REGION Network 22: Salidas Mesas
   RUNG wire#powerrail
      Contact( TRUE )
      wire#w1
      Contact( #Avance_E1 )
      Coil( "DB900_Estado_Mesas".EstadoVI[#Mesa].Sa_Rod_Avance )
   END_RUNG
   RUNG wire#w1
      Contact( #Avance_S2 )
      Coil( "DB900_Estado_Mesas".EstadoVI[#Mesa].Sa_Cad_Avance )
   END_RUNG
   RUNG wire#w1
      Contact( #TEMP_MA_TR_Pos_E1 )
      Coil( "DB900_Estado_Mesas".EstadoVI[#Mesa].Sa_Trans_Sub )
   END_RUNG
   RUNG wire#w1
      Contact( #TEMP_MA_TR_Pos_S2 )
      Coil( "DB900_Estado_Mesas".EstadoVI[#Mesa].Sa_Trans_Baj )
   END_RUNG
   // the same network as SCL:
   "DB900_Estado_Mesas".EstadoVI[#Mesa].Sa_Rod_Avance := TRUE AND #Avance_E1;
   "DB900_Estado_Mesas".EstadoVI[#Mesa].Sa_Cad_Avance := TRUE AND #Avance_S2;
   "DB900_Estado_Mesas".EstadoVI[#Mesa].Sa_Trans_Sub := TRUE AND #TEMP_MA_TR_Pos_E1;
   "DB900_Estado_Mesas".EstadoVI[#Mesa].Sa_Trans_Baj := TRUE AND #TEMP_MA_TR_Pos_S2;
END_REGION

REGION Network 23: Etapa MESA en RESET
   RUNG wire#powerrail
      Contact( TRUE )
      wire#w1
      Contact( "DB902_Estado_ZonaMesa".EstadoMesas[#Mesa].PerReset_CBx )
      Coil( "DB900_Estado_Mesas".EstadoVI[#Mesa].Etapas_Reset )
   END_RUNG
   RUNG wire#w1
      Contact( #Avance_E1 )
      Coil( "DB900_Estado_Mesas".EstadoVI[#Mesa].Etapas_Carga_E1 )
   END_RUNG
   RUNG wire#w1
      Contact( #Avance_S2 )
      Coil( "DB900_Estado_Mesas".EstadoVI[#Mesa].Etapas_Descarga_S2 )
   END_RUNG
   RUNG wire#w1
      I_Contact( #Avance_E1 )
      I_Contact( #Avance_S2 )
      Contact( #PhsMx )
      Coil( "DB900_Estado_Mesas".EstadoVI[#Mesa].Etapa_Cargada )
   END_RUNG
   RUNG wire#w1
      I_Contact( #Avance_E1 )
      I_Contact( #Avance_S2 )
      I_Contact( #PhsMx )
      Coil( "DB900_Estado_Mesas".EstadoVI[#Mesa].Etapa_Vacia )
   END_RUNG
   // the same network as SCL:
   "DB900_Estado_Mesas".EstadoVI[#Mesa].Etapas_Reset := TRUE AND "DB902_Estado_ZonaMesa".EstadoMesas[#Mesa].PerReset_CBx;
   "DB900_Estado_Mesas".EstadoVI[#Mesa].Etapas_Carga_E1 := TRUE AND #Avance_E1;
   "DB900_Estado_Mesas".EstadoVI[#Mesa].Etapas_Descarga_S2 := TRUE AND #Avance_S2;
   "DB900_Estado_Mesas".EstadoVI[#Mesa].Etapa_Cargada := TRUE AND NOT #Avance_E1 AND NOT #Avance_S2 AND #PhsMx;
   "DB900_Estado_Mesas".EstadoVI[#Mesa].Etapa_Vacia := TRUE AND NOT #Avance_E1 AND NOT #Avance_S2 AND NOT #PhsMx;
END_REGION

REGION Network 24
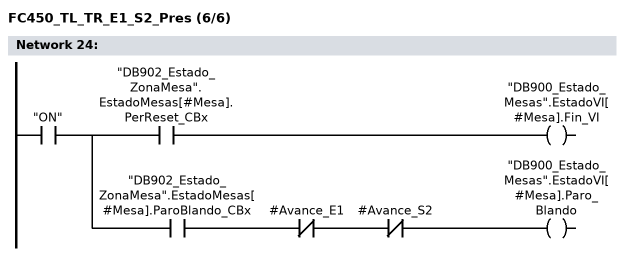
   RUNG wire#powerrail
      Contact( "ON" )
      wire#w1
      Contact( "DB902_Estado_ZonaMesa".EstadoMesas[#Mesa].PerReset_CBx )
      Coil( "DB900_Estado_Mesas".EstadoVI[#Mesa].Fin_VI )
   END_RUNG
   RUNG wire#w1
      Contact( "DB902_Estado_ZonaMesa".EstadoMesas[#Mesa].ParoBlando_CBx )
      I_Contact( #Avance_E1 )
      I_Contact( #Avance_S2 )
      Coil( "DB900_Estado_Mesas".EstadoVI[#Mesa].Paro_Blando )
   END_RUNG
   // the same network as SCL:
   "DB900_Estado_Mesas".EstadoVI[#Mesa].Fin_VI := "ON" AND "DB902_Estado_ZonaMesa".EstadoMesas[#Mesa].PerReset_CBx;
   "DB900_Estado_Mesas".EstadoVI[#Mesa].Paro_Blando := "ON" AND "DB902_Estado_ZonaMesa".EstadoMesas[#Mesa].ParoBlando_CBx AND NOT #Avance_E1 AND NOT #Avance_S2;
END_REGION
END_FUNCTION

FUNCTION "FC451_TL_TR_E1E2_S3_Simul_Pres" : Void   // FC451, LAD
{ S7_Optimized_Access := 'FALSE' }
AUTHOR : TLigero
NAME : 20160208
VERSION : 3.2
// stored: AutoNumber false, SetENOAutomatically false
   VAR_INPUT
      Mesa : UInt;
      En_Tension : Bool;
      PhsMx : Bool;
      Termico_E1 : Bool;
      Termico_E2 : Bool;
      PosTR_E1 : Bool;
      PosTR_E2 : Bool;
      PosTR_EnReposo_E2 : Bool;   // Si está a false la posición de reposo será E1
      Avance_E1_Tx_Ok : Bool;
      Avance_E2_Tx_Ok : Bool;
      AVTF_Ent_M1 : Bool;
      AVTF_Ent_M2 : Bool;
      NXT_Avance : Bool;
      PTF_Mx_MSig : Bool;
      V_CNT_ApHsMx : UDInt;
      V_Paro : UDInt;
      V_Separacion : UDInt;
      V_Caja_Max : UDInt;
      V_CNT_pHsMx_E1 : UDInt;
      V_CNT_pHsMx_E2 : UDInt;
      V_TOut_Tx_Mx : UDInt;
      V_TOut_TR : UDInt;
      V_Reparto_E1_E2 : UDInt;   // cuantas cajas de E1 dejamos pasar antes de forzar una entrada por E2 (en caso de que siempre haya cajas esperando en ambas entradas)
   END_VAR
   VAR_OUTPUT
      PTF_Ent_M1 : Bool;
      PTF_Ent_M2 : Bool;
      AVTF_Mx_MSig : Bool;
   END_VAR
   VAR_IN_OUT
      NXT_Descarga_Act : Bool;
      Mem_FP_pHs : Bool;
      Mem_FN_pHs : Bool;
   END_VAR
   VAR_TEMP
      Aux_Parar : Bool;
      Mem_CNT_Separacion : Bool;
      Mem_CNT_Pres : Bool;
      atasco : Bool;
      tout_tr : Bool;
      Mem_CNT_Tmp_AUS : Bool;
      Mem_CNT_Tmp_Paro : Bool;
      TEMP_MA_Ir_Pos_E2 : Bool;
      TEMP_MA_Ir_Pos_E1 : Bool;
      ok_tension : Bool;
      Valor_presencia : UDInt;
   END_VAR
   VAR_TEMP   // added for the SCL form of the ladder/FBD networks
      _w1 : Bool;
   END_VAR
BEGIN

REGION Network 1: Marca General Error
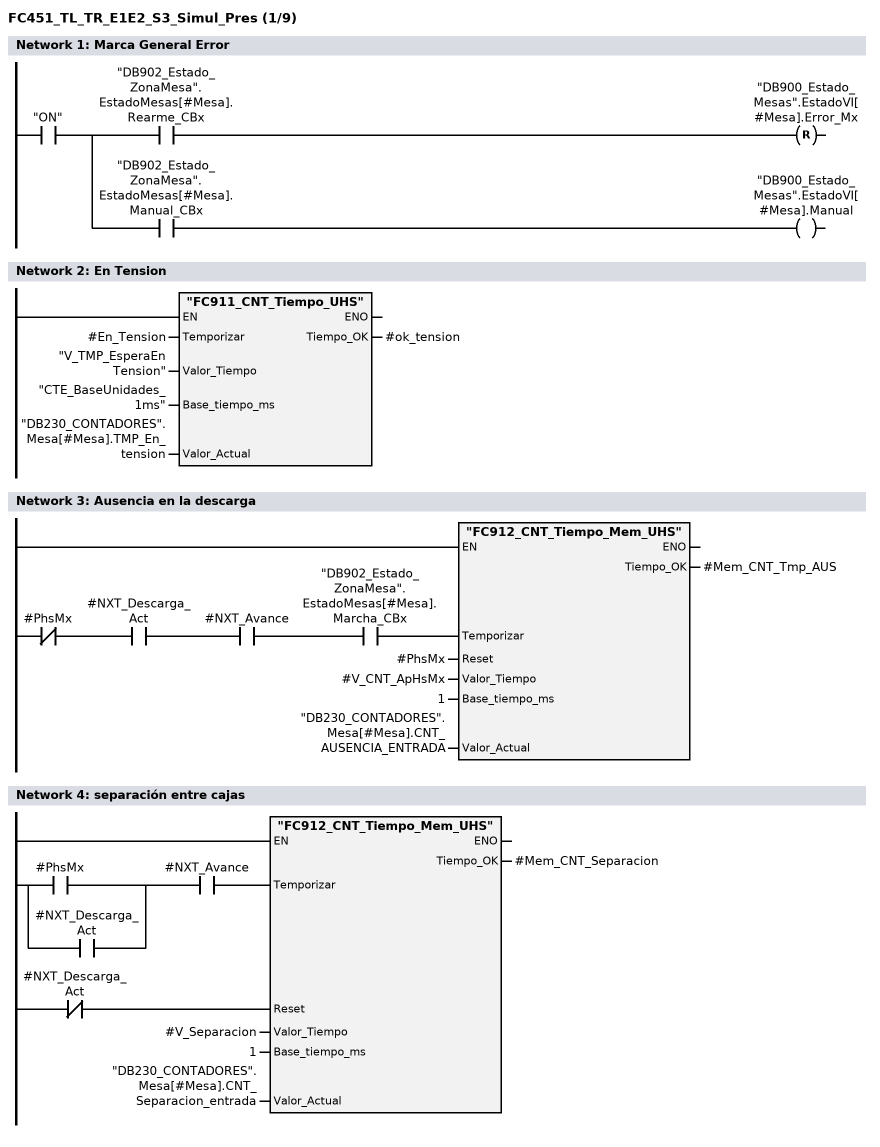
   RUNG wire#powerrail
      Contact( "ON" )
      wire#w1
      Contact( "DB902_Estado_ZonaMesa".EstadoMesas[#Mesa].Rearme_CBx )
      R_Coil( "DB900_Estado_Mesas".EstadoVI[#Mesa].Error_Mx )
   END_RUNG
   RUNG wire#w1
      Contact( "DB902_Estado_ZonaMesa".EstadoMesas[#Mesa].Manual_CBx )
      Coil( "DB900_Estado_Mesas".EstadoVI[#Mesa].Manual )
   END_RUNG
   // the same network as SCL:
   IF "ON" AND "DB902_Estado_ZonaMesa".EstadoMesas[#Mesa].Rearme_CBx THEN
       "DB900_Estado_Mesas".EstadoVI[#Mesa].Error_Mx := FALSE;
   END_IF;
   "DB900_Estado_Mesas".EstadoVI[#Mesa].Manual := "ON" AND "DB902_Estado_ZonaMesa".EstadoMesas[#Mesa].Manual_CBx;
END_REGION

REGION Network 2: En Tension
   RUNG wire#powerrail
      "FC911_CNT_Tiempo_UHS"(Temporizar := #En_Tension, Valor_Tiempo := "V_TMP_EsperaEnTension", Base_tiempo_ms := "CTE_BaseUnidades_1ms", Valor_Actual := "DB230_CONTADORES".Mesa[#Mesa].TMP_En_tension, Tiempo_OK => #ok_tension)
   END_RUNG
   // the same network as SCL:
   "FC911_CNT_Tiempo_UHS"(Temporizar := #En_Tension,
                          Valor_Tiempo := "V_TMP_EsperaEnTension",
                          Base_tiempo_ms := "CTE_BaseUnidades_1ms",
                          Valor_Actual := "DB230_CONTADORES".Mesa[#Mesa].TMP_En_tension,
                          Tiempo_OK => #ok_tension);
END_REGION

REGION Network 3: Ausencia en la descarga
   RUNG wire#powerrail
      "FC912_CNT_Tiempo_Mem_UHS"(Temporizar := wire#w1, Reset := #PhsMx, Valor_Tiempo := #V_CNT_ApHsMx, Base_tiempo_ms := 1, Valor_Actual := "DB230_CONTADORES".Mesa[#Mesa].CNT_AUSENCIA_ENTRADA, Tiempo_OK => #Mem_CNT_Tmp_AUS)
   END_RUNG
   RUNG wire#powerrail
      I_Contact( #PhsMx )
      Contact( #NXT_Descarga_Act )
      Contact( #NXT_Avance )
      Contact( "DB902_Estado_ZonaMesa".EstadoMesas[#Mesa].Marcha_CBx )
   END_RUNG wire#w1
   // the same network as SCL:
   "FC912_CNT_Tiempo_Mem_UHS"(Temporizar := NOT #PhsMx AND #NXT_Descarga_Act AND #NXT_Avance AND "DB902_Estado_ZonaMesa".EstadoMesas[#Mesa].Marcha_CBx,
                           Reset := #PhsMx,
                           Valor_Tiempo := #V_CNT_ApHsMx,
                           Base_tiempo_ms := 1,
                           Valor_Actual := "DB230_CONTADORES".Mesa[#Mesa].CNT_AUSENCIA_ENTRADA,
                           Tiempo_OK => #Mem_CNT_Tmp_AUS);
END_REGION

REGION Network 4: separación entre cajas
   RUNG wire#powerrail
      "FC912_CNT_Tiempo_Mem_UHS"(Temporizar := wire#w2, Reset := wire#w3, Valor_Tiempo := #V_Separacion, Base_tiempo_ms := 1, Valor_Actual := "DB230_CONTADORES".Mesa[#Mesa].CNT_Separacion_entrada, Tiempo_OK => #Mem_CNT_Separacion)
   END_RUNG
   RUNG wire#powerrail
      Contact( #PhsMx )
      wire#w1
      Contact( #NXT_Avance )
   END_RUNG wire#w2
   RUNG wire#powerrail
      Contact( #NXT_Descarga_Act )
   END_RUNG wire#w1
   RUNG wire#powerrail
      I_Contact( #NXT_Descarga_Act )
   END_RUNG wire#w3
   // the same network as SCL:
   "FC912_CNT_Tiempo_Mem_UHS"(Temporizar := (#PhsMx OR #NXT_Descarga_Act) AND #NXT_Avance,
                           Reset := NOT #NXT_Descarga_Act,
                           Valor_Tiempo := #V_Separacion,
                           Base_tiempo_ms := 1,
                           Valor_Actual := "DB230_CONTADORES".Mesa[#Mesa].CNT_Separacion_entrada,
                           Tiempo_OK => #Mem_CNT_Separacion);
END_REGION

REGION Network 5: Valor de presencia
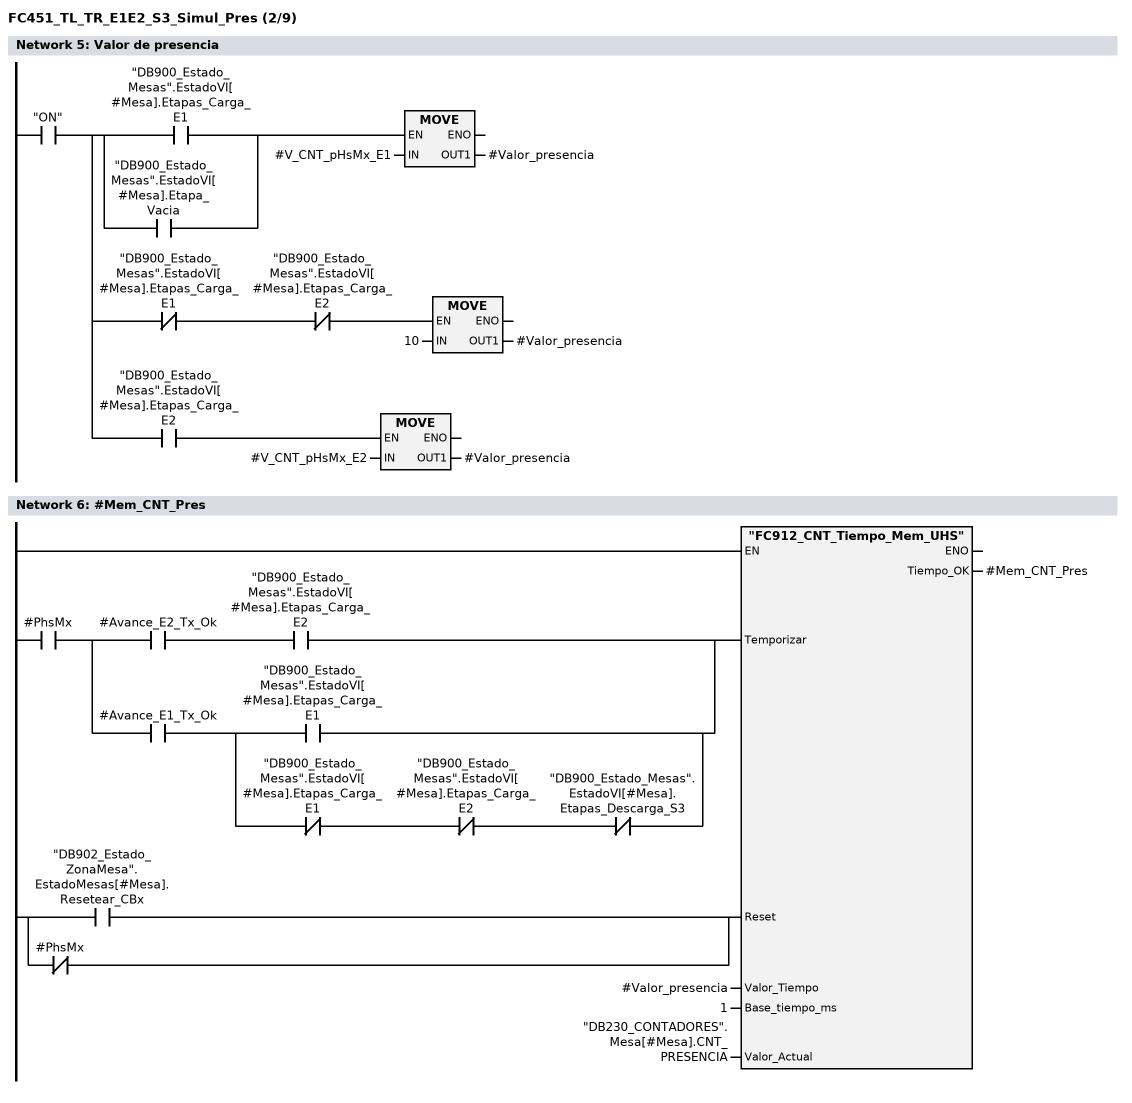
   RUNG wire#powerrail
      Contact( "ON" )
      wire#w1
      Contact( "DB900_Estado_Mesas".EstadoVI[#Mesa].Etapas_Carga_E1 )
      wire#w2
      Move(in := #V_CNT_pHsMx_E1, out1 => #Valor_presencia)
   END_RUNG
   RUNG wire#w1
      Contact( "DB900_Estado_Mesas".EstadoVI[#Mesa].Etapa_Vacia )
   END_RUNG wire#w2
   RUNG wire#w1
      I_Contact( "DB900_Estado_Mesas".EstadoVI[#Mesa].Etapas_Carga_E1 )
      I_Contact( "DB900_Estado_Mesas".EstadoVI[#Mesa].Etapas_Carga_E2 )
      Move(in := 10, out1 => #Valor_presencia)
   END_RUNG
   RUNG wire#w1
      Contact( "DB900_Estado_Mesas".EstadoVI[#Mesa].Etapas_Carga_E2 )
      Move(in := #V_CNT_pHsMx_E2, out1 => #Valor_presencia)
   END_RUNG
   // the same network as SCL:
   IF "ON" AND ("DB900_Estado_Mesas".EstadoVI[#Mesa].Etapas_Carga_E1 OR "DB900_Estado_Mesas".EstadoVI[#Mesa].Etapa_Vacia) THEN
       #Valor_presencia := #V_CNT_pHsMx_E1;
   END_IF;
   IF "ON" AND NOT "DB900_Estado_Mesas".EstadoVI[#Mesa].Etapas_Carga_E1 AND NOT "DB900_Estado_Mesas".EstadoVI[#Mesa].Etapas_Carga_E2 THEN
       #Valor_presencia := 10;
   END_IF;
   IF "ON" AND "DB900_Estado_Mesas".EstadoVI[#Mesa].Etapas_Carga_E2 THEN
       #Valor_presencia := #V_CNT_pHsMx_E2;
   END_IF;
END_REGION

REGION Network 6: #Mem_CNT_Pres
   RUNG wire#powerrail
      "FC912_CNT_Tiempo_Mem_UHS"(Temporizar := wire#w3, Reset := wire#w4, Valor_Tiempo := #Valor_presencia, Base_tiempo_ms := 1, Valor_Actual := "DB230_CONTADORES".Mesa[#Mesa].CNT_PRESENCIA, Tiempo_OK => #Mem_CNT_Pres)
   END_RUNG
   RUNG wire#powerrail
      Contact( #PhsMx )
      wire#w1
      Contact( #Avance_E2_Tx_Ok )
      Contact( "DB900_Estado_Mesas".EstadoVI[#Mesa].Etapas_Carga_E2 )
   END_RUNG wire#w3
   RUNG wire#w1
      Contact( #Avance_E1_Tx_Ok )
      wire#w2
      Contact( "DB900_Estado_Mesas".EstadoVI[#Mesa].Etapas_Carga_E1 )
   END_RUNG wire#w3
   RUNG wire#w2
      I_Contact( "DB900_Estado_Mesas".EstadoVI[#Mesa].Etapas_Carga_E1 )
      I_Contact( "DB900_Estado_Mesas".EstadoVI[#Mesa].Etapas_Carga_E2 )
      I_Contact( "DB900_Estado_Mesas".EstadoVI[#Mesa].Etapas_Descarga_S3 )
   END_RUNG wire#w3
   RUNG wire#powerrail
      Contact( "DB902_Estado_ZonaMesa".EstadoMesas[#Mesa].Resetear_CBx )
   END_RUNG wire#w4
   RUNG wire#powerrail
      I_Contact( #PhsMx )
   END_RUNG wire#w4
   // the same network as SCL:
   "FC912_CNT_Tiempo_Mem_UHS"(Temporizar := #PhsMx AND ((#Avance_E2_Tx_Ok AND "DB900_Estado_Mesas".EstadoVI[#Mesa].Etapas_Carga_E2) OR (#Avance_E1_Tx_Ok AND ("DB900_Estado_Mesas".EstadoVI[#Mesa].Etapas_Carga_E1 OR (NOT "DB900_Estado_Mesas".EstadoVI[#Mesa].Etapas_Carga_E1 AND NOT "DB900_Estado_Mesas".EstadoVI[#Mesa].Etapas_Carga_E2 AND NOT "DB900_Estado_Mesas".EstadoVI[#Mesa].Etapas_Descarga_S3)))),
                           Reset := "DB902_Estado_ZonaMesa".EstadoMesas[#Mesa].Resetear_CBx OR NOT #PhsMx,
                           Valor_Tiempo := #Valor_presencia,
                           Base_tiempo_ms := 1,
                           Valor_Actual := "DB230_CONTADORES".Mesa[#Mesa].CNT_PRESENCIA,
                           Tiempo_OK => #Mem_CNT_Pres);
END_REGION

REGION Network 7: Temporizador PARO
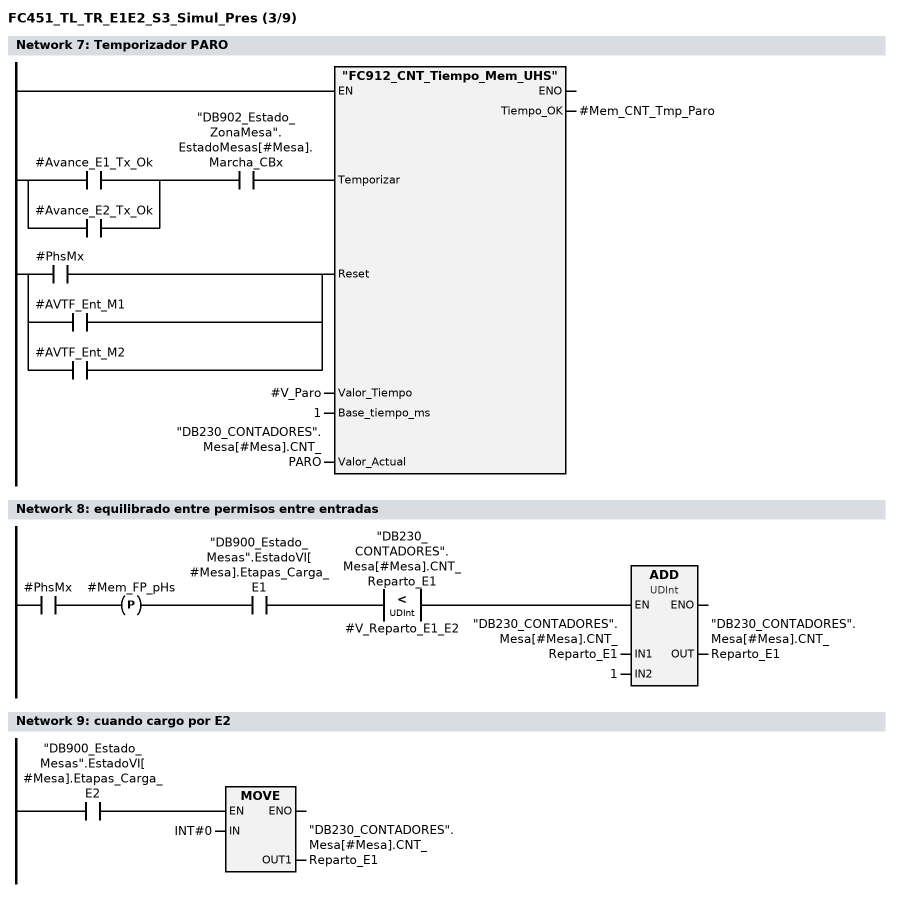
   RUNG wire#powerrail
      "FC912_CNT_Tiempo_Mem_UHS"(Temporizar := wire#w2, Reset := wire#w3, Valor_Tiempo := #V_Paro, Base_tiempo_ms := 1, Valor_Actual := "DB230_CONTADORES".Mesa[#Mesa].CNT_PARO, Tiempo_OK => #Mem_CNT_Tmp_Paro)
   END_RUNG
   RUNG wire#powerrail
      Contact( #Avance_E1_Tx_Ok )
      wire#w1
      Contact( "DB902_Estado_ZonaMesa".EstadoMesas[#Mesa].Marcha_CBx )
   END_RUNG wire#w2
   RUNG wire#powerrail
      Contact( #Avance_E2_Tx_Ok )
   END_RUNG wire#w1
   RUNG wire#powerrail
      Contact( #PhsMx )
   END_RUNG wire#w3
   RUNG wire#powerrail
      Contact( #AVTF_Ent_M1 )
   END_RUNG wire#w3
   RUNG wire#powerrail
      Contact( #AVTF_Ent_M2 )
   END_RUNG wire#w3
   // the same network as SCL:
   "FC912_CNT_Tiempo_Mem_UHS"(Temporizar := (#Avance_E1_Tx_Ok OR #Avance_E2_Tx_Ok) AND "DB902_Estado_ZonaMesa".EstadoMesas[#Mesa].Marcha_CBx,
                           Reset := #PhsMx OR #AVTF_Ent_M1 OR #AVTF_Ent_M2,
                           Valor_Tiempo := #V_Paro,
                           Base_tiempo_ms := 1,
                           Valor_Actual := "DB230_CONTADORES".Mesa[#Mesa].CNT_PARO,
                           Tiempo_OK => #Mem_CNT_Tmp_Paro);
END_REGION

REGION Network 8: equilibrado entre permisos entre entradas
   RUNG wire#powerrail
      Contact( #PhsMx )
      P_Trig( #Mem_FP_pHs )
      Contact( "DB900_Estado_Mesas".EstadoVI[#Mesa].Etapas_Carga_E1 )
      { S7_Templates := "SrcType := UDInt" } LT_Contact(in1 := "DB230_CONTADORES".Mesa[#Mesa].CNT_Reparto_E1, in2 := #V_Reparto_E1_E2)
      { S7_Templates := "SrcType := UDInt"; S7_GenerateENO := "TRUE" } Add(in1 := "DB230_CONTADORES".Mesa[#Mesa].CNT_Reparto_E1, in2 := 1, out => "DB230_CONTADORES".Mesa[#Mesa].CNT_Reparto_E1)
   END_RUNG
   // the same network as SCL:
   #_w1 := #PhsMx AND NOT #Mem_FP_pHs;   // rising edge
   #Mem_FP_pHs := #PhsMx;
   IF #_w1 AND "DB900_Estado_Mesas".EstadoVI[#Mesa].Etapas_Carga_E1 AND ("DB230_CONTADORES".Mesa[#Mesa].CNT_Reparto_E1 < #V_Reparto_E1_E2) THEN
       "DB230_CONTADORES".Mesa[#Mesa].CNT_Reparto_E1 := "DB230_CONTADORES".Mesa[#Mesa].CNT_Reparto_E1 + 1;
   END_IF;
END_REGION

REGION Network 9: cuando cargo por E2
   RUNG wire#powerrail
      Contact( "DB900_Estado_Mesas".EstadoVI[#Mesa].Etapas_Carga_E2 )
      { S7_GenerateENO := "TRUE" } Move(in := INT#0, out1 => "DB230_CONTADORES".Mesa[#Mesa].CNT_Reparto_E1)
   END_RUNG
   // the same network as SCL:
   IF "DB900_Estado_Mesas".EstadoVI[#Mesa].Etapas_Carga_E2 THEN
       "DB230_CONTADORES".Mesa[#Mesa].CNT_Reparto_E1 := INT#0;
   END_IF;
END_REGION

REGION Network 10: Etapas carga E1
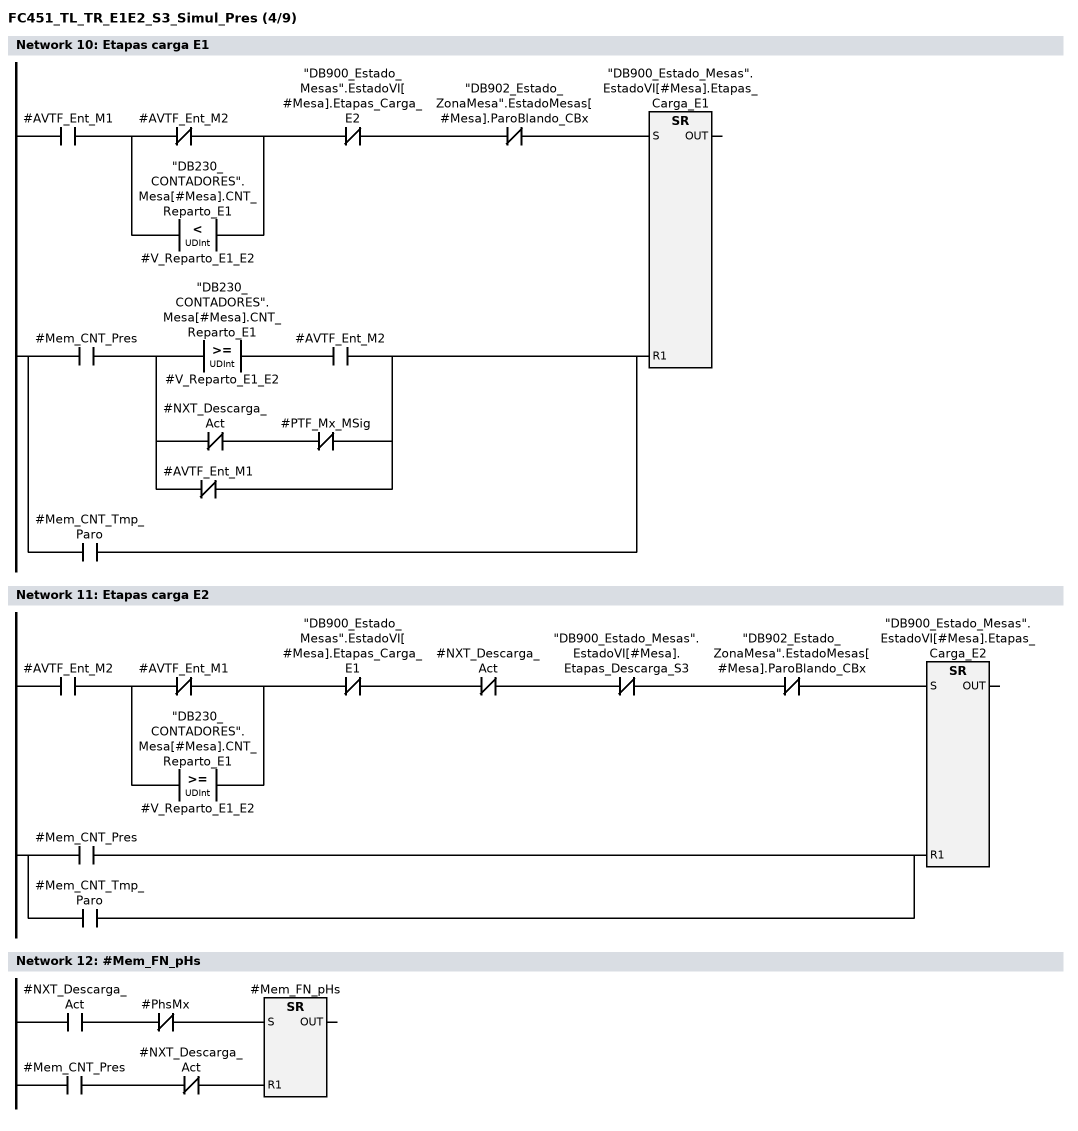
   RUNG wire#powerrail
      Contact( #AVTF_Ent_M1 )
      wire#w1
      I_Contact( #AVTF_Ent_M2 )
      wire#w2
      I_Contact( "DB900_Estado_Mesas".EstadoVI[#Mesa].Etapas_Carga_E2 )
      I_Contact( "DB902_Estado_ZonaMesa".EstadoMesas[#Mesa].ParoBlando_CBx )
      S_SR(operand := "DB900_Estado_Mesas".EstadoVI[#Mesa].Etapas_Carga_E1, r1 := wire#w4)
   END_RUNG
   RUNG wire#w1
      { S7_Templates := "SrcType := UDInt" } LT_Contact(in1 := "DB230_CONTADORES".Mesa[#Mesa].CNT_Reparto_E1, in2 := #V_Reparto_E1_E2)
   END_RUNG wire#w2
   RUNG wire#powerrail
      Contact( #Mem_CNT_Pres )
      wire#w3
      { S7_Templates := "SrcType := UDInt" } GE_Contact(in1 := "DB230_CONTADORES".Mesa[#Mesa].CNT_Reparto_E1, in2 := #V_Reparto_E1_E2)
      Contact( #AVTF_Ent_M2 )
   END_RUNG wire#w4
   RUNG wire#w3
      I_Contact( #NXT_Descarga_Act )
      I_Contact( #PTF_Mx_MSig )
   END_RUNG wire#w4
   RUNG wire#w3
      I_Contact( #AVTF_Ent_M1 )
   END_RUNG wire#w4
   RUNG wire#powerrail
      Contact( #Mem_CNT_Tmp_Paro )
   END_RUNG wire#w4
   // the same network as SCL:
   #_w1 := (#Mem_CNT_Pres AND ((("DB230_CONTADORES".Mesa[#Mesa].CNT_Reparto_E1 >= #V_Reparto_E1_E2) AND #AVTF_Ent_M2) OR (NOT #NXT_Descarga_Act AND NOT #PTF_Mx_MSig) OR NOT #AVTF_Ent_M1)) OR #Mem_CNT_Tmp_Paro;
   IF #AVTF_Ent_M1 AND (NOT #AVTF_Ent_M2 OR ("DB230_CONTADORES".Mesa[#Mesa].CNT_Reparto_E1 < #V_Reparto_E1_E2)) AND NOT "DB900_Estado_Mesas".EstadoVI[#Mesa].Etapas_Carga_E2 AND NOT "DB902_Estado_ZonaMesa".EstadoMesas[#Mesa].ParoBlando_CBx THEN
       "DB900_Estado_Mesas".EstadoVI[#Mesa].Etapas_Carga_E1 := TRUE;   // SR flip-flop
   END_IF;
   IF #_w1 THEN "DB900_Estado_Mesas".EstadoVI[#Mesa].Etapas_Carga_E1 := FALSE; END_IF;
END_REGION

REGION Network 11: Etapas carga E2
   RUNG wire#powerrail
      Contact( #AVTF_Ent_M2 )
      wire#w1
      I_Contact( #AVTF_Ent_M1 )
      wire#w2
      I_Contact( "DB900_Estado_Mesas".EstadoVI[#Mesa].Etapas_Carga_E1 )
      I_Contact( #NXT_Descarga_Act )
      I_Contact( "DB900_Estado_Mesas".EstadoVI[#Mesa].Etapas_Descarga_S3 )
      I_Contact( "DB902_Estado_ZonaMesa".EstadoMesas[#Mesa].ParoBlando_CBx )
      S_SR(operand := "DB900_Estado_Mesas".EstadoVI[#Mesa].Etapas_Carga_E2, r1 := wire#w3)
   END_RUNG
   RUNG wire#w1
      { S7_Templates := "SrcType := UDInt" } GE_Contact(in1 := "DB230_CONTADORES".Mesa[#Mesa].CNT_Reparto_E1, in2 := #V_Reparto_E1_E2)
   END_RUNG wire#w2
   RUNG wire#powerrail
      Contact( #Mem_CNT_Pres )
   END_RUNG wire#w3
   RUNG wire#powerrail
      Contact( #Mem_CNT_Tmp_Paro )
   END_RUNG wire#w3
   // the same network as SCL:
   IF #AVTF_Ent_M2 AND (NOT #AVTF_Ent_M1 OR ("DB230_CONTADORES".Mesa[#Mesa].CNT_Reparto_E1 >= #V_Reparto_E1_E2)) AND NOT "DB900_Estado_Mesas".EstadoVI[#Mesa].Etapas_Carga_E1 AND NOT #NXT_Descarga_Act AND NOT "DB900_Estado_Mesas".EstadoVI[#Mesa].Etapas_Descarga_S3 AND NOT "DB902_Estado_ZonaMesa".EstadoMesas[#Mesa].ParoBlando_CBx THEN
       "DB900_Estado_Mesas".EstadoVI[#Mesa].Etapas_Carga_E2 := TRUE;   // SR flip-flop
   END_IF;
   IF #Mem_CNT_Pres OR #Mem_CNT_Tmp_Paro THEN
       "DB900_Estado_Mesas".EstadoVI[#Mesa].Etapas_Carga_E2 := FALSE;
   END_IF;
END_REGION

REGION Network 12: #Mem_FN_pHs
   RUNG wire#powerrail
      Contact( #NXT_Descarga_Act )
      I_Contact( #PhsMx )
      S_SR(operand := #Mem_FN_pHs, r1 := wire#w1)
   END_RUNG
   RUNG wire#powerrail
      Contact( #Mem_CNT_Pres )
      I_Contact( #NXT_Descarga_Act )
   END_RUNG wire#w1
   // the same network as SCL:
   IF #NXT_Descarga_Act AND NOT #PhsMx THEN
       #Mem_FN_pHs := TRUE;   // SR flip-flop
   END_IF;
   IF #Mem_CNT_Pres AND NOT #NXT_Descarga_Act THEN #Mem_FN_pHs := FALSE; END_IF;
END_REGION

REGION Network 13: #Aux_Parar
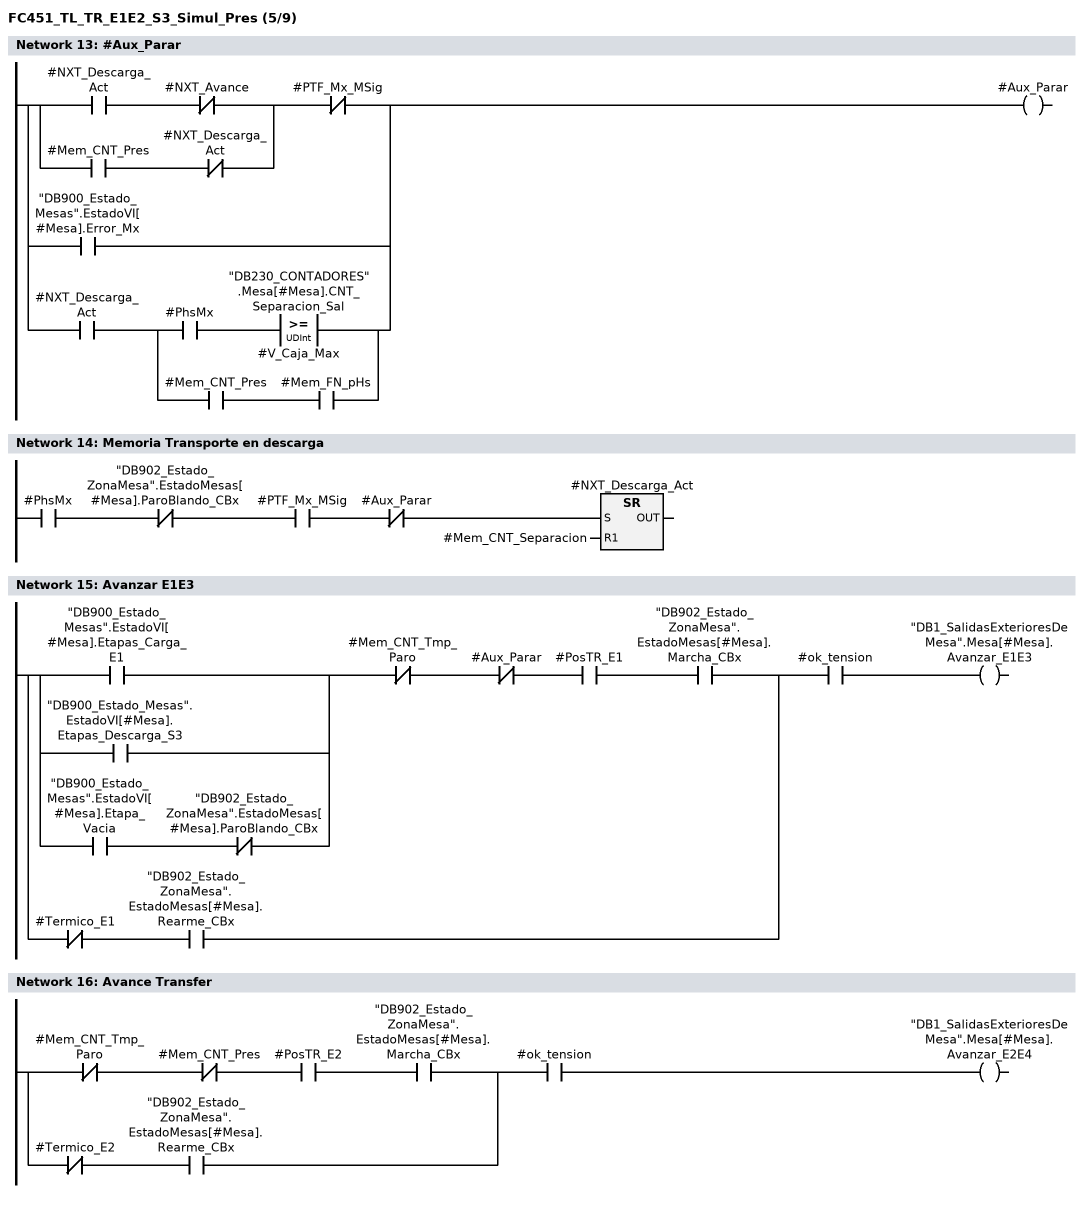
   RUNG wire#powerrail
      Contact( #NXT_Descarga_Act )
      I_Contact( #NXT_Avance )
      wire#w1
      I_Contact( #PTF_Mx_MSig )
      wire#w2
      Coil( #Aux_Parar )
   END_RUNG
   RUNG wire#powerrail
      Contact( #Mem_CNT_Pres )
      I_Contact( #NXT_Descarga_Act )
   END_RUNG wire#w1
   RUNG wire#powerrail
      Contact( "DB900_Estado_Mesas".EstadoVI[#Mesa].Error_Mx )
   END_RUNG wire#w2
   RUNG wire#powerrail
      Contact( #NXT_Descarga_Act )
      wire#w3
      Contact( #PhsMx )
      { S7_Templates := "SrcType := UDInt" } GE_Contact(in1 := "DB230_CONTADORES".Mesa[#Mesa].CNT_Separacion_Sal, in2 := #V_Caja_Max)
   END_RUNG wire#w2
   RUNG wire#w3
      Contact( #Mem_CNT_Pres )
      Contact( #Mem_FN_pHs )
   END_RUNG wire#w2
   // the same network as SCL:
   #Aux_Parar := (((#NXT_Descarga_Act AND NOT #NXT_Avance) OR (#Mem_CNT_Pres AND NOT #NXT_Descarga_Act)) AND NOT #PTF_Mx_MSig) OR "DB900_Estado_Mesas".EstadoVI[#Mesa].Error_Mx OR (#NXT_Descarga_Act AND ((#PhsMx AND ("DB230_CONTADORES".Mesa[#Mesa].CNT_Separacion_Sal >= #V_Caja_Max)) OR (#Mem_CNT_Pres AND #Mem_FN_pHs)));
END_REGION

REGION Network 14: Memoria Transporte en descarga
   RUNG wire#powerrail
      Contact( #PhsMx )
      I_Contact( "DB902_Estado_ZonaMesa".EstadoMesas[#Mesa].ParoBlando_CBx )
      Contact( #PTF_Mx_MSig )
      I_Contact( #Aux_Parar )
      S_SR(operand := #NXT_Descarga_Act, r1 := #Mem_CNT_Separacion)
   END_RUNG
   // the same network as SCL:
   IF #PhsMx AND NOT "DB902_Estado_ZonaMesa".EstadoMesas[#Mesa].ParoBlando_CBx AND #PTF_Mx_MSig AND NOT #Aux_Parar THEN
       #NXT_Descarga_Act := TRUE;   // SR flip-flop
   END_IF;
   IF #Mem_CNT_Separacion THEN #NXT_Descarga_Act := FALSE; END_IF;
END_REGION

REGION Network 15: Avanzar E1E3
   RUNG wire#powerrail
      Contact( "DB900_Estado_Mesas".EstadoVI[#Mesa].Etapas_Carga_E1 )
      wire#w1
      I_Contact( #Mem_CNT_Tmp_Paro )
      I_Contact( #Aux_Parar )
      Contact( #PosTR_E1 )
      Contact( "DB902_Estado_ZonaMesa".EstadoMesas[#Mesa].Marcha_CBx )
      wire#w2
      Contact( #ok_tension )
      Coil( "DB1_SalidasExterioresDeMesa".Mesa[#Mesa].Avanzar_E1E3 )
   END_RUNG
   RUNG wire#powerrail
      Contact( "DB900_Estado_Mesas".EstadoVI[#Mesa].Etapas_Descarga_S3 )
   END_RUNG wire#w1
   RUNG wire#powerrail
      Contact( "DB900_Estado_Mesas".EstadoVI[#Mesa].Etapa_Vacia )
      I_Contact( "DB902_Estado_ZonaMesa".EstadoMesas[#Mesa].ParoBlando_CBx )
   END_RUNG wire#w1
   RUNG wire#powerrail
      I_Contact( #Termico_E1 )
      Contact( "DB902_Estado_ZonaMesa".EstadoMesas[#Mesa].Rearme_CBx )
   END_RUNG wire#w2
   // the same network as SCL:
   "DB1_SalidasExterioresDeMesa".Mesa[#Mesa].Avanzar_E1E3 := ((("DB900_Estado_Mesas".EstadoVI[#Mesa].Etapas_Carga_E1 OR "DB900_Estado_Mesas".EstadoVI[#Mesa].Etapas_Descarga_S3 OR ("DB900_Estado_Mesas".EstadoVI[#Mesa].Etapa_Vacia AND NOT "DB902_Estado_ZonaMesa".EstadoMesas[#Mesa].ParoBlando_CBx)) AND NOT #Mem_CNT_Tmp_Paro AND NOT #Aux_Parar AND #PosTR_E1 AND "DB902_Estado_ZonaMesa".EstadoMesas[#Mesa].Marcha_CBx) OR (NOT #Termico_E1 AND "DB902_Estado_ZonaMesa".EstadoMesas[#Mesa].Rearme_CBx)) AND #ok_tension;
END_REGION

REGION Network 16: Avance Transfer
   RUNG wire#powerrail
      I_Contact( #Mem_CNT_Tmp_Paro )
      I_Contact( #Mem_CNT_Pres )
      Contact( #PosTR_E2 )
      Contact( "DB902_Estado_ZonaMesa".EstadoMesas[#Mesa].Marcha_CBx )
      wire#w1
      Contact( #ok_tension )
      Coil( "DB1_SalidasExterioresDeMesa".Mesa[#Mesa].Avanzar_E2E4 )
   END_RUNG
   RUNG wire#powerrail
      I_Contact( #Termico_E2 )
      Contact( "DB902_Estado_ZonaMesa".EstadoMesas[#Mesa].Rearme_CBx )
   END_RUNG wire#w1
   // the same network as SCL:
   "DB1_SalidasExterioresDeMesa".Mesa[#Mesa].Avanzar_E2E4 := ((NOT #Mem_CNT_Tmp_Paro AND NOT #Mem_CNT_Pres AND #PosTR_E2 AND "DB902_Estado_ZonaMesa".EstadoMesas[#Mesa].Marcha_CBx) OR (NOT #Termico_E2 AND "DB902_Estado_ZonaMesa".EstadoMesas[#Mesa].Rearme_CBx)) AND #ok_tension;
END_REGION

REGION Network 17: Ir_Pos_E2E4
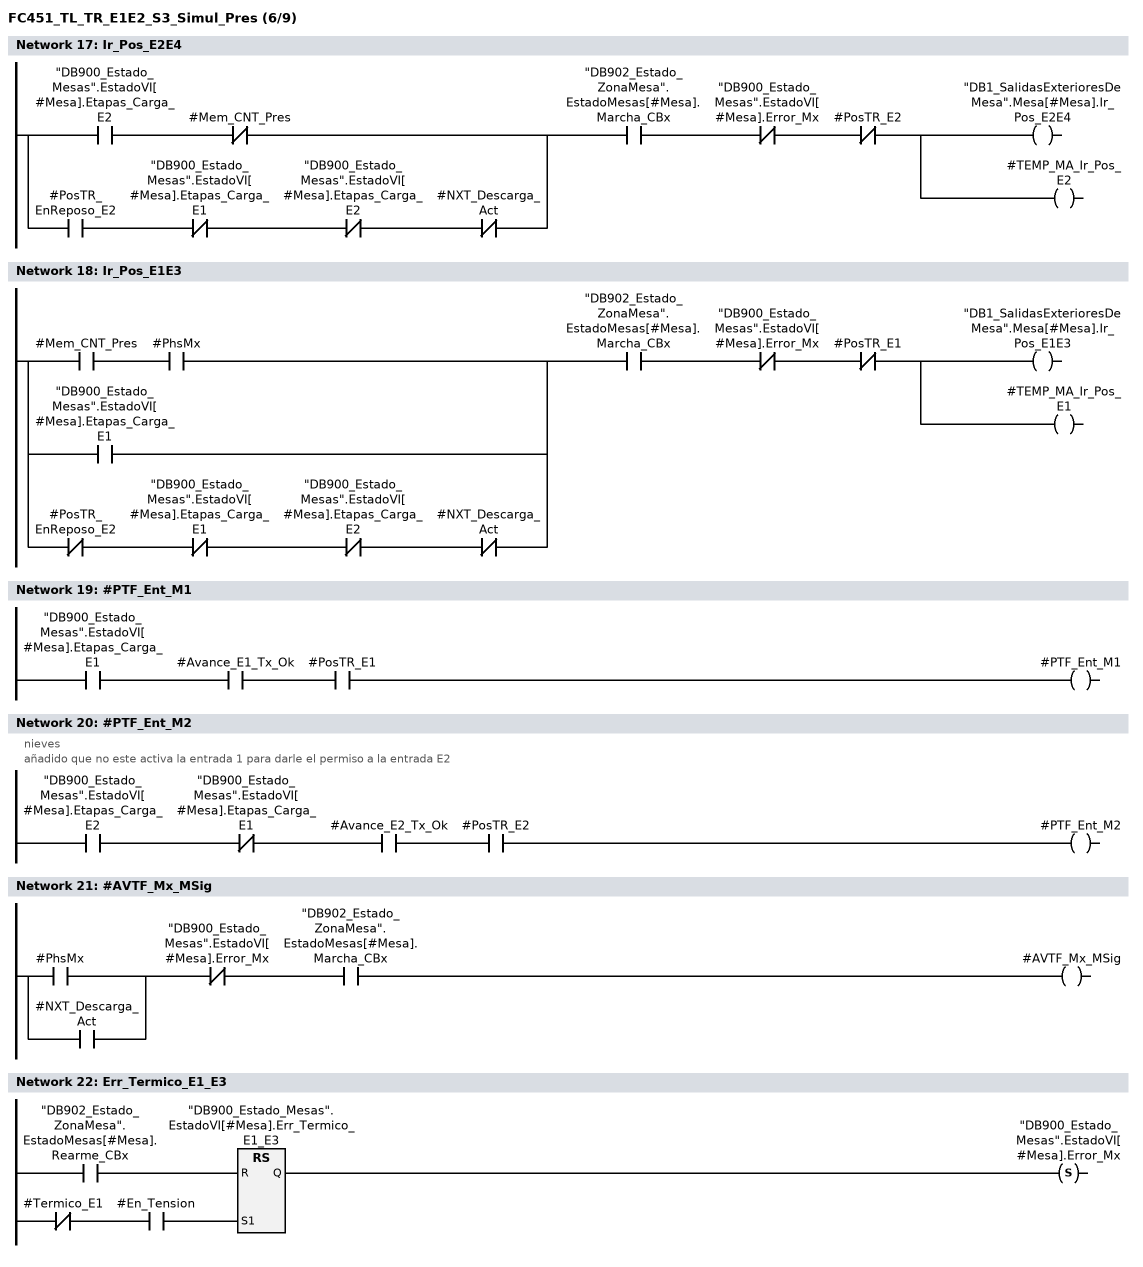
   RUNG wire#powerrail
      Contact( "DB900_Estado_Mesas".EstadoVI[#Mesa].Etapas_Carga_E2 )
      I_Contact( #Mem_CNT_Pres )
      wire#w1
      Contact( "DB902_Estado_ZonaMesa".EstadoMesas[#Mesa].Marcha_CBx )
      I_Contact( "DB900_Estado_Mesas".EstadoVI[#Mesa].Error_Mx )
      I_Contact( #PosTR_E2 )
      wire#w2
      Coil( "DB1_SalidasExterioresDeMesa".Mesa[#Mesa].Ir_Pos_E2E4 )
   END_RUNG
   RUNG wire#powerrail
      Contact( #PosTR_EnReposo_E2 )
      I_Contact( "DB900_Estado_Mesas".EstadoVI[#Mesa].Etapas_Carga_E1 )
      I_Contact( "DB900_Estado_Mesas".EstadoVI[#Mesa].Etapas_Carga_E2 )
      I_Contact( #NXT_Descarga_Act )
   END_RUNG wire#w1
   RUNG wire#w2
      Coil( #TEMP_MA_Ir_Pos_E2 )
   END_RUNG
   // the same network as SCL:
   #_w1 := (("DB900_Estado_Mesas".EstadoVI[#Mesa].Etapas_Carga_E2 AND NOT #Mem_CNT_Pres) OR (#PosTR_EnReposo_E2 AND NOT "DB900_Estado_Mesas".EstadoVI[#Mesa].Etapas_Carga_E1 AND NOT "DB900_Estado_Mesas".EstadoVI[#Mesa].Etapas_Carga_E2 AND NOT #NXT_Descarga_Act)) AND "DB902_Estado_ZonaMesa".EstadoMesas[#Mesa].Marcha_CBx AND NOT "DB900_Estado_Mesas".EstadoVI[#Mesa].Error_Mx AND NOT #PosTR_E2;
   "DB1_SalidasExterioresDeMesa".Mesa[#Mesa].Ir_Pos_E2E4 := (("DB900_Estado_Mesas".EstadoVI[#Mesa].Etapas_Carga_E2 AND NOT #Mem_CNT_Pres) OR (#PosTR_EnReposo_E2 AND NOT "DB900_Estado_Mesas".EstadoVI[#Mesa].Etapas_Carga_E1 AND NOT "DB900_Estado_Mesas".EstadoVI[#Mesa].Etapas_Carga_E2 AND NOT #NXT_Descarga_Act)) AND "DB902_Estado_ZonaMesa".EstadoMesas[#Mesa].Marcha_CBx AND NOT "DB900_Estado_Mesas".EstadoVI[#Mesa].Error_Mx AND NOT #PosTR_E2;
   #TEMP_MA_Ir_Pos_E2 := #_w1;
END_REGION

REGION Network 18: Ir_Pos_E1E3
   RUNG wire#powerrail
      Contact( #Mem_CNT_Pres )
      Contact( #PhsMx )
      wire#w1
      Contact( "DB902_Estado_ZonaMesa".EstadoMesas[#Mesa].Marcha_CBx )
      I_Contact( "DB900_Estado_Mesas".EstadoVI[#Mesa].Error_Mx )
      I_Contact( #PosTR_E1 )
      wire#w2
      Coil( "DB1_SalidasExterioresDeMesa".Mesa[#Mesa].Ir_Pos_E1E3 )
   END_RUNG
   RUNG wire#powerrail
      Contact( "DB900_Estado_Mesas".EstadoVI[#Mesa].Etapas_Carga_E1 )
   END_RUNG wire#w1
   RUNG wire#powerrail
      I_Contact( #PosTR_EnReposo_E2 )
      I_Contact( "DB900_Estado_Mesas".EstadoVI[#Mesa].Etapas_Carga_E1 )
      I_Contact( "DB900_Estado_Mesas".EstadoVI[#Mesa].Etapas_Carga_E2 )
      I_Contact( #NXT_Descarga_Act )
   END_RUNG wire#w1
   RUNG wire#w2
      Coil( #TEMP_MA_Ir_Pos_E1 )
   END_RUNG
   // the same network as SCL:
   #_w1 := ((#Mem_CNT_Pres AND #PhsMx) OR "DB900_Estado_Mesas".EstadoVI[#Mesa].Etapas_Carga_E1 OR (NOT #PosTR_EnReposo_E2 AND NOT "DB900_Estado_Mesas".EstadoVI[#Mesa].Etapas_Carga_E1 AND NOT "DB900_Estado_Mesas".EstadoVI[#Mesa].Etapas_Carga_E2 AND NOT #NXT_Descarga_Act)) AND "DB902_Estado_ZonaMesa".EstadoMesas[#Mesa].Marcha_CBx AND NOT "DB900_Estado_Mesas".EstadoVI[#Mesa].Error_Mx AND NOT #PosTR_E1;
   "DB1_SalidasExterioresDeMesa".Mesa[#Mesa].Ir_Pos_E1E3 := ((#Mem_CNT_Pres AND #PhsMx) OR "DB900_Estado_Mesas".EstadoVI[#Mesa].Etapas_Carga_E1 OR (NOT #PosTR_EnReposo_E2 AND NOT "DB900_Estado_Mesas".EstadoVI[#Mesa].Etapas_Carga_E1 AND NOT "DB900_Estado_Mesas".EstadoVI[#Mesa].Etapas_Carga_E2 AND NOT #NXT_Descarga_Act)) AND "DB902_Estado_ZonaMesa".EstadoMesas[#Mesa].Marcha_CBx AND NOT "DB900_Estado_Mesas".EstadoVI[#Mesa].Error_Mx AND NOT #PosTR_E1;
   #TEMP_MA_Ir_Pos_E1 := #_w1;
END_REGION

REGION Network 19: #PTF_Ent_M1
   RUNG wire#powerrail
      Contact( "DB900_Estado_Mesas".EstadoVI[#Mesa].Etapas_Carga_E1 )
      Contact( #Avance_E1_Tx_Ok )
      Contact( #PosTR_E1 )
      Coil( #PTF_Ent_M1 )
   END_RUNG
   // the same network as SCL:
   #PTF_Ent_M1 := "DB900_Estado_Mesas".EstadoVI[#Mesa].Etapas_Carga_E1 AND #Avance_E1_Tx_Ok AND #PosTR_E1;
END_REGION

REGION Network 20: #PTF_Ent_M2
   // nieves
   // añadido que no este activa la entrada 1 para darle el permiso a la entrada E2
   RUNG wire#powerrail
      Contact( "DB900_Estado_Mesas".EstadoVI[#Mesa].Etapas_Carga_E2 )
      I_Contact( "DB900_Estado_Mesas".EstadoVI[#Mesa].Etapas_Carga_E1 )
      Contact( #Avance_E2_Tx_Ok )
      Contact( #PosTR_E2 )
      Coil( #PTF_Ent_M2 )
   END_RUNG
   // the same network as SCL:
   #PTF_Ent_M2 := "DB900_Estado_Mesas".EstadoVI[#Mesa].Etapas_Carga_E2 AND NOT "DB900_Estado_Mesas".EstadoVI[#Mesa].Etapas_Carga_E1 AND #Avance_E2_Tx_Ok AND #PosTR_E2;
END_REGION

REGION Network 21: #AVTF_Mx_MSig
   RUNG wire#powerrail
      Contact( #PhsMx )
      wire#w1
      I_Contact( "DB900_Estado_Mesas".EstadoVI[#Mesa].Error_Mx )
      Contact( "DB902_Estado_ZonaMesa".EstadoMesas[#Mesa].Marcha_CBx )
      Coil( #AVTF_Mx_MSig )
   END_RUNG
   RUNG wire#powerrail
      Contact( #NXT_Descarga_Act )
   END_RUNG wire#w1
   // the same network as SCL:
   #AVTF_Mx_MSig := (#PhsMx OR #NXT_Descarga_Act) AND NOT "DB900_Estado_Mesas".EstadoVI[#Mesa].Error_Mx AND "DB902_Estado_ZonaMesa".EstadoMesas[#Mesa].Marcha_CBx;
END_REGION

REGION Network 22: Err_Termico_E1_E3
   RUNG wire#powerrail
      Contact( "DB902_Estado_ZonaMesa".EstadoMesas[#Mesa].Rearme_CBx )
      S_RS(operand := "DB900_Estado_Mesas".EstadoVI[#Mesa].Err_Termico_E1_E3, s1 := wire#w1)
      S_Coil( "DB900_Estado_Mesas".EstadoVI[#Mesa].Error_Mx )
   END_RUNG
   RUNG wire#powerrail
      I_Contact( #Termico_E1 )
      Contact( #En_Tension )
   END_RUNG wire#w1
   // the same network as SCL:
   IF "DB902_Estado_ZonaMesa".EstadoMesas[#Mesa].Rearme_CBx THEN
       "DB900_Estado_Mesas".EstadoVI[#Mesa].Err_Termico_E1_E3 := FALSE;   // RS flip-flop
   END_IF;
   IF NOT #Termico_E1 AND #En_Tension THEN
       "DB900_Estado_Mesas".EstadoVI[#Mesa].Err_Termico_E1_E3 := TRUE;
   END_IF;
   IF "DB900_Estado_Mesas".EstadoVI[#Mesa].Err_Termico_E1_E3 THEN
       "DB900_Estado_Mesas".EstadoVI[#Mesa].Error_Mx := TRUE;
   END_IF;
END_REGION

REGION Network 23: Err_Termico_E2_E4
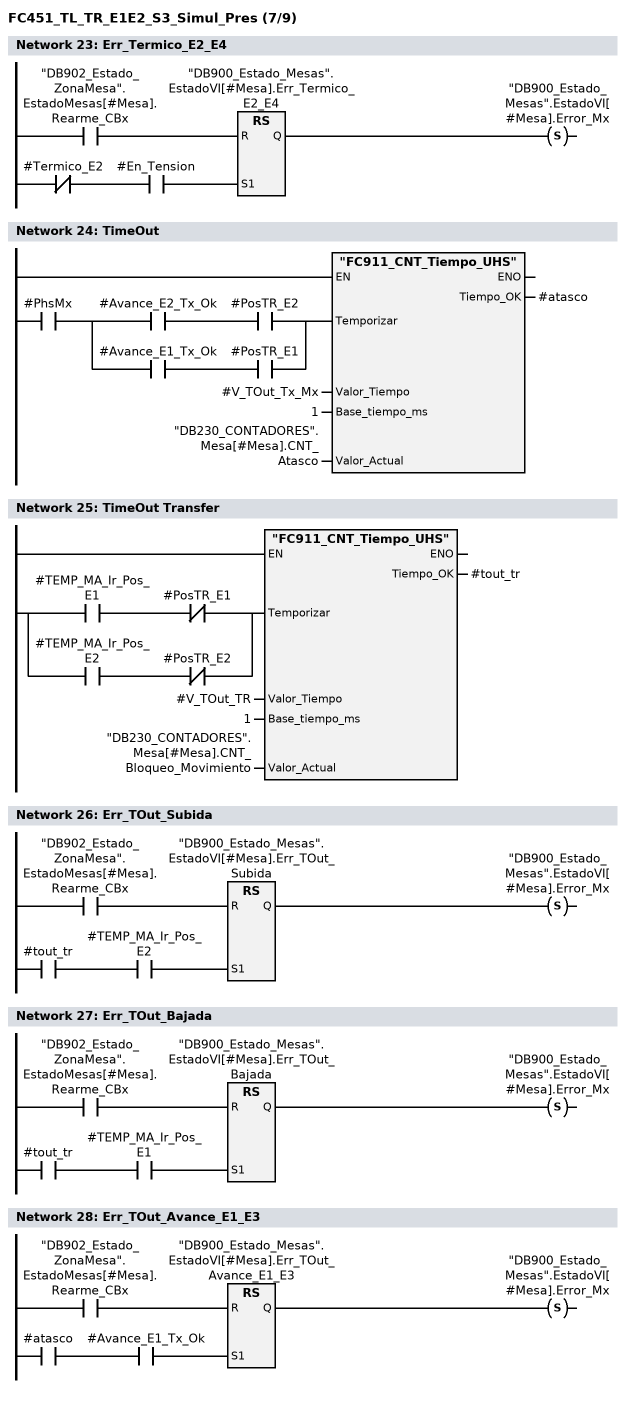
   RUNG wire#powerrail
      Contact( "DB902_Estado_ZonaMesa".EstadoMesas[#Mesa].Rearme_CBx )
      S_RS(operand := "DB900_Estado_Mesas".EstadoVI[#Mesa].Err_Termico_E2_E4, s1 := wire#w1)
      S_Coil( "DB900_Estado_Mesas".EstadoVI[#Mesa].Error_Mx )
   END_RUNG
   RUNG wire#powerrail
      I_Contact( #Termico_E2 )
      Contact( #En_Tension )
   END_RUNG wire#w1
   // the same network as SCL:
   IF "DB902_Estado_ZonaMesa".EstadoMesas[#Mesa].Rearme_CBx THEN
       "DB900_Estado_Mesas".EstadoVI[#Mesa].Err_Termico_E2_E4 := FALSE;   // RS flip-flop
   END_IF;
   IF NOT #Termico_E2 AND #En_Tension THEN
       "DB900_Estado_Mesas".EstadoVI[#Mesa].Err_Termico_E2_E4 := TRUE;
   END_IF;
   IF "DB900_Estado_Mesas".EstadoVI[#Mesa].Err_Termico_E2_E4 THEN
       "DB900_Estado_Mesas".EstadoVI[#Mesa].Error_Mx := TRUE;
   END_IF;
END_REGION

REGION Network 24: TimeOut
   RUNG wire#powerrail
      "FC911_CNT_Tiempo_UHS"(Temporizar := wire#w2, Valor_Tiempo := #V_TOut_Tx_Mx, Base_tiempo_ms := 1, Valor_Actual := "DB230_CONTADORES".Mesa[#Mesa].CNT_Atasco, Tiempo_OK => #atasco)
   END_RUNG
   RUNG wire#powerrail
      Contact( #PhsMx )
      wire#w1
      Contact( #Avance_E2_Tx_Ok )
      Contact( #PosTR_E2 )
   END_RUNG wire#w2
   RUNG wire#w1
      Contact( #Avance_E1_Tx_Ok )
      Contact( #PosTR_E1 )
   END_RUNG wire#w2
   // the same network as SCL:
   "FC911_CNT_Tiempo_UHS"(Temporizar := #PhsMx AND ((#Avance_E2_Tx_Ok AND #PosTR_E2) OR (#Avance_E1_Tx_Ok AND #PosTR_E1)),
                          Valor_Tiempo := #V_TOut_Tx_Mx,
                          Base_tiempo_ms := 1,
                          Valor_Actual := "DB230_CONTADORES".Mesa[#Mesa].CNT_Atasco,
                          Tiempo_OK => #atasco);
END_REGION

REGION Network 25: TimeOut Transfer
   RUNG wire#powerrail
      "FC911_CNT_Tiempo_UHS"(Temporizar := wire#w1, Valor_Tiempo := #V_TOut_TR, Base_tiempo_ms := 1, Valor_Actual := "DB230_CONTADORES".Mesa[#Mesa].CNT_Bloqueo_Movimiento, Tiempo_OK => #tout_tr)
   END_RUNG
   RUNG wire#powerrail
      Contact( #TEMP_MA_Ir_Pos_E1 )
      I_Contact( #PosTR_E1 )
   END_RUNG wire#w1
   RUNG wire#powerrail
      Contact( #TEMP_MA_Ir_Pos_E2 )
      I_Contact( #PosTR_E2 )
   END_RUNG wire#w1
   // the same network as SCL:
   "FC911_CNT_Tiempo_UHS"(Temporizar := (#TEMP_MA_Ir_Pos_E1 AND NOT #PosTR_E1) OR (#TEMP_MA_Ir_Pos_E2 AND NOT #PosTR_E2),
                          Valor_Tiempo := #V_TOut_TR,
                          Base_tiempo_ms := 1,
                          Valor_Actual := "DB230_CONTADORES".Mesa[#Mesa].CNT_Bloqueo_Movimiento,
                          Tiempo_OK => #tout_tr);
END_REGION

REGION Network 26: Err_TOut_Subida
   RUNG wire#powerrail
      Contact( "DB902_Estado_ZonaMesa".EstadoMesas[#Mesa].Rearme_CBx )
      S_RS(operand := "DB900_Estado_Mesas".EstadoVI[#Mesa].Err_TOut_Subida, s1 := wire#w1)
      S_Coil( "DB900_Estado_Mesas".EstadoVI[#Mesa].Error_Mx )
   END_RUNG
   RUNG wire#powerrail
      Contact( #tout_tr )
      Contact( #TEMP_MA_Ir_Pos_E2 )
   END_RUNG wire#w1
   // the same network as SCL:
   IF "DB902_Estado_ZonaMesa".EstadoMesas[#Mesa].Rearme_CBx THEN
       "DB900_Estado_Mesas".EstadoVI[#Mesa].Err_TOut_Subida := FALSE;   // RS flip-flop
   END_IF;
   IF #tout_tr AND #TEMP_MA_Ir_Pos_E2 THEN
       "DB900_Estado_Mesas".EstadoVI[#Mesa].Err_TOut_Subida := TRUE;
   END_IF;
   IF "DB900_Estado_Mesas".EstadoVI[#Mesa].Err_TOut_Subida THEN
       "DB900_Estado_Mesas".EstadoVI[#Mesa].Error_Mx := TRUE;
   END_IF;
END_REGION

REGION Network 27: Err_TOut_Bajada
   RUNG wire#powerrail
      Contact( "DB902_Estado_ZonaMesa".EstadoMesas[#Mesa].Rearme_CBx )
      S_RS(operand := "DB900_Estado_Mesas".EstadoVI[#Mesa].Err_TOut_Bajada, s1 := wire#w1)
      S_Coil( "DB900_Estado_Mesas".EstadoVI[#Mesa].Error_Mx )
   END_RUNG
   RUNG wire#powerrail
      Contact( #tout_tr )
      Contact( #TEMP_MA_Ir_Pos_E1 )
   END_RUNG wire#w1
   // the same network as SCL:
   IF "DB902_Estado_ZonaMesa".EstadoMesas[#Mesa].Rearme_CBx THEN
       "DB900_Estado_Mesas".EstadoVI[#Mesa].Err_TOut_Bajada := FALSE;   // RS flip-flop
   END_IF;
   IF #tout_tr AND #TEMP_MA_Ir_Pos_E1 THEN
       "DB900_Estado_Mesas".EstadoVI[#Mesa].Err_TOut_Bajada := TRUE;
   END_IF;
   IF "DB900_Estado_Mesas".EstadoVI[#Mesa].Err_TOut_Bajada THEN
       "DB900_Estado_Mesas".EstadoVI[#Mesa].Error_Mx := TRUE;
   END_IF;
END_REGION

REGION Network 28: Err_TOut_Avance_E1_E3
   RUNG wire#powerrail
      Contact( "DB902_Estado_ZonaMesa".EstadoMesas[#Mesa].Rearme_CBx )
      S_RS(operand := "DB900_Estado_Mesas".EstadoVI[#Mesa].Err_TOut_Avance_E1_E3, s1 := wire#w1)
      S_Coil( "DB900_Estado_Mesas".EstadoVI[#Mesa].Error_Mx )
   END_RUNG
   RUNG wire#powerrail
      Contact( #atasco )
      Contact( #Avance_E1_Tx_Ok )
   END_RUNG wire#w1
   // the same network as SCL:
   IF "DB902_Estado_ZonaMesa".EstadoMesas[#Mesa].Rearme_CBx THEN
       "DB900_Estado_Mesas".EstadoVI[#Mesa].Err_TOut_Avance_E1_E3 := FALSE;   // RS flip-flop
   END_IF;
   IF #atasco AND #Avance_E1_Tx_Ok THEN
       "DB900_Estado_Mesas".EstadoVI[#Mesa].Err_TOut_Avance_E1_E3 := TRUE;
   END_IF;
   IF "DB900_Estado_Mesas".EstadoVI[#Mesa].Err_TOut_Avance_E1_E3 THEN
       "DB900_Estado_Mesas".EstadoVI[#Mesa].Error_Mx := TRUE;
   END_IF;
END_REGION

REGION Network 29: Err_TOut_Avance_E2_E4
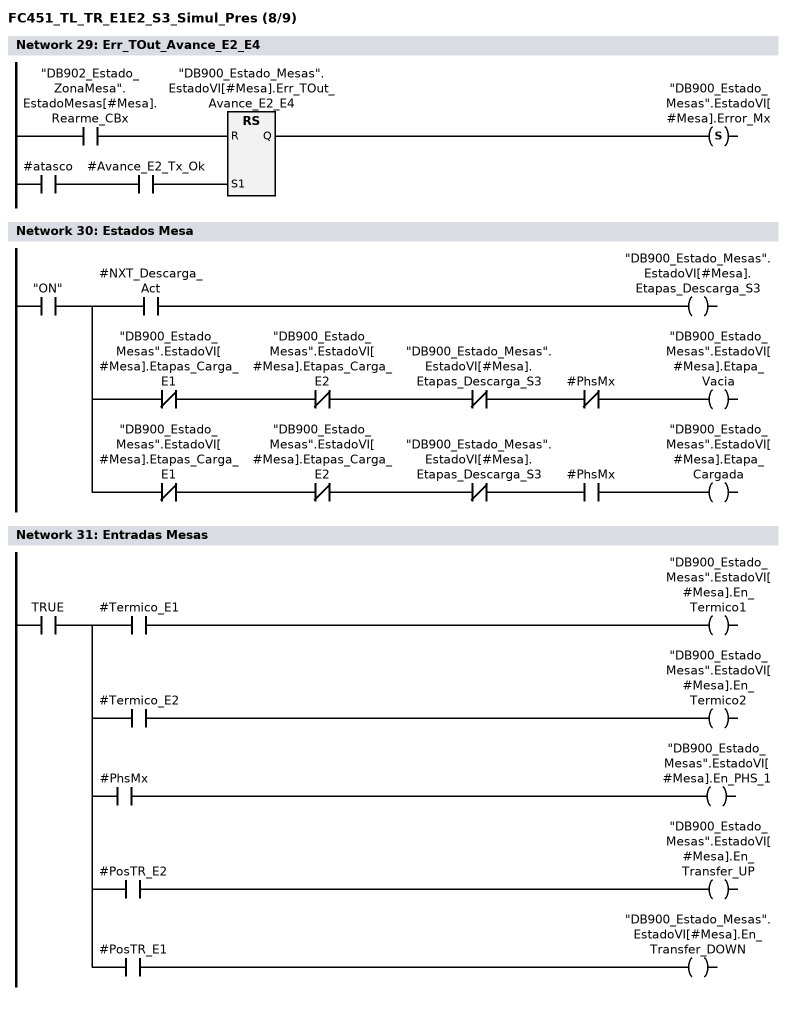
   RUNG wire#powerrail
      Contact( "DB902_Estado_ZonaMesa".EstadoMesas[#Mesa].Rearme_CBx )
      S_RS(operand := "DB900_Estado_Mesas".EstadoVI[#Mesa].Err_TOut_Avance_E2_E4, s1 := wire#w1)
      S_Coil( "DB900_Estado_Mesas".EstadoVI[#Mesa].Error_Mx )
   END_RUNG
   RUNG wire#powerrail
      Contact( #atasco )
      Contact( #Avance_E2_Tx_Ok )
   END_RUNG wire#w1
   // the same network as SCL:
   IF "DB902_Estado_ZonaMesa".EstadoMesas[#Mesa].Rearme_CBx THEN
       "DB900_Estado_Mesas".EstadoVI[#Mesa].Err_TOut_Avance_E2_E4 := FALSE;   // RS flip-flop
   END_IF;
   IF #atasco AND #Avance_E2_Tx_Ok THEN
       "DB900_Estado_Mesas".EstadoVI[#Mesa].Err_TOut_Avance_E2_E4 := TRUE;
   END_IF;
   IF "DB900_Estado_Mesas".EstadoVI[#Mesa].Err_TOut_Avance_E2_E4 THEN
       "DB900_Estado_Mesas".EstadoVI[#Mesa].Error_Mx := TRUE;
   END_IF;
END_REGION

REGION Network 30: Estados Mesa
   RUNG wire#powerrail
      Contact( "ON" )
      wire#w1
      Contact( #NXT_Descarga_Act )
      Coil( "DB900_Estado_Mesas".EstadoVI[#Mesa].Etapas_Descarga_S3 )
   END_RUNG
   RUNG wire#w1
      I_Contact( "DB900_Estado_Mesas".EstadoVI[#Mesa].Etapas_Carga_E1 )
      I_Contact( "DB900_Estado_Mesas".EstadoVI[#Mesa].Etapas_Carga_E2 )
      I_Contact( "DB900_Estado_Mesas".EstadoVI[#Mesa].Etapas_Descarga_S3 )
      I_Contact( #PhsMx )
      Coil( "DB900_Estado_Mesas".EstadoVI[#Mesa].Etapa_Vacia )
   END_RUNG
   RUNG wire#w1
      I_Contact( "DB900_Estado_Mesas".EstadoVI[#Mesa].Etapas_Carga_E1 )
      I_Contact( "DB900_Estado_Mesas".EstadoVI[#Mesa].Etapas_Carga_E2 )
      I_Contact( "DB900_Estado_Mesas".EstadoVI[#Mesa].Etapas_Descarga_S3 )
      Contact( #PhsMx )
      Coil( "DB900_Estado_Mesas".EstadoVI[#Mesa].Etapa_Cargada )
   END_RUNG
   // the same network as SCL:
   "DB900_Estado_Mesas".EstadoVI[#Mesa].Etapas_Descarga_S3 := "ON" AND #NXT_Descarga_Act;
   "DB900_Estado_Mesas".EstadoVI[#Mesa].Etapa_Vacia := "ON" AND NOT "DB900_Estado_Mesas".EstadoVI[#Mesa].Etapas_Carga_E1 AND NOT "DB900_Estado_Mesas".EstadoVI[#Mesa].Etapas_Carga_E2 AND NOT "DB900_Estado_Mesas".EstadoVI[#Mesa].Etapas_Descarga_S3 AND NOT #PhsMx;
   "DB900_Estado_Mesas".EstadoVI[#Mesa].Etapa_Cargada := "ON" AND NOT "DB900_Estado_Mesas".EstadoVI[#Mesa].Etapas_Carga_E1 AND NOT "DB900_Estado_Mesas".EstadoVI[#Mesa].Etapas_Carga_E2 AND NOT "DB900_Estado_Mesas".EstadoVI[#Mesa].Etapas_Descarga_S3 AND #PhsMx;
END_REGION

REGION Network 31: Entradas Mesas
   RUNG wire#powerrail
      Contact( TRUE )
      wire#w1
      Contact( #Termico_E1 )
      Coil( "DB900_Estado_Mesas".EstadoVI[#Mesa].En_Termico1 )
   END_RUNG
   RUNG wire#w1
      Contact( #Termico_E2 )
      Coil( "DB900_Estado_Mesas".EstadoVI[#Mesa].En_Termico2 )
   END_RUNG
   RUNG wire#w1
      Contact( #PhsMx )
      Coil( "DB900_Estado_Mesas".EstadoVI[#Mesa].En_PHS_1 )
   END_RUNG
   RUNG wire#w1
      Contact( #PosTR_E2 )
      Coil( "DB900_Estado_Mesas".EstadoVI[#Mesa].En_Transfer_UP )
   END_RUNG
   RUNG wire#w1
      Contact( #PosTR_E1 )
      Coil( "DB900_Estado_Mesas".EstadoVI[#Mesa].En_Transfer_DOWN )
   END_RUNG
   // the same network as SCL:
   "DB900_Estado_Mesas".EstadoVI[#Mesa].En_Termico1 := TRUE AND #Termico_E1;
   "DB900_Estado_Mesas".EstadoVI[#Mesa].En_Termico2 := TRUE AND #Termico_E2;
   "DB900_Estado_Mesas".EstadoVI[#Mesa].En_PHS_1 := TRUE AND #PhsMx;
   "DB900_Estado_Mesas".EstadoVI[#Mesa].En_Transfer_UP := TRUE AND #PosTR_E2;
   "DB900_Estado_Mesas".EstadoVI[#Mesa].En_Transfer_DOWN := TRUE AND #PosTR_E1;
END_REGION

REGION Network 32: Salidas Mesas
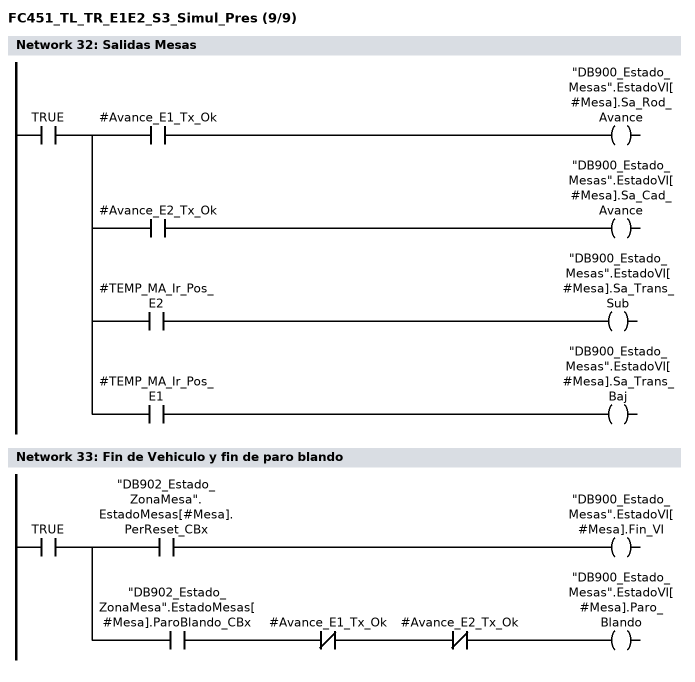
   RUNG wire#powerrail
      Contact( TRUE )
      wire#w1
      Contact( #Avance_E1_Tx_Ok )
      Coil( "DB900_Estado_Mesas".EstadoVI[#Mesa].Sa_Rod_Avance )
   END_RUNG
   RUNG wire#w1
      Contact( #Avance_E2_Tx_Ok )
      Coil( "DB900_Estado_Mesas".EstadoVI[#Mesa].Sa_Cad_Avance )
   END_RUNG
   RUNG wire#w1
      Contact( #TEMP_MA_Ir_Pos_E2 )
      Coil( "DB900_Estado_Mesas".EstadoVI[#Mesa].Sa_Trans_Sub )
   END_RUNG
   RUNG wire#w1
      Contact( #TEMP_MA_Ir_Pos_E1 )
      Coil( "DB900_Estado_Mesas".EstadoVI[#Mesa].Sa_Trans_Baj )
   END_RUNG
   // the same network as SCL:
   "DB900_Estado_Mesas".EstadoVI[#Mesa].Sa_Rod_Avance := TRUE AND #Avance_E1_Tx_Ok;
   "DB900_Estado_Mesas".EstadoVI[#Mesa].Sa_Cad_Avance := TRUE AND #Avance_E2_Tx_Ok;
   "DB900_Estado_Mesas".EstadoVI[#Mesa].Sa_Trans_Sub := TRUE AND #TEMP_MA_Ir_Pos_E2;
   "DB900_Estado_Mesas".EstadoVI[#Mesa].Sa_Trans_Baj := TRUE AND #TEMP_MA_Ir_Pos_E1;
END_REGION

REGION Network 33: Fin de Vehiculo y fin de paro blando
   RUNG wire#powerrail
      Contact( TRUE )
      wire#w1
      Contact( "DB902_Estado_ZonaMesa".EstadoMesas[#Mesa].PerReset_CBx )
      Coil( "DB900_Estado_Mesas".EstadoVI[#Mesa].Fin_VI )
   END_RUNG
   RUNG wire#w1
      Contact( "DB902_Estado_ZonaMesa".EstadoMesas[#Mesa].ParoBlando_CBx )
      I_Contact( #Avance_E1_Tx_Ok )
      I_Contact( #Avance_E2_Tx_Ok )
      Coil( "DB900_Estado_Mesas".EstadoVI[#Mesa].Paro_Blando )
   END_RUNG
   // the same network as SCL:
   "DB900_Estado_Mesas".EstadoVI[#Mesa].Fin_VI := TRUE AND "DB902_Estado_ZonaMesa".EstadoMesas[#Mesa].PerReset_CBx;
   "DB900_Estado_Mesas".EstadoVI[#Mesa].Paro_Blando := TRUE AND "DB902_Estado_ZonaMesa".EstadoMesas[#Mesa].ParoBlando_CBx AND NOT #Avance_E1_Tx_Ok AND NOT #Avance_E2_Tx_Ok;
END_REGION
END_FUNCTION

FUNCTION "FC456_TL_TRE1E2_S3_Simul_Aus" : Void   // FC456, LAD
{ S7_Optimized_Access := 'FALSE' }
AUTHOR : TLigero
NAME : 20160512
VERSION : 3.6
// stored: AutoNumber false, SetENOAutomatically false
   VAR_INPUT
      Mesa : UInt;
      En_Tension : Bool;
      pHsMx_E1 : Bool;
      pHsMx_E2 : Bool;
      pHsMx_S3 : Bool;
      Termico_E1_Tx : Bool;
      Termico_E2_Tx : Bool;
      Avance_E1_Tx_Ok : Bool;
      Avance_S2_Tx_Ok : Bool;
      PosTR_E1 : Bool;
      PosTR_E2 : Bool;
      AVTF_Ent_M1 : Bool;
      AVTF_Ent_M2 : Bool;
      NXT_Avance : Bool;
      PTF_Mx_MSig : Bool;
      PosTR_EnReposo_E2 : Bool;
      V_CNT_ApHsMx_S3 : UDInt;
      V_CNT_ApHsMx_E1 : UDInt;
      V_CNT_ApHsMx_E2 : UDInt;
      V_Paro : UDInt;
      V_TOut_Tx_Mx : UDInt;
      V_TOut_TR : UDInt;
      V_RepartoColector : UDInt;
   END_VAR
   VAR_OUTPUT
      PTF_Ent_M1 : Bool;
      PTF_Ent_M2 : Bool;
      AVTF_Mx_MSig : Bool;
   END_VAR
   VAR_IN_OUT
      MAux_FN_E1 : Bool;
      MemFN_pHsE1 : Bool;
      Maux_FP_pHsE1 : Bool;
      MAux_FN_E2 : Bool;
      MemFN_pHsE2 : Bool;
      MAux_FN_S3 : Bool;
      MemFN_pHsS3 : Bool;
   END_VAR
   VAR_TEMP
      OK_Ausencia_Entrada : Bool;
      OK_Ausencia_Salida : Bool;
      OK_Vaciado : Bool;
      Error_Atasco : Bool;
      Error_TOut_TR : Bool;
      bloqueado : Bool;
      Mem_TmpParo : Bool;
      TEMP_MA_TR_PosE2 : Bool;
      TEMP_MA_TR_PosE1S3 : Bool;
      ok_tension : Bool;
      V_Ausencia_Entrada : UDInt;
   END_VAR
   VAR_TEMP   // added for the SCL form of the ladder/FBD networks
      _w1 : Bool;
      _w2 : Bool;
      _w3 : Bool;
      _w4 : Bool;
      _w5 : Bool;
      _w6 : Bool;
   END_VAR
BEGIN

REGION Network 1: Marca General Error
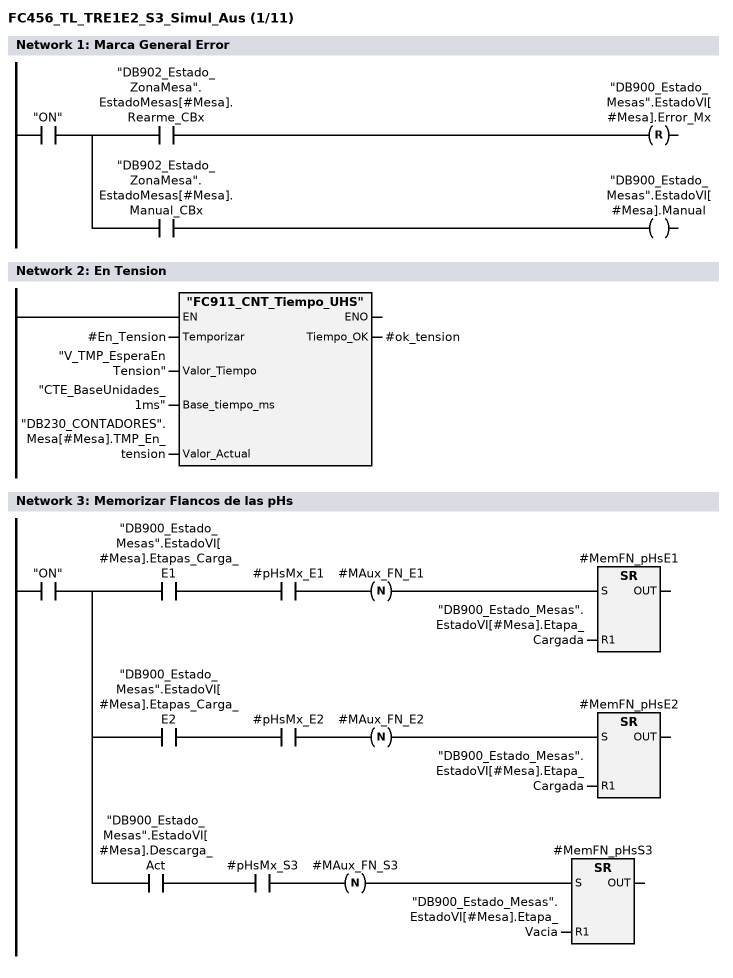
   RUNG wire#powerrail
      Contact( "ON" )
      wire#w1
      Contact( "DB902_Estado_ZonaMesa".EstadoMesas[#Mesa].Rearme_CBx )
      R_Coil( "DB900_Estado_Mesas".EstadoVI[#Mesa].Error_Mx )
   END_RUNG
   RUNG wire#w1
      Contact( "DB902_Estado_ZonaMesa".EstadoMesas[#Mesa].Manual_CBx )
      Coil( "DB900_Estado_Mesas".EstadoVI[#Mesa].Manual )
   END_RUNG
   // the same network as SCL:
   IF "ON" AND "DB902_Estado_ZonaMesa".EstadoMesas[#Mesa].Rearme_CBx THEN
       "DB900_Estado_Mesas".EstadoVI[#Mesa].Error_Mx := FALSE;
   END_IF;
   "DB900_Estado_Mesas".EstadoVI[#Mesa].Manual := "ON" AND "DB902_Estado_ZonaMesa".EstadoMesas[#Mesa].Manual_CBx;
END_REGION

REGION Network 2: En Tension
   RUNG wire#powerrail
      "FC911_CNT_Tiempo_UHS"(Temporizar := #En_Tension, Valor_Tiempo := "V_TMP_EsperaEnTension", Base_tiempo_ms := "CTE_BaseUnidades_1ms", Valor_Actual := "DB230_CONTADORES".Mesa[#Mesa].TMP_En_tension, Tiempo_OK => #ok_tension)
   END_RUNG
   // the same network as SCL:
   "FC911_CNT_Tiempo_UHS"(Temporizar := #En_Tension,
                          Valor_Tiempo := "V_TMP_EsperaEnTension",
                          Base_tiempo_ms := "CTE_BaseUnidades_1ms",
                          Valor_Actual := "DB230_CONTADORES".Mesa[#Mesa].TMP_En_tension,
                          Tiempo_OK => #ok_tension);
END_REGION

REGION Network 3: Memorizar Flancos de las pHs
   RUNG wire#powerrail
      Contact( "ON" )
      wire#w1
      Contact( "DB900_Estado_Mesas".EstadoVI[#Mesa].Etapas_Carga_E1 )
      Contact( #pHsMx_E1 )
      N_Trig( #MAux_FN_E1 )
      S_SR(operand := #MemFN_pHsE1, r1 := "DB900_Estado_Mesas".EstadoVI[#Mesa].Etapa_Cargada)
   END_RUNG
   RUNG wire#w1
      Contact( "DB900_Estado_Mesas".EstadoVI[#Mesa].Etapas_Carga_E2 )
      Contact( #pHsMx_E2 )
      N_Trig( #MAux_FN_E2 )
      S_SR(operand := #MemFN_pHsE2, r1 := "DB900_Estado_Mesas".EstadoVI[#Mesa].Etapa_Cargada)
   END_RUNG
   RUNG wire#w1
      Contact( "DB900_Estado_Mesas".EstadoVI[#Mesa].Descarga_Act )
      Contact( #pHsMx_S3 )
      N_Trig( #MAux_FN_S3 )
      S_SR(operand := #MemFN_pHsS3, r1 := "DB900_Estado_Mesas".EstadoVI[#Mesa].Etapa_Vacia)
   END_RUNG
   // the same network as SCL:
   #_w1 := "ON" AND "DB900_Estado_Mesas".EstadoVI[#Mesa].Etapas_Carga_E1 AND #pHsMx_E1;
   #_w2 := NOT #_w1 AND #MAux_FN_E1;   // falling edge
   #MAux_FN_E1 := #_w1;
   IF #_w2 THEN
       #MemFN_pHsE1 := TRUE;   // SR flip-flop
   END_IF;
   IF "DB900_Estado_Mesas".EstadoVI[#Mesa].Etapa_Cargada THEN #MemFN_pHsE1 := FALSE; END_IF;
   #_w3 := "ON" AND "DB900_Estado_Mesas".EstadoVI[#Mesa].Etapas_Carga_E2 AND #pHsMx_E2;
   #_w4 := NOT #_w3 AND #MAux_FN_E2;   // falling edge
   #MAux_FN_E2 := #_w3;
   IF #_w4 THEN
       #MemFN_pHsE2 := TRUE;   // SR flip-flop
   END_IF;
   IF "DB900_Estado_Mesas".EstadoVI[#Mesa].Etapa_Cargada THEN #MemFN_pHsE2 := FALSE; END_IF;
   #_w5 := "ON" AND "DB900_Estado_Mesas".EstadoVI[#Mesa].Descarga_Act AND #pHsMx_S3;
   #_w6 := NOT #_w5 AND #MAux_FN_S3;   // falling edge
   #MAux_FN_S3 := #_w5;
   IF #_w6 THEN
       #MemFN_pHsS3 := TRUE;   // SR flip-flop
   END_IF;
   IF "DB900_Estado_Mesas".EstadoVI[#Mesa].Etapa_Vacia THEN #MemFN_pHsS3 := FALSE; END_IF;
END_REGION

REGION Network 4: Contador de Ausencia de Salida
   // Contador ausencia
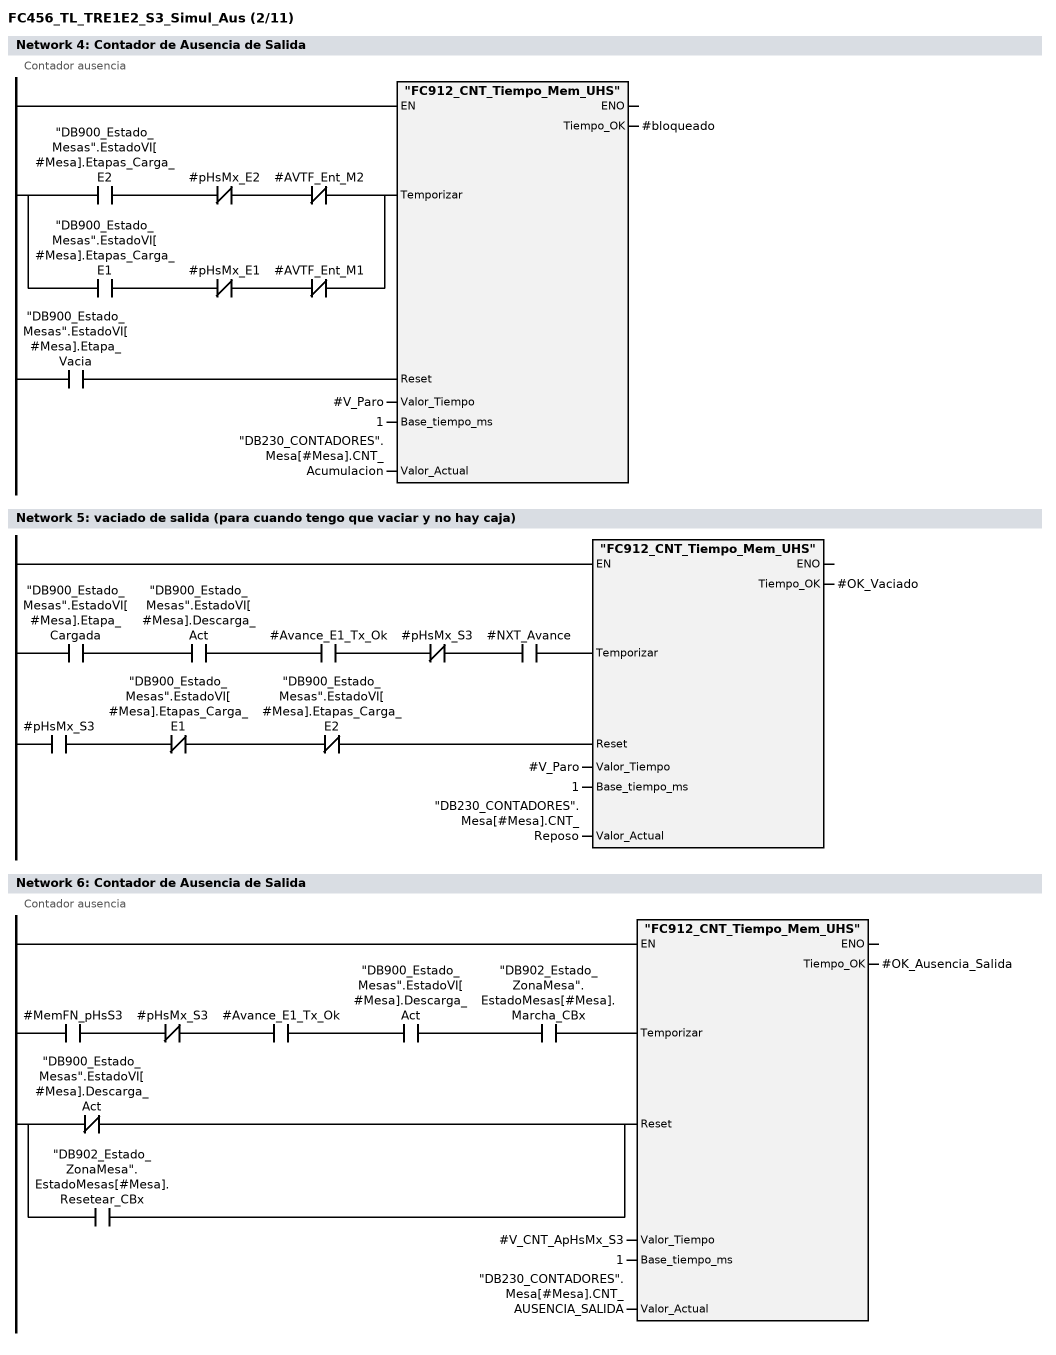
   RUNG wire#powerrail
      "FC912_CNT_Tiempo_Mem_UHS"(Temporizar := wire#w1, Reset := wire#w2, Valor_Tiempo := #V_Paro, Base_tiempo_ms := 1, Valor_Actual := "DB230_CONTADORES".Mesa[#Mesa].CNT_Acumulacion, Tiempo_OK => #bloqueado)
   END_RUNG
   RUNG wire#powerrail
      Contact( "DB900_Estado_Mesas".EstadoVI[#Mesa].Etapas_Carga_E2 )
      I_Contact( #pHsMx_E2 )
      I_Contact( #AVTF_Ent_M2 )
   END_RUNG wire#w1
   RUNG wire#powerrail
      Contact( "DB900_Estado_Mesas".EstadoVI[#Mesa].Etapas_Carga_E1 )
      I_Contact( #pHsMx_E1 )
      I_Contact( #AVTF_Ent_M1 )
   END_RUNG wire#w1
   RUNG wire#powerrail
      Contact( "DB900_Estado_Mesas".EstadoVI[#Mesa].Etapa_Vacia )
   END_RUNG wire#w2
   // the same network as SCL:
   "FC912_CNT_Tiempo_Mem_UHS"(Temporizar := ("DB900_Estado_Mesas".EstadoVI[#Mesa].Etapas_Carga_E2 AND NOT #pHsMx_E2 AND NOT #AVTF_Ent_M2) OR ("DB900_Estado_Mesas".EstadoVI[#Mesa].Etapas_Carga_E1 AND NOT #pHsMx_E1 AND NOT #AVTF_Ent_M1),
                           Reset := "DB900_Estado_Mesas".EstadoVI[#Mesa].Etapa_Vacia,
                           Valor_Tiempo := #V_Paro,
                           Base_tiempo_ms := 1,
                           Valor_Actual := "DB230_CONTADORES".Mesa[#Mesa].CNT_Acumulacion,
                           Tiempo_OK => #bloqueado);
END_REGION

REGION Network 5: vaciado de salida (para cuando tengo que vaciar y no hay caja)
   RUNG wire#powerrail
      "FC912_CNT_Tiempo_Mem_UHS"(Temporizar := wire#w1, Reset := wire#w2, Valor_Tiempo := #V_Paro, Base_tiempo_ms := 1, Valor_Actual := "DB230_CONTADORES".Mesa[#Mesa].CNT_Reposo, Tiempo_OK => #OK_Vaciado)
   END_RUNG
   RUNG wire#powerrail
      Contact( "DB900_Estado_Mesas".EstadoVI[#Mesa].Etapa_Cargada )
      Contact( "DB900_Estado_Mesas".EstadoVI[#Mesa].Descarga_Act )
      Contact( #Avance_E1_Tx_Ok )
      I_Contact( #pHsMx_S3 )
      Contact( #NXT_Avance )
   END_RUNG wire#w1
   RUNG wire#powerrail
      Contact( #pHsMx_S3 )
      I_Contact( "DB900_Estado_Mesas".EstadoVI[#Mesa].Etapas_Carga_E1 )
      I_Contact( "DB900_Estado_Mesas".EstadoVI[#Mesa].Etapas_Carga_E2 )
   END_RUNG wire#w2
   // the same network as SCL:
   "FC912_CNT_Tiempo_Mem_UHS"(Temporizar := "DB900_Estado_Mesas".EstadoVI[#Mesa].Etapa_Cargada AND "DB900_Estado_Mesas".EstadoVI[#Mesa].Descarga_Act AND #Avance_E1_Tx_Ok AND NOT #pHsMx_S3 AND #NXT_Avance,
                           Reset := #pHsMx_S3 AND NOT "DB900_Estado_Mesas".EstadoVI[#Mesa].Etapas_Carga_E1 AND NOT "DB900_Estado_Mesas".EstadoVI[#Mesa].Etapas_Carga_E2,
                           Valor_Tiempo := #V_Paro,
                           Base_tiempo_ms := 1,
                           Valor_Actual := "DB230_CONTADORES".Mesa[#Mesa].CNT_Reposo,
                           Tiempo_OK => #OK_Vaciado);
END_REGION

REGION Network 6: Contador de Ausencia de Salida
   // Contador ausencia
   RUNG wire#powerrail
      "FC912_CNT_Tiempo_Mem_UHS"(Temporizar := wire#w1, Reset := wire#w2, Valor_Tiempo := #V_CNT_ApHsMx_S3, Base_tiempo_ms := 1, Valor_Actual := "DB230_CONTADORES".Mesa[#Mesa].CNT_AUSENCIA_SALIDA, Tiempo_OK => #OK_Ausencia_Salida)
   END_RUNG
   RUNG wire#powerrail
      Contact( #MemFN_pHsS3 )
      I_Contact( #pHsMx_S3 )
      Contact( #Avance_E1_Tx_Ok )
      Contact( "DB900_Estado_Mesas".EstadoVI[#Mesa].Descarga_Act )
      Contact( "DB902_Estado_ZonaMesa".EstadoMesas[#Mesa].Marcha_CBx )
   END_RUNG wire#w1
   RUNG wire#powerrail
      I_Contact( "DB900_Estado_Mesas".EstadoVI[#Mesa].Descarga_Act )
   END_RUNG wire#w2
   RUNG wire#powerrail
      Contact( "DB902_Estado_ZonaMesa".EstadoMesas[#Mesa].Resetear_CBx )
   END_RUNG wire#w2
   // the same network as SCL:
   "FC912_CNT_Tiempo_Mem_UHS"(Temporizar := #MemFN_pHsS3 AND NOT #pHsMx_S3 AND #Avance_E1_Tx_Ok AND "DB900_Estado_Mesas".EstadoVI[#Mesa].Descarga_Act AND "DB902_Estado_ZonaMesa".EstadoMesas[#Mesa].Marcha_CBx,
                           Reset := NOT "DB900_Estado_Mesas".EstadoVI[#Mesa].Descarga_Act OR "DB902_Estado_ZonaMesa".EstadoMesas[#Mesa].Resetear_CBx,
                           Valor_Tiempo := #V_CNT_ApHsMx_S3,
                           Base_tiempo_ms := 1,
                           Valor_Actual := "DB230_CONTADORES".Mesa[#Mesa].CNT_AUSENCIA_SALIDA,
                           Tiempo_OK => #OK_Ausencia_Salida);
END_REGION

REGION Network 7: seleccionar valor de ausencia de entrada en función de la entrada seleccionada
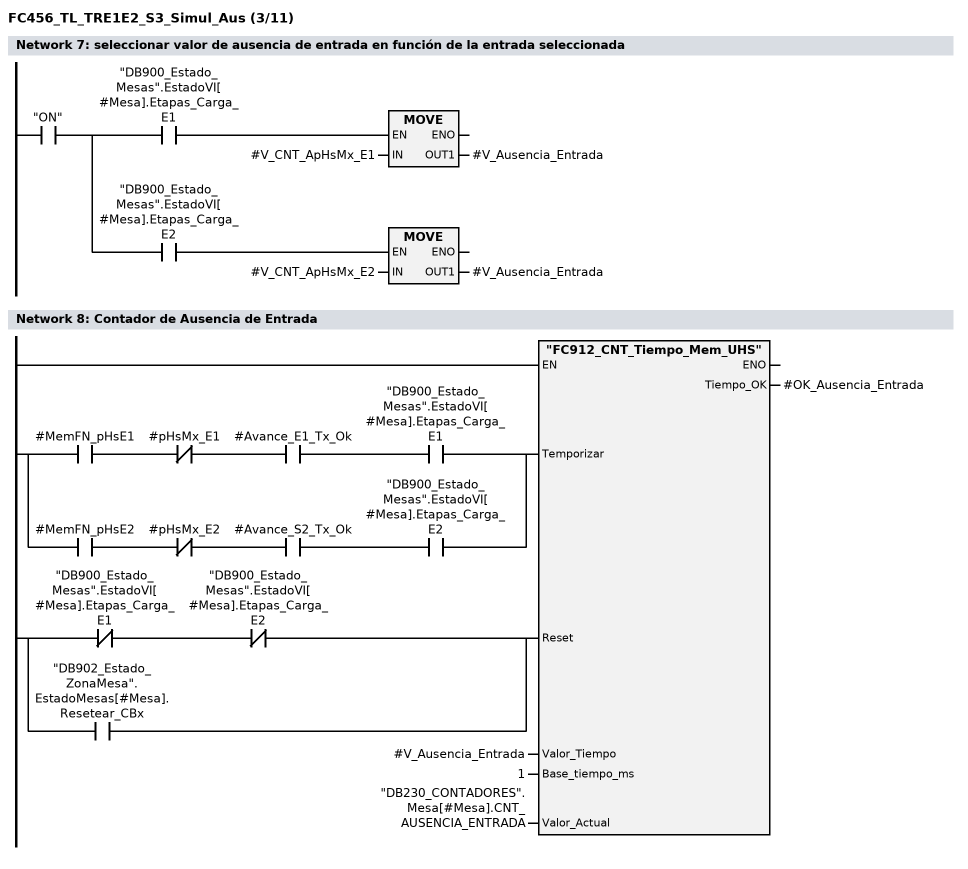
   RUNG wire#powerrail
      Contact( "ON" )
      wire#w1
      Contact( "DB900_Estado_Mesas".EstadoVI[#Mesa].Etapas_Carga_E1 )
      Move(in := #V_CNT_ApHsMx_E1, out1 => #V_Ausencia_Entrada)
   END_RUNG
   RUNG wire#w1
      Contact( "DB900_Estado_Mesas".EstadoVI[#Mesa].Etapas_Carga_E2 )
      Move(in := #V_CNT_ApHsMx_E2, out1 => #V_Ausencia_Entrada)
   END_RUNG
   // the same network as SCL:
   IF "ON" AND "DB900_Estado_Mesas".EstadoVI[#Mesa].Etapas_Carga_E1 THEN
       #V_Ausencia_Entrada := #V_CNT_ApHsMx_E1;
   END_IF;
   IF "ON" AND "DB900_Estado_Mesas".EstadoVI[#Mesa].Etapas_Carga_E2 THEN
       #V_Ausencia_Entrada := #V_CNT_ApHsMx_E2;
   END_IF;
END_REGION

REGION Network 8: Contador de Ausencia de Entrada
   RUNG wire#powerrail
      "FC912_CNT_Tiempo_Mem_UHS"(Temporizar := wire#w1, Reset := wire#w2, Valor_Tiempo := #V_Ausencia_Entrada, Base_tiempo_ms := 1, Valor_Actual := "DB230_CONTADORES".Mesa[#Mesa].CNT_AUSENCIA_ENTRADA, Tiempo_OK => #OK_Ausencia_Entrada)
   END_RUNG
   RUNG wire#powerrail
      Contact( #MemFN_pHsE1 )
      I_Contact( #pHsMx_E1 )
      Contact( #Avance_E1_Tx_Ok )
      Contact( "DB900_Estado_Mesas".EstadoVI[#Mesa].Etapas_Carga_E1 )
   END_RUNG wire#w1
   RUNG wire#powerrail
      Contact( #MemFN_pHsE2 )
      I_Contact( #pHsMx_E2 )
      Contact( #Avance_S2_Tx_Ok )
      Contact( "DB900_Estado_Mesas".EstadoVI[#Mesa].Etapas_Carga_E2 )
   END_RUNG wire#w1
   RUNG wire#powerrail
      I_Contact( "DB900_Estado_Mesas".EstadoVI[#Mesa].Etapas_Carga_E1 )
      I_Contact( "DB900_Estado_Mesas".EstadoVI[#Mesa].Etapas_Carga_E2 )
   END_RUNG wire#w2
   RUNG wire#powerrail
      Contact( "DB902_Estado_ZonaMesa".EstadoMesas[#Mesa].Resetear_CBx )
   END_RUNG wire#w2
   // the same network as SCL:
   "FC912_CNT_Tiempo_Mem_UHS"(Temporizar := (#MemFN_pHsE1 AND NOT #pHsMx_E1 AND #Avance_E1_Tx_Ok AND "DB900_Estado_Mesas".EstadoVI[#Mesa].Etapas_Carga_E1) OR (#MemFN_pHsE2 AND NOT #pHsMx_E2 AND #Avance_S2_Tx_Ok AND "DB900_Estado_Mesas".EstadoVI[#Mesa].Etapas_Carga_E2),
                           Reset := (NOT "DB900_Estado_Mesas".EstadoVI[#Mesa].Etapas_Carga_E1 AND NOT "DB900_Estado_Mesas".EstadoVI[#Mesa].Etapas_Carga_E2) OR "DB902_Estado_ZonaMesa".EstadoMesas[#Mesa].Resetear_CBx,
                           Valor_Tiempo := #V_Ausencia_Entrada,
                           Base_tiempo_ms := 1,
                           Valor_Actual := "DB230_CONTADORES".Mesa[#Mesa].CNT_AUSENCIA_ENTRADA,
                           Tiempo_OK => #OK_Ausencia_Entrada);
END_REGION

REGION Network 9: Temporizador de PARO de E1S3
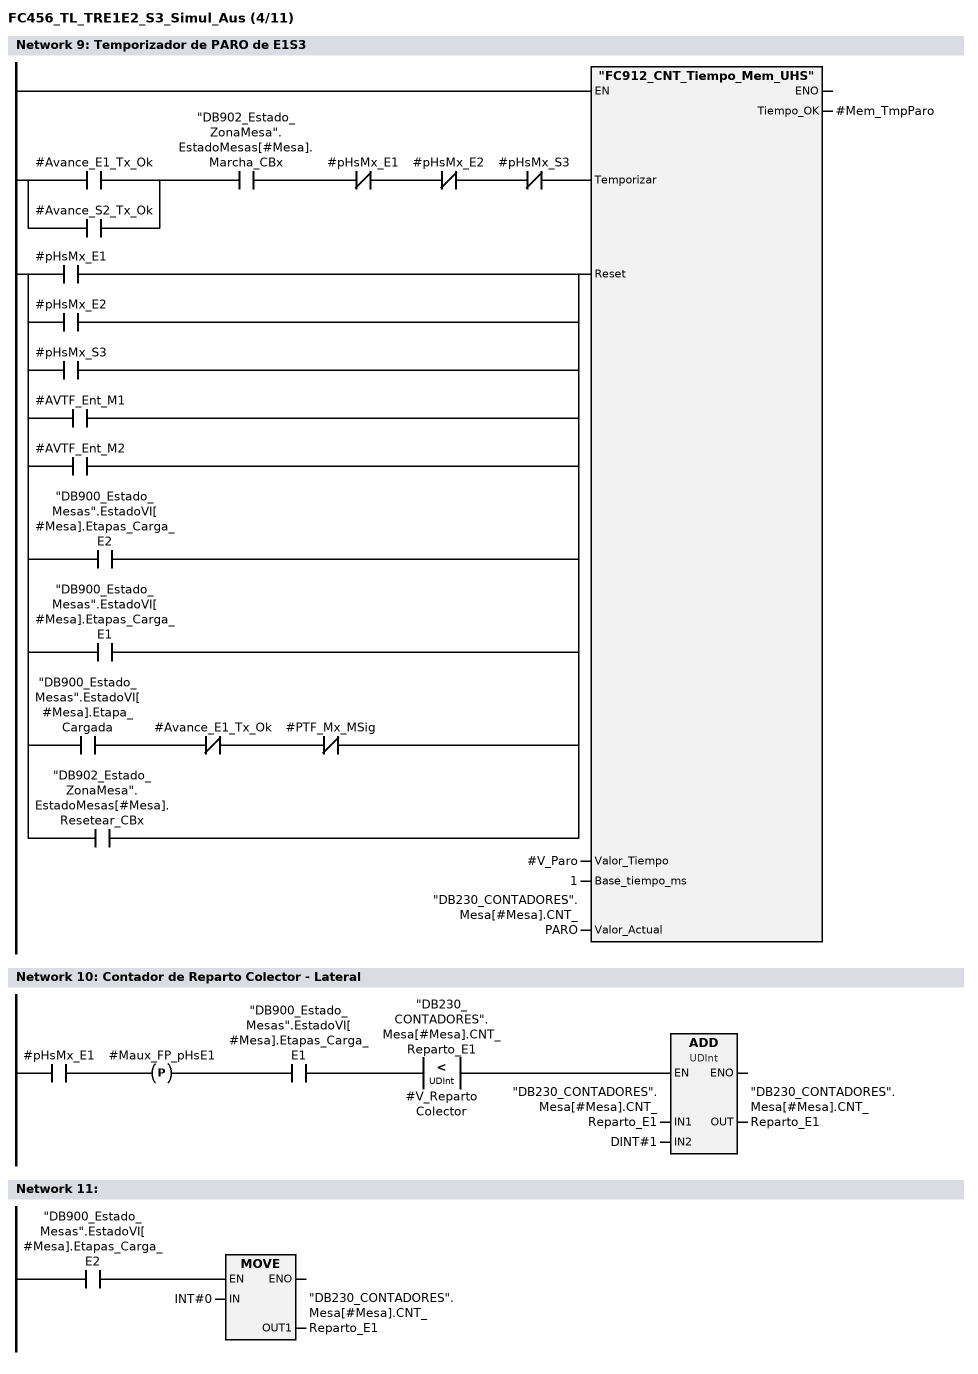
   RUNG wire#powerrail
      "FC912_CNT_Tiempo_Mem_UHS"(Temporizar := wire#w2, Reset := wire#w3, Valor_Tiempo := #V_Paro, Base_tiempo_ms := 1, Valor_Actual := "DB230_CONTADORES".Mesa[#Mesa].CNT_PARO, Tiempo_OK => #Mem_TmpParo)
   END_RUNG
   RUNG wire#powerrail
      Contact( #Avance_E1_Tx_Ok )
      wire#w1
      Contact( "DB902_Estado_ZonaMesa".EstadoMesas[#Mesa].Marcha_CBx )
      I_Contact( #pHsMx_E1 )
      I_Contact( #pHsMx_E2 )
      I_Contact( #pHsMx_S3 )
   END_RUNG wire#w2
   RUNG wire#powerrail
      Contact( #Avance_S2_Tx_Ok )
   END_RUNG wire#w1
   RUNG wire#powerrail
      Contact( #pHsMx_E1 )
   END_RUNG wire#w3
   RUNG wire#powerrail
      Contact( #pHsMx_E2 )
   END_RUNG wire#w3
   RUNG wire#powerrail
      Contact( #pHsMx_S3 )
   END_RUNG wire#w3
   RUNG wire#powerrail
      Contact( #AVTF_Ent_M1 )
   END_RUNG wire#w3
   RUNG wire#powerrail
      Contact( #AVTF_Ent_M2 )
   END_RUNG wire#w3
   RUNG wire#powerrail
      Contact( "DB900_Estado_Mesas".EstadoVI[#Mesa].Etapas_Carga_E2 )
   END_RUNG wire#w3
   RUNG wire#powerrail
      Contact( "DB900_Estado_Mesas".EstadoVI[#Mesa].Etapas_Carga_E1 )
   END_RUNG wire#w3
   RUNG wire#powerrail
      Contact( "DB900_Estado_Mesas".EstadoVI[#Mesa].Etapa_Cargada )
      I_Contact( #Avance_E1_Tx_Ok )
      I_Contact( #PTF_Mx_MSig )
   END_RUNG wire#w3
   RUNG wire#powerrail
      Contact( "DB902_Estado_ZonaMesa".EstadoMesas[#Mesa].Resetear_CBx )
   END_RUNG wire#w3
   // the same network as SCL:
   "FC912_CNT_Tiempo_Mem_UHS"(Temporizar := (#Avance_E1_Tx_Ok OR #Avance_S2_Tx_Ok) AND "DB902_Estado_ZonaMesa".EstadoMesas[#Mesa].Marcha_CBx AND NOT #pHsMx_E1 AND NOT #pHsMx_E2 AND NOT #pHsMx_S3,
                           Reset := #pHsMx_E1 OR #pHsMx_E2 OR #pHsMx_S3 OR #AVTF_Ent_M1 OR #AVTF_Ent_M2 OR "DB900_Estado_Mesas".EstadoVI[#Mesa].Etapas_Carga_E2 OR "DB900_Estado_Mesas".EstadoVI[#Mesa].Etapas_Carga_E1 OR ("DB900_Estado_Mesas".EstadoVI[#Mesa].Etapa_Cargada AND NOT #Avance_E1_Tx_Ok AND NOT #PTF_Mx_MSig) OR "DB902_Estado_ZonaMesa".EstadoMesas[#Mesa].Resetear_CBx,
                           Valor_Tiempo := #V_Paro,
                           Base_tiempo_ms := 1,
                           Valor_Actual := "DB230_CONTADORES".Mesa[#Mesa].CNT_PARO,
                           Tiempo_OK => #Mem_TmpParo);
END_REGION

REGION Network 10: Contador de Reparto Colector - Lateral
   RUNG wire#powerrail
      Contact( #pHsMx_E1 )
      P_Trig( #Maux_FP_pHsE1 )
      Contact( "DB900_Estado_Mesas".EstadoVI[#Mesa].Etapas_Carga_E1 )
      { S7_Templates := "SrcType := UDInt" } LT_Contact(in1 := "DB230_CONTADORES".Mesa[#Mesa].CNT_Reparto_E1, in2 := #V_RepartoColector)
      { S7_Templates := "SrcType := UDInt"; S7_GenerateENO := "TRUE" } Add(in1 := "DB230_CONTADORES".Mesa[#Mesa].CNT_Reparto_E1, in2 := DINT#1, out => "DB230_CONTADORES".Mesa[#Mesa].CNT_Reparto_E1)
   END_RUNG
   // the same network as SCL:
   #_w1 := #pHsMx_E1 AND NOT #Maux_FP_pHsE1;   // rising edge
   #Maux_FP_pHsE1 := #pHsMx_E1;
   IF #_w1 AND "DB900_Estado_Mesas".EstadoVI[#Mesa].Etapas_Carga_E1 AND ("DB230_CONTADORES".Mesa[#Mesa].CNT_Reparto_E1 < #V_RepartoColector) THEN
       "DB230_CONTADORES".Mesa[#Mesa].CNT_Reparto_E1 := "DB230_CONTADORES".Mesa[#Mesa].CNT_Reparto_E1 + DINT#1;
   END_IF;
END_REGION

REGION Network 11
   RUNG wire#powerrail
      Contact( "DB900_Estado_Mesas".EstadoVI[#Mesa].Etapas_Carga_E2 )
      { S7_GenerateENO := "TRUE" } Move(in := INT#0, out1 => "DB230_CONTADORES".Mesa[#Mesa].CNT_Reparto_E1)
   END_RUNG
   // the same network as SCL:
   IF "DB900_Estado_Mesas".EstadoVI[#Mesa].Etapas_Carga_E2 THEN
       "DB230_CONTADORES".Mesa[#Mesa].CNT_Reparto_E1 := INT#0;
   END_IF;
END_REGION

REGION Network 12: Control de Estado de la Mesa
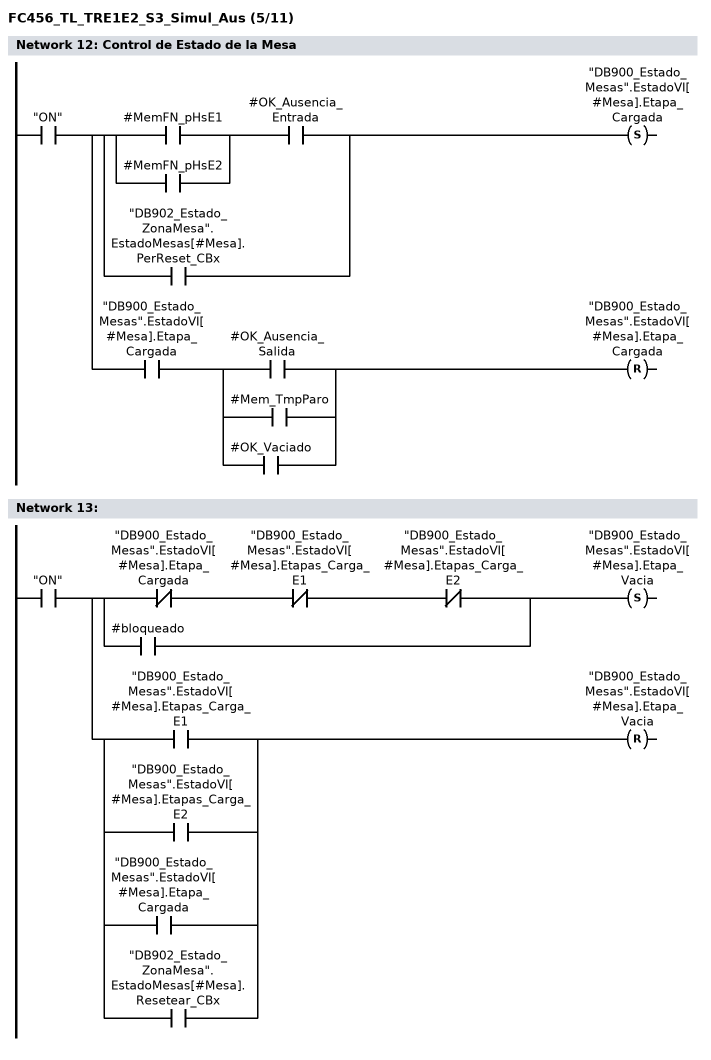
   RUNG wire#powerrail
      Contact( "ON" )
      wire#w1
      Contact( #MemFN_pHsE1 )
      wire#w2
      Contact( #OK_Ausencia_Entrada )
      wire#w3
      S_Coil( "DB900_Estado_Mesas".EstadoVI[#Mesa].Etapa_Cargada )
   END_RUNG
   RUNG wire#w1
      Contact( #MemFN_pHsE2 )
   END_RUNG wire#w2
   RUNG wire#w1
      Contact( "DB902_Estado_ZonaMesa".EstadoMesas[#Mesa].PerReset_CBx )
   END_RUNG wire#w3
   RUNG wire#w1
      Contact( "DB900_Estado_Mesas".EstadoVI[#Mesa].Etapa_Cargada )
      wire#w4
      Contact( #OK_Ausencia_Salida )
      wire#w5
      R_Coil( "DB900_Estado_Mesas".EstadoVI[#Mesa].Etapa_Cargada )
   END_RUNG
   RUNG wire#w4
      Contact( #Mem_TmpParo )
   END_RUNG wire#w5
   RUNG wire#w4
      Contact( #OK_Vaciado )
   END_RUNG wire#w5
   // the same network as SCL:
   IF "ON" AND (((#MemFN_pHsE1 OR #MemFN_pHsE2) AND #OK_Ausencia_Entrada) OR "DB902_Estado_ZonaMesa".EstadoMesas[#Mesa].PerReset_CBx) THEN
       "DB900_Estado_Mesas".EstadoVI[#Mesa].Etapa_Cargada := TRUE;
   END_IF;
   IF "ON" AND "DB900_Estado_Mesas".EstadoVI[#Mesa].Etapa_Cargada AND (#OK_Ausencia_Salida OR #Mem_TmpParo OR #OK_Vaciado) THEN
       "DB900_Estado_Mesas".EstadoVI[#Mesa].Etapa_Cargada := FALSE;
   END_IF;
END_REGION

REGION Network 13
   RUNG wire#powerrail
      Contact( "ON" )
      wire#w1
      I_Contact( "DB900_Estado_Mesas".EstadoVI[#Mesa].Etapa_Cargada )
      I_Contact( "DB900_Estado_Mesas".EstadoVI[#Mesa].Etapas_Carga_E1 )
      I_Contact( "DB900_Estado_Mesas".EstadoVI[#Mesa].Etapas_Carga_E2 )
      wire#w2
      S_Coil( "DB900_Estado_Mesas".EstadoVI[#Mesa].Etapa_Vacia )
   END_RUNG
   RUNG wire#w1
      Contact( #bloqueado )
   END_RUNG wire#w2
   RUNG wire#w1
      Contact( "DB900_Estado_Mesas".EstadoVI[#Mesa].Etapas_Carga_E1 )
      wire#w3
      R_Coil( "DB900_Estado_Mesas".EstadoVI[#Mesa].Etapa_Vacia )
   END_RUNG
   RUNG wire#w1
      Contact( "DB900_Estado_Mesas".EstadoVI[#Mesa].Etapas_Carga_E2 )
   END_RUNG wire#w3
   RUNG wire#w1
      Contact( "DB900_Estado_Mesas".EstadoVI[#Mesa].Etapa_Cargada )
   END_RUNG wire#w3
   RUNG wire#w1
      Contact( "DB902_Estado_ZonaMesa".EstadoMesas[#Mesa].Resetear_CBx )
   END_RUNG wire#w3
   // the same network as SCL:
   IF "ON" AND ((NOT "DB900_Estado_Mesas".EstadoVI[#Mesa].Etapa_Cargada AND NOT "DB900_Estado_Mesas".EstadoVI[#Mesa].Etapas_Carga_E1 AND NOT "DB900_Estado_Mesas".EstadoVI[#Mesa].Etapas_Carga_E2) OR #bloqueado) THEN
       "DB900_Estado_Mesas".EstadoVI[#Mesa].Etapa_Vacia := TRUE;
   END_IF;
   IF "ON" AND ("DB900_Estado_Mesas".EstadoVI[#Mesa].Etapas_Carga_E1 OR "DB900_Estado_Mesas".EstadoVI[#Mesa].Etapas_Carga_E2 OR "DB900_Estado_Mesas".EstadoVI[#Mesa].Etapa_Cargada OR "DB902_Estado_ZonaMesa".EstadoMesas[#Mesa].Resetear_CBx) THEN
       "DB900_Estado_Mesas".EstadoVI[#Mesa].Etapa_Vacia := FALSE;
   END_IF;
END_REGION

REGION Network 14
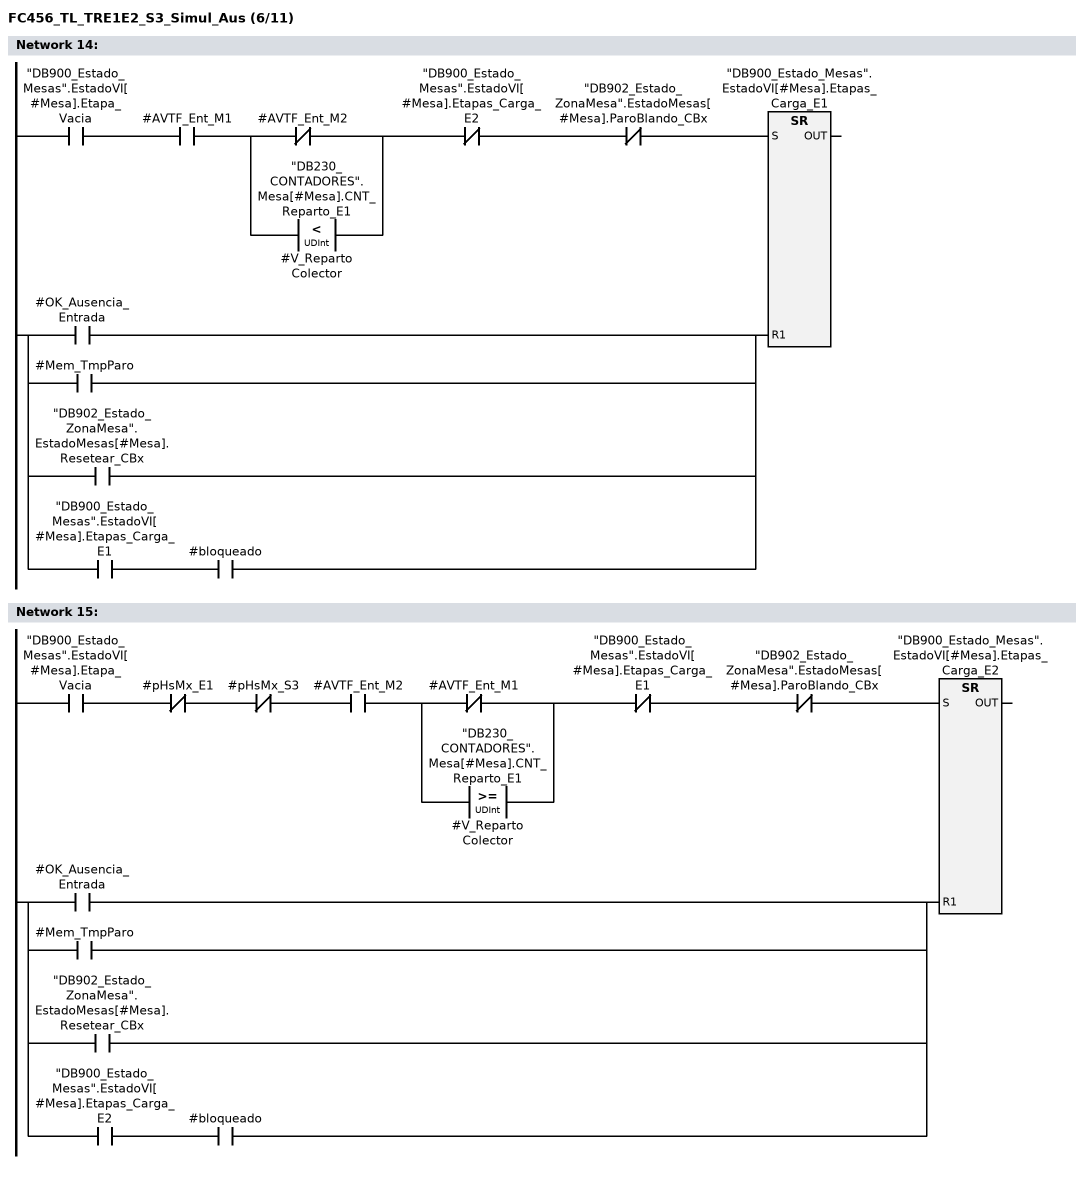
   RUNG wire#powerrail
      Contact( "DB900_Estado_Mesas".EstadoVI[#Mesa].Etapa_Vacia )
      Contact( #AVTF_Ent_M1 )
      wire#w1
      I_Contact( #AVTF_Ent_M2 )
      wire#w2
      I_Contact( "DB900_Estado_Mesas".EstadoVI[#Mesa].Etapas_Carga_E2 )
      I_Contact( "DB902_Estado_ZonaMesa".EstadoMesas[#Mesa].ParoBlando_CBx )
      S_SR(operand := "DB900_Estado_Mesas".EstadoVI[#Mesa].Etapas_Carga_E1, r1 := wire#w3)
   END_RUNG
   RUNG wire#w1
      { S7_Templates := "SrcType := UDInt" } LT_Contact(in1 := "DB230_CONTADORES".Mesa[#Mesa].CNT_Reparto_E1, in2 := #V_RepartoColector)
   END_RUNG wire#w2
   RUNG wire#powerrail
      Contact( #OK_Ausencia_Entrada )
   END_RUNG wire#w3
   RUNG wire#powerrail
      Contact( #Mem_TmpParo )
   END_RUNG wire#w3
   RUNG wire#powerrail
      Contact( "DB902_Estado_ZonaMesa".EstadoMesas[#Mesa].Resetear_CBx )
   END_RUNG wire#w3
   RUNG wire#powerrail
      Contact( "DB900_Estado_Mesas".EstadoVI[#Mesa].Etapas_Carga_E1 )
      Contact( #bloqueado )
   END_RUNG wire#w3
   // the same network as SCL:
   #_w1 := #OK_Ausencia_Entrada OR #Mem_TmpParo OR "DB902_Estado_ZonaMesa".EstadoMesas[#Mesa].Resetear_CBx OR ("DB900_Estado_Mesas".EstadoVI[#Mesa].Etapas_Carga_E1 AND #bloqueado);
   IF "DB900_Estado_Mesas".EstadoVI[#Mesa].Etapa_Vacia AND #AVTF_Ent_M1 AND (NOT #AVTF_Ent_M2 OR ("DB230_CONTADORES".Mesa[#Mesa].CNT_Reparto_E1 < #V_RepartoColector)) AND NOT "DB900_Estado_Mesas".EstadoVI[#Mesa].Etapas_Carga_E2 AND NOT "DB902_Estado_ZonaMesa".EstadoMesas[#Mesa].ParoBlando_CBx THEN
       "DB900_Estado_Mesas".EstadoVI[#Mesa].Etapas_Carga_E1 := TRUE;   // SR flip-flop
   END_IF;
   IF #_w1 THEN "DB900_Estado_Mesas".EstadoVI[#Mesa].Etapas_Carga_E1 := FALSE; END_IF;
END_REGION

REGION Network 15
   RUNG wire#powerrail
      Contact( "DB900_Estado_Mesas".EstadoVI[#Mesa].Etapa_Vacia )
      I_Contact( #pHsMx_E1 )
      I_Contact( #pHsMx_S3 )
      Contact( #AVTF_Ent_M2 )
      wire#w1
      I_Contact( #AVTF_Ent_M1 )
      wire#w2
      I_Contact( "DB900_Estado_Mesas".EstadoVI[#Mesa].Etapas_Carga_E1 )
      I_Contact( "DB902_Estado_ZonaMesa".EstadoMesas[#Mesa].ParoBlando_CBx )
      S_SR(operand := "DB900_Estado_Mesas".EstadoVI[#Mesa].Etapas_Carga_E2, r1 := wire#w3)
   END_RUNG
   RUNG wire#w1
      { S7_Templates := "SrcType := UDInt" } GE_Contact(in1 := "DB230_CONTADORES".Mesa[#Mesa].CNT_Reparto_E1, in2 := #V_RepartoColector)
   END_RUNG wire#w2
   RUNG wire#powerrail
      Contact( #OK_Ausencia_Entrada )
   END_RUNG wire#w3
   RUNG wire#powerrail
      Contact( #Mem_TmpParo )
   END_RUNG wire#w3
   RUNG wire#powerrail
      Contact( "DB902_Estado_ZonaMesa".EstadoMesas[#Mesa].Resetear_CBx )
   END_RUNG wire#w3
   RUNG wire#powerrail
      Contact( "DB900_Estado_Mesas".EstadoVI[#Mesa].Etapas_Carga_E2 )
      Contact( #bloqueado )
   END_RUNG wire#w3
   // the same network as SCL:
   #_w1 := #OK_Ausencia_Entrada OR #Mem_TmpParo OR "DB902_Estado_ZonaMesa".EstadoMesas[#Mesa].Resetear_CBx OR ("DB900_Estado_Mesas".EstadoVI[#Mesa].Etapas_Carga_E2 AND #bloqueado);
   IF "DB900_Estado_Mesas".EstadoVI[#Mesa].Etapa_Vacia AND NOT #pHsMx_E1 AND NOT #pHsMx_S3 AND #AVTF_Ent_M2 AND (NOT #AVTF_Ent_M1 OR ("DB230_CONTADORES".Mesa[#Mesa].CNT_Reparto_E1 >= #V_RepartoColector)) AND NOT "DB900_Estado_Mesas".EstadoVI[#Mesa].Etapas_Carga_E1 AND NOT "DB902_Estado_ZonaMesa".EstadoMesas[#Mesa].ParoBlando_CBx THEN
       "DB900_Estado_Mesas".EstadoVI[#Mesa].Etapas_Carga_E2 := TRUE;   // SR flip-flop
   END_IF;
   IF #_w1 THEN "DB900_Estado_Mesas".EstadoVI[#Mesa].Etapas_Carga_E2 := FALSE; END_IF;
END_REGION

REGION Network 16
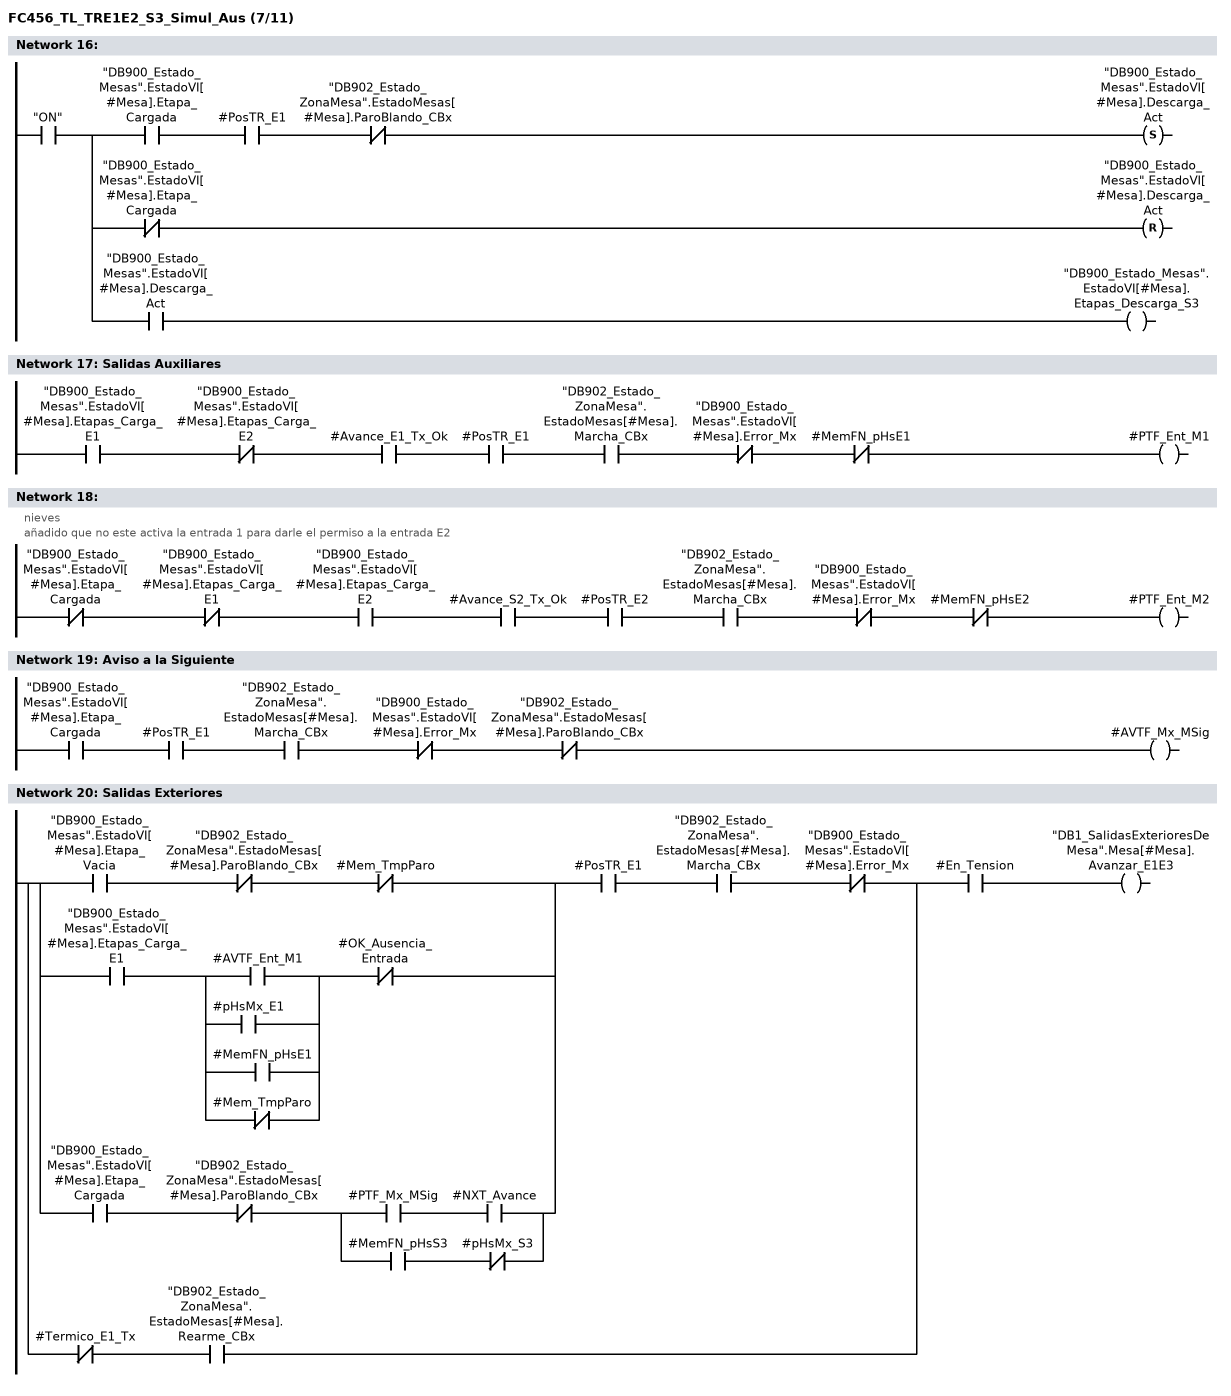
   RUNG wire#powerrail
      Contact( "ON" )
      wire#w1
      Contact( "DB900_Estado_Mesas".EstadoVI[#Mesa].Etapa_Cargada )
      Contact( #PosTR_E1 )
      I_Contact( "DB902_Estado_ZonaMesa".EstadoMesas[#Mesa].ParoBlando_CBx )
      S_Coil( "DB900_Estado_Mesas".EstadoVI[#Mesa].Descarga_Act )
   END_RUNG
   RUNG wire#w1
      I_Contact( "DB900_Estado_Mesas".EstadoVI[#Mesa].Etapa_Cargada )
      R_Coil( "DB900_Estado_Mesas".EstadoVI[#Mesa].Descarga_Act )
   END_RUNG
   RUNG wire#w1
      Contact( "DB900_Estado_Mesas".EstadoVI[#Mesa].Descarga_Act )
      Coil( "DB900_Estado_Mesas".EstadoVI[#Mesa].Etapas_Descarga_S3 )
   END_RUNG
   // the same network as SCL:
   IF "ON" AND "DB900_Estado_Mesas".EstadoVI[#Mesa].Etapa_Cargada AND #PosTR_E1 AND NOT "DB902_Estado_ZonaMesa".EstadoMesas[#Mesa].ParoBlando_CBx THEN
       "DB900_Estado_Mesas".EstadoVI[#Mesa].Descarga_Act := TRUE;
   END_IF;
   IF "ON" AND NOT "DB900_Estado_Mesas".EstadoVI[#Mesa].Etapa_Cargada THEN
       "DB900_Estado_Mesas".EstadoVI[#Mesa].Descarga_Act := FALSE;
   END_IF;
   "DB900_Estado_Mesas".EstadoVI[#Mesa].Etapas_Descarga_S3 := "ON" AND "DB900_Estado_Mesas".EstadoVI[#Mesa].Descarga_Act;
END_REGION

REGION Network 17: Salidas Auxiliares
   RUNG wire#powerrail
      Contact( "DB900_Estado_Mesas".EstadoVI[#Mesa].Etapas_Carga_E1 )
      I_Contact( "DB900_Estado_Mesas".EstadoVI[#Mesa].Etapas_Carga_E2 )
      Contact( #Avance_E1_Tx_Ok )
      Contact( #PosTR_E1 )
      Contact( "DB902_Estado_ZonaMesa".EstadoMesas[#Mesa].Marcha_CBx )
      I_Contact( "DB900_Estado_Mesas".EstadoVI[#Mesa].Error_Mx )
      I_Contact( #MemFN_pHsE1 )
      Coil( #PTF_Ent_M1 )
   END_RUNG
   // the same network as SCL:
   #PTF_Ent_M1 := "DB900_Estado_Mesas".EstadoVI[#Mesa].Etapas_Carga_E1 AND NOT "DB900_Estado_Mesas".EstadoVI[#Mesa].Etapas_Carga_E2 AND #Avance_E1_Tx_Ok AND #PosTR_E1 AND "DB902_Estado_ZonaMesa".EstadoMesas[#Mesa].Marcha_CBx AND NOT "DB900_Estado_Mesas".EstadoVI[#Mesa].Error_Mx AND NOT #MemFN_pHsE1;
END_REGION

REGION Network 18
   // nieves
   // añadido que no este activa la entrada 1 para darle el permiso a la entrada E2
   RUNG wire#powerrail
      I_Contact( "DB900_Estado_Mesas".EstadoVI[#Mesa].Etapa_Cargada )
      I_Contact( "DB900_Estado_Mesas".EstadoVI[#Mesa].Etapas_Carga_E1 )
      Contact( "DB900_Estado_Mesas".EstadoVI[#Mesa].Etapas_Carga_E2 )
      Contact( #Avance_S2_Tx_Ok )
      Contact( #PosTR_E2 )
      Contact( "DB902_Estado_ZonaMesa".EstadoMesas[#Mesa].Marcha_CBx )
      I_Contact( "DB900_Estado_Mesas".EstadoVI[#Mesa].Error_Mx )
      I_Contact( #MemFN_pHsE2 )
      Coil( #PTF_Ent_M2 )
   END_RUNG
   // the same network as SCL:
   #PTF_Ent_M2 := NOT "DB900_Estado_Mesas".EstadoVI[#Mesa].Etapa_Cargada AND NOT "DB900_Estado_Mesas".EstadoVI[#Mesa].Etapas_Carga_E1 AND "DB900_Estado_Mesas".EstadoVI[#Mesa].Etapas_Carga_E2 AND #Avance_S2_Tx_Ok AND #PosTR_E2 AND "DB902_Estado_ZonaMesa".EstadoMesas[#Mesa].Marcha_CBx AND NOT "DB900_Estado_Mesas".EstadoVI[#Mesa].Error_Mx AND NOT #MemFN_pHsE2;
END_REGION

REGION Network 19: Aviso a la Siguiente
   RUNG wire#powerrail
      Contact( "DB900_Estado_Mesas".EstadoVI[#Mesa].Etapa_Cargada )
      Contact( #PosTR_E1 )
      Contact( "DB902_Estado_ZonaMesa".EstadoMesas[#Mesa].Marcha_CBx )
      I_Contact( "DB900_Estado_Mesas".EstadoVI[#Mesa].Error_Mx )
      I_Contact( "DB902_Estado_ZonaMesa".EstadoMesas[#Mesa].ParoBlando_CBx )
      Coil( #AVTF_Mx_MSig )
   END_RUNG
   // the same network as SCL:
   #AVTF_Mx_MSig := "DB900_Estado_Mesas".EstadoVI[#Mesa].Etapa_Cargada AND #PosTR_E1 AND "DB902_Estado_ZonaMesa".EstadoMesas[#Mesa].Marcha_CBx AND NOT "DB900_Estado_Mesas".EstadoVI[#Mesa].Error_Mx AND NOT "DB902_Estado_ZonaMesa".EstadoMesas[#Mesa].ParoBlando_CBx;
END_REGION

REGION Network 20: Salidas Exteriores
   RUNG wire#powerrail
      Contact( "DB900_Estado_Mesas".EstadoVI[#Mesa].Etapa_Vacia )
      I_Contact( "DB902_Estado_ZonaMesa".EstadoMesas[#Mesa].ParoBlando_CBx )
      I_Contact( #Mem_TmpParo )
      wire#w1
      Contact( #PosTR_E1 )
      Contact( "DB902_Estado_ZonaMesa".EstadoMesas[#Mesa].Marcha_CBx )
      I_Contact( "DB900_Estado_Mesas".EstadoVI[#Mesa].Error_Mx )
      wire#w5
      Contact( #En_Tension )
      Coil( "DB1_SalidasExterioresDeMesa".Mesa[#Mesa].Avanzar_E1E3 )
   END_RUNG
   RUNG wire#powerrail
      Contact( "DB900_Estado_Mesas".EstadoVI[#Mesa].Etapas_Carga_E1 )
      wire#w2
      Contact( #AVTF_Ent_M1 )
      wire#w3
      I_Contact( #OK_Ausencia_Entrada )
   END_RUNG wire#w1
   RUNG wire#w2
      Contact( #pHsMx_E1 )
   END_RUNG wire#w3
   RUNG wire#w2
      Contact( #MemFN_pHsE1 )
   END_RUNG wire#w3
   RUNG wire#w2
      I_Contact( #Mem_TmpParo )
   END_RUNG wire#w3
   RUNG wire#powerrail
      Contact( "DB900_Estado_Mesas".EstadoVI[#Mesa].Etapa_Cargada )
      I_Contact( "DB902_Estado_ZonaMesa".EstadoMesas[#Mesa].ParoBlando_CBx )
      wire#w4
      Contact( #PTF_Mx_MSig )
      Contact( #NXT_Avance )
   END_RUNG wire#w1
   RUNG wire#w4
      Contact( #MemFN_pHsS3 )
      I_Contact( #pHsMx_S3 )
   END_RUNG wire#w1
   RUNG wire#powerrail
      I_Contact( #Termico_E1_Tx )
      Contact( "DB902_Estado_ZonaMesa".EstadoMesas[#Mesa].Rearme_CBx )
   END_RUNG wire#w5
   // the same network as SCL:
   "DB1_SalidasExterioresDeMesa".Mesa[#Mesa].Avanzar_E1E3 := (((("DB900_Estado_Mesas".EstadoVI[#Mesa].Etapa_Vacia AND NOT "DB902_Estado_ZonaMesa".EstadoMesas[#Mesa].ParoBlando_CBx AND NOT #Mem_TmpParo) OR ("DB900_Estado_Mesas".EstadoVI[#Mesa].Etapas_Carga_E1 AND (#AVTF_Ent_M1 OR #pHsMx_E1 OR #MemFN_pHsE1 OR NOT #Mem_TmpParo) AND NOT #OK_Ausencia_Entrada) OR ("DB900_Estado_Mesas".EstadoVI[#Mesa].Etapa_Cargada AND NOT "DB902_Estado_ZonaMesa".EstadoMesas[#Mesa].ParoBlando_CBx AND ((#PTF_Mx_MSig AND #NXT_Avance) OR (#MemFN_pHsS3 AND NOT #pHsMx_S3)))) AND #PosTR_E1 AND "DB902_Estado_ZonaMesa".EstadoMesas[#Mesa].Marcha_CBx AND NOT "DB900_Estado_Mesas".EstadoVI[#Mesa].Error_Mx) OR (NOT #Termico_E1_Tx AND "DB902_Estado_ZonaMesa".EstadoMesas[#Mesa].Rearme_CBx)) AND #En_Tension;
END_REGION

REGION Network 21
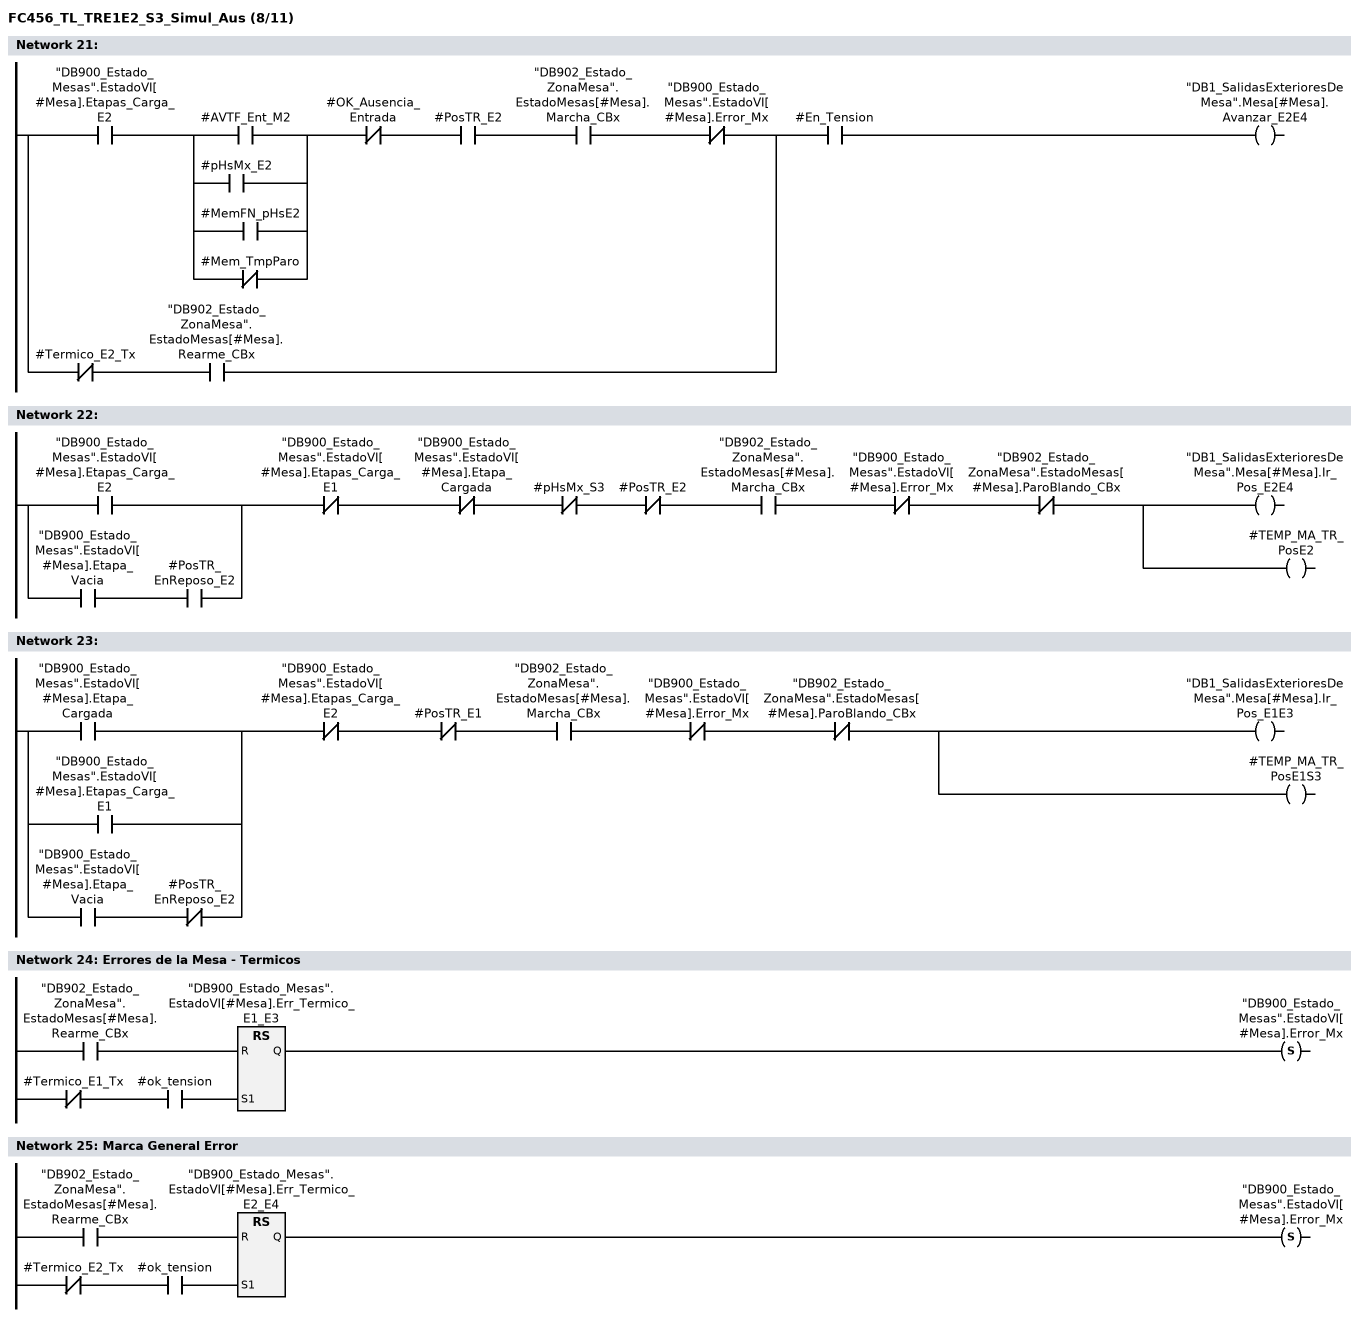
   RUNG wire#powerrail
      Contact( "DB900_Estado_Mesas".EstadoVI[#Mesa].Etapas_Carga_E2 )
      wire#w1
      Contact( #AVTF_Ent_M2 )
      wire#w2
      I_Contact( #OK_Ausencia_Entrada )
      Contact( #PosTR_E2 )
      Contact( "DB902_Estado_ZonaMesa".EstadoMesas[#Mesa].Marcha_CBx )
      I_Contact( "DB900_Estado_Mesas".EstadoVI[#Mesa].Error_Mx )
      wire#w3
      Contact( #En_Tension )
      Coil( "DB1_SalidasExterioresDeMesa".Mesa[#Mesa].Avanzar_E2E4 )
   END_RUNG
   RUNG wire#w1
      Contact( #pHsMx_E2 )
   END_RUNG wire#w2
   RUNG wire#w1
      Contact( #MemFN_pHsE2 )
   END_RUNG wire#w2
   RUNG wire#w1
      I_Contact( #Mem_TmpParo )
   END_RUNG wire#w2
   RUNG wire#powerrail
      I_Contact( #Termico_E2_Tx )
      Contact( "DB902_Estado_ZonaMesa".EstadoMesas[#Mesa].Rearme_CBx )
   END_RUNG wire#w3
   // the same network as SCL:
   "DB1_SalidasExterioresDeMesa".Mesa[#Mesa].Avanzar_E2E4 := (("DB900_Estado_Mesas".EstadoVI[#Mesa].Etapas_Carga_E2 AND (#AVTF_Ent_M2 OR #pHsMx_E2 OR #MemFN_pHsE2 OR NOT #Mem_TmpParo) AND NOT #OK_Ausencia_Entrada AND #PosTR_E2 AND "DB902_Estado_ZonaMesa".EstadoMesas[#Mesa].Marcha_CBx AND NOT "DB900_Estado_Mesas".EstadoVI[#Mesa].Error_Mx) OR (NOT #Termico_E2_Tx AND "DB902_Estado_ZonaMesa".EstadoMesas[#Mesa].Rearme_CBx)) AND #En_Tension;
END_REGION

REGION Network 22
   RUNG wire#powerrail
      Contact( "DB900_Estado_Mesas".EstadoVI[#Mesa].Etapas_Carga_E2 )
      wire#w1
      I_Contact( "DB900_Estado_Mesas".EstadoVI[#Mesa].Etapas_Carga_E1 )
      I_Contact( "DB900_Estado_Mesas".EstadoVI[#Mesa].Etapa_Cargada )
      I_Contact( #pHsMx_S3 )
      I_Contact( #PosTR_E2 )
      Contact( "DB902_Estado_ZonaMesa".EstadoMesas[#Mesa].Marcha_CBx )
      I_Contact( "DB900_Estado_Mesas".EstadoVI[#Mesa].Error_Mx )
      I_Contact( "DB902_Estado_ZonaMesa".EstadoMesas[#Mesa].ParoBlando_CBx )
      wire#w2
      Coil( "DB1_SalidasExterioresDeMesa".Mesa[#Mesa].Ir_Pos_E2E4 )
   END_RUNG
   RUNG wire#powerrail
      Contact( "DB900_Estado_Mesas".EstadoVI[#Mesa].Etapa_Vacia )
      Contact( #PosTR_EnReposo_E2 )
   END_RUNG wire#w1
   RUNG wire#w2
      Coil( #TEMP_MA_TR_PosE2 )
   END_RUNG
   // the same network as SCL:
   #_w1 := ("DB900_Estado_Mesas".EstadoVI[#Mesa].Etapas_Carga_E2 OR ("DB900_Estado_Mesas".EstadoVI[#Mesa].Etapa_Vacia AND #PosTR_EnReposo_E2)) AND NOT "DB900_Estado_Mesas".EstadoVI[#Mesa].Etapas_Carga_E1 AND NOT "DB900_Estado_Mesas".EstadoVI[#Mesa].Etapa_Cargada AND NOT #pHsMx_S3 AND NOT #PosTR_E2 AND "DB902_Estado_ZonaMesa".EstadoMesas[#Mesa].Marcha_CBx AND NOT "DB900_Estado_Mesas".EstadoVI[#Mesa].Error_Mx AND NOT "DB902_Estado_ZonaMesa".EstadoMesas[#Mesa].ParoBlando_CBx;
   "DB1_SalidasExterioresDeMesa".Mesa[#Mesa].Ir_Pos_E2E4 := ("DB900_Estado_Mesas".EstadoVI[#Mesa].Etapas_Carga_E2 OR ("DB900_Estado_Mesas".EstadoVI[#Mesa].Etapa_Vacia AND #PosTR_EnReposo_E2)) AND NOT "DB900_Estado_Mesas".EstadoVI[#Mesa].Etapas_Carga_E1 AND NOT "DB900_Estado_Mesas".EstadoVI[#Mesa].Etapa_Cargada AND NOT #pHsMx_S3 AND NOT #PosTR_E2 AND "DB902_Estado_ZonaMesa".EstadoMesas[#Mesa].Marcha_CBx AND NOT "DB900_Estado_Mesas".EstadoVI[#Mesa].Error_Mx AND NOT "DB902_Estado_ZonaMesa".EstadoMesas[#Mesa].ParoBlando_CBx;
   #TEMP_MA_TR_PosE2 := #_w1;
END_REGION

REGION Network 23
   RUNG wire#powerrail
      Contact( "DB900_Estado_Mesas".EstadoVI[#Mesa].Etapa_Cargada )
      wire#w1
      I_Contact( "DB900_Estado_Mesas".EstadoVI[#Mesa].Etapas_Carga_E2 )
      I_Contact( #PosTR_E1 )
      Contact( "DB902_Estado_ZonaMesa".EstadoMesas[#Mesa].Marcha_CBx )
      I_Contact( "DB900_Estado_Mesas".EstadoVI[#Mesa].Error_Mx )
      I_Contact( "DB902_Estado_ZonaMesa".EstadoMesas[#Mesa].ParoBlando_CBx )
      wire#w2
      Coil( "DB1_SalidasExterioresDeMesa".Mesa[#Mesa].Ir_Pos_E1E3 )
   END_RUNG
   RUNG wire#powerrail
      Contact( "DB900_Estado_Mesas".EstadoVI[#Mesa].Etapas_Carga_E1 )
   END_RUNG wire#w1
   RUNG wire#powerrail
      Contact( "DB900_Estado_Mesas".EstadoVI[#Mesa].Etapa_Vacia )
      I_Contact( #PosTR_EnReposo_E2 )
   END_RUNG wire#w1
   RUNG wire#w2
      Coil( #TEMP_MA_TR_PosE1S3 )
   END_RUNG
   // the same network as SCL:
   #_w1 := ("DB900_Estado_Mesas".EstadoVI[#Mesa].Etapa_Cargada OR "DB900_Estado_Mesas".EstadoVI[#Mesa].Etapas_Carga_E1 OR ("DB900_Estado_Mesas".EstadoVI[#Mesa].Etapa_Vacia AND NOT #PosTR_EnReposo_E2)) AND NOT "DB900_Estado_Mesas".EstadoVI[#Mesa].Etapas_Carga_E2 AND NOT #PosTR_E1 AND "DB902_Estado_ZonaMesa".EstadoMesas[#Mesa].Marcha_CBx AND NOT "DB900_Estado_Mesas".EstadoVI[#Mesa].Error_Mx AND NOT "DB902_Estado_ZonaMesa".EstadoMesas[#Mesa].ParoBlando_CBx;
   "DB1_SalidasExterioresDeMesa".Mesa[#Mesa].Ir_Pos_E1E3 := ("DB900_Estado_Mesas".EstadoVI[#Mesa].Etapa_Cargada OR "DB900_Estado_Mesas".EstadoVI[#Mesa].Etapas_Carga_E1 OR ("DB900_Estado_Mesas".EstadoVI[#Mesa].Etapa_Vacia AND NOT #PosTR_EnReposo_E2)) AND NOT "DB900_Estado_Mesas".EstadoVI[#Mesa].Etapas_Carga_E2 AND NOT #PosTR_E1 AND "DB902_Estado_ZonaMesa".EstadoMesas[#Mesa].Marcha_CBx AND NOT "DB900_Estado_Mesas".EstadoVI[#Mesa].Error_Mx AND NOT "DB902_Estado_ZonaMesa".EstadoMesas[#Mesa].ParoBlando_CBx;
   #TEMP_MA_TR_PosE1S3 := #_w1;
END_REGION

REGION Network 24: Errores de la Mesa - Termicos
   RUNG wire#powerrail
      Contact( "DB902_Estado_ZonaMesa".EstadoMesas[#Mesa].Rearme_CBx )
      S_RS(operand := "DB900_Estado_Mesas".EstadoVI[#Mesa].Err_Termico_E1_E3, s1 := wire#w1)
      S_Coil( "DB900_Estado_Mesas".EstadoVI[#Mesa].Error_Mx )
   END_RUNG
   RUNG wire#powerrail
      I_Contact( #Termico_E1_Tx )
      Contact( #ok_tension )
   END_RUNG wire#w1
   // the same network as SCL:
   IF "DB902_Estado_ZonaMesa".EstadoMesas[#Mesa].Rearme_CBx THEN
       "DB900_Estado_Mesas".EstadoVI[#Mesa].Err_Termico_E1_E3 := FALSE;   // RS flip-flop
   END_IF;
   IF NOT #Termico_E1_Tx AND #ok_tension THEN
       "DB900_Estado_Mesas".EstadoVI[#Mesa].Err_Termico_E1_E3 := TRUE;
   END_IF;
   IF "DB900_Estado_Mesas".EstadoVI[#Mesa].Err_Termico_E1_E3 THEN
       "DB900_Estado_Mesas".EstadoVI[#Mesa].Error_Mx := TRUE;
   END_IF;
END_REGION

REGION Network 25: Marca General Error
   RUNG wire#powerrail
      Contact( "DB902_Estado_ZonaMesa".EstadoMesas[#Mesa].Rearme_CBx )
      S_RS(operand := "DB900_Estado_Mesas".EstadoVI[#Mesa].Err_Termico_E2_E4, s1 := wire#w1)
      S_Coil( "DB900_Estado_Mesas".EstadoVI[#Mesa].Error_Mx )
   END_RUNG
   RUNG wire#powerrail
      I_Contact( #Termico_E2_Tx )
      Contact( #ok_tension )
   END_RUNG wire#w1
   // the same network as SCL:
   IF "DB902_Estado_ZonaMesa".EstadoMesas[#Mesa].Rearme_CBx THEN
       "DB900_Estado_Mesas".EstadoVI[#Mesa].Err_Termico_E2_E4 := FALSE;   // RS flip-flop
   END_IF;
   IF NOT #Termico_E2_Tx AND #ok_tension THEN
       "DB900_Estado_Mesas".EstadoVI[#Mesa].Err_Termico_E2_E4 := TRUE;
   END_IF;
   IF "DB900_Estado_Mesas".EstadoVI[#Mesa].Err_Termico_E2_E4 THEN
       "DB900_Estado_Mesas".EstadoVI[#Mesa].Error_Mx := TRUE;
   END_IF;
END_REGION

REGION Network 26: Errores de la Mesa - TimeOuts de Avances
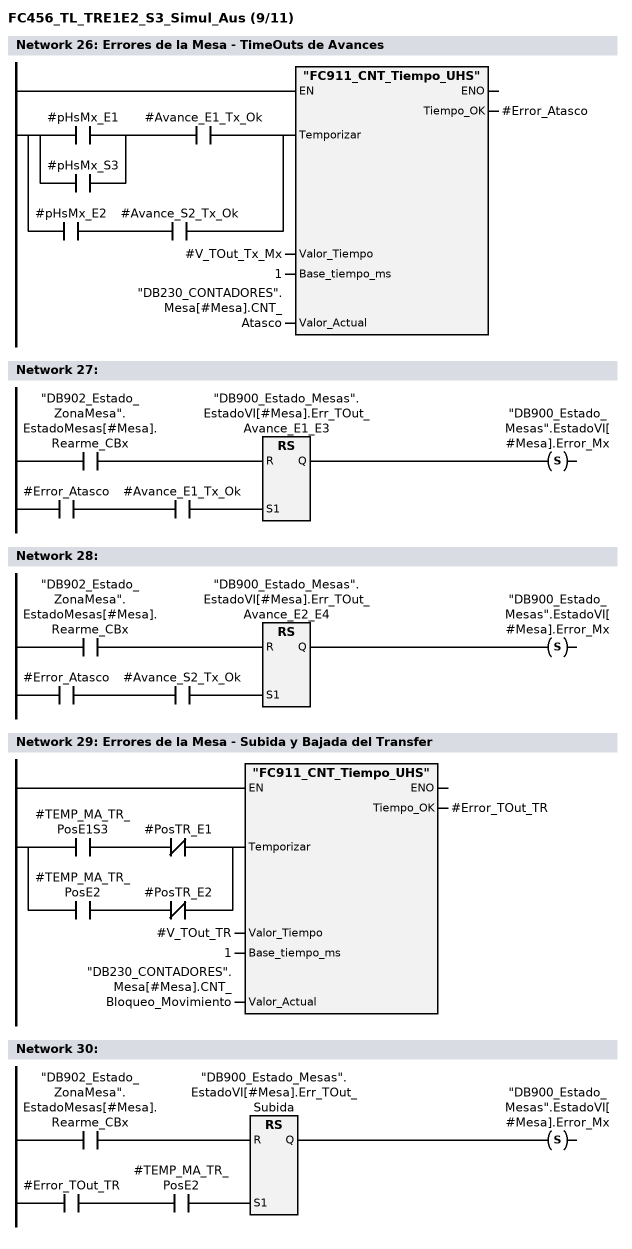
   RUNG wire#powerrail
      "FC911_CNT_Tiempo_UHS"(Temporizar := wire#w2, Valor_Tiempo := #V_TOut_Tx_Mx, Base_tiempo_ms := 1, Valor_Actual := "DB230_CONTADORES".Mesa[#Mesa].CNT_Atasco, Tiempo_OK => #Error_Atasco)
   END_RUNG
   RUNG wire#powerrail
      Contact( #pHsMx_E1 )
      wire#w1
      Contact( #Avance_E1_Tx_Ok )
   END_RUNG wire#w2
   RUNG wire#powerrail
      Contact( #pHsMx_S3 )
   END_RUNG wire#w1
   RUNG wire#powerrail
      Contact( #pHsMx_E2 )
      Contact( #Avance_S2_Tx_Ok )
   END_RUNG wire#w2
   // the same network as SCL:
   "FC911_CNT_Tiempo_UHS"(Temporizar := ((#pHsMx_E1 OR #pHsMx_S3) AND #Avance_E1_Tx_Ok) OR (#pHsMx_E2 AND #Avance_S2_Tx_Ok),
                          Valor_Tiempo := #V_TOut_Tx_Mx,
                          Base_tiempo_ms := 1,
                          Valor_Actual := "DB230_CONTADORES".Mesa[#Mesa].CNT_Atasco,
                          Tiempo_OK => #Error_Atasco);
END_REGION

REGION Network 27
   RUNG wire#powerrail
      Contact( "DB902_Estado_ZonaMesa".EstadoMesas[#Mesa].Rearme_CBx )
      S_RS(operand := "DB900_Estado_Mesas".EstadoVI[#Mesa].Err_TOut_Avance_E1_E3, s1 := wire#w1)
      S_Coil( "DB900_Estado_Mesas".EstadoVI[#Mesa].Error_Mx )
   END_RUNG
   RUNG wire#powerrail
      Contact( #Error_Atasco )
      Contact( #Avance_E1_Tx_Ok )
   END_RUNG wire#w1
   // the same network as SCL:
   IF "DB902_Estado_ZonaMesa".EstadoMesas[#Mesa].Rearme_CBx THEN
       "DB900_Estado_Mesas".EstadoVI[#Mesa].Err_TOut_Avance_E1_E3 := FALSE;   // RS flip-flop
   END_IF;
   IF #Error_Atasco AND #Avance_E1_Tx_Ok THEN
       "DB900_Estado_Mesas".EstadoVI[#Mesa].Err_TOut_Avance_E1_E3 := TRUE;
   END_IF;
   IF "DB900_Estado_Mesas".EstadoVI[#Mesa].Err_TOut_Avance_E1_E3 THEN
       "DB900_Estado_Mesas".EstadoVI[#Mesa].Error_Mx := TRUE;
   END_IF;
END_REGION

REGION Network 28
   RUNG wire#powerrail
      Contact( "DB902_Estado_ZonaMesa".EstadoMesas[#Mesa].Rearme_CBx )
      S_RS(operand := "DB900_Estado_Mesas".EstadoVI[#Mesa].Err_TOut_Avance_E2_E4, s1 := wire#w1)
      S_Coil( "DB900_Estado_Mesas".EstadoVI[#Mesa].Error_Mx )
   END_RUNG
   RUNG wire#powerrail
      Contact( #Error_Atasco )
      Contact( #Avance_S2_Tx_Ok )
   END_RUNG wire#w1
   // the same network as SCL:
   IF "DB902_Estado_ZonaMesa".EstadoMesas[#Mesa].Rearme_CBx THEN
       "DB900_Estado_Mesas".EstadoVI[#Mesa].Err_TOut_Avance_E2_E4 := FALSE;   // RS flip-flop
   END_IF;
   IF #Error_Atasco AND #Avance_S2_Tx_Ok THEN
       "DB900_Estado_Mesas".EstadoVI[#Mesa].Err_TOut_Avance_E2_E4 := TRUE;
   END_IF;
   IF "DB900_Estado_Mesas".EstadoVI[#Mesa].Err_TOut_Avance_E2_E4 THEN
       "DB900_Estado_Mesas".EstadoVI[#Mesa].Error_Mx := TRUE;
   END_IF;
END_REGION

REGION Network 29: Errores de la Mesa - Subida y Bajada del Transfer
   RUNG wire#powerrail
      "FC911_CNT_Tiempo_UHS"(Temporizar := wire#w1, Valor_Tiempo := #V_TOut_TR, Base_tiempo_ms := 1, Valor_Actual := "DB230_CONTADORES".Mesa[#Mesa].CNT_Bloqueo_Movimiento, Tiempo_OK => #Error_TOut_TR)
   END_RUNG
   RUNG wire#powerrail
      Contact( #TEMP_MA_TR_PosE1S3 )
      I_Contact( #PosTR_E1 )
   END_RUNG wire#w1
   RUNG wire#powerrail
      Contact( #TEMP_MA_TR_PosE2 )
      I_Contact( #PosTR_E2 )
   END_RUNG wire#w1
   // the same network as SCL:
   "FC911_CNT_Tiempo_UHS"(Temporizar := (#TEMP_MA_TR_PosE1S3 AND NOT #PosTR_E1) OR (#TEMP_MA_TR_PosE2 AND NOT #PosTR_E2),
                          Valor_Tiempo := #V_TOut_TR,
                          Base_tiempo_ms := 1,
                          Valor_Actual := "DB230_CONTADORES".Mesa[#Mesa].CNT_Bloqueo_Movimiento,
                          Tiempo_OK => #Error_TOut_TR);
END_REGION

REGION Network 30
   RUNG wire#powerrail
      Contact( "DB902_Estado_ZonaMesa".EstadoMesas[#Mesa].Rearme_CBx )
      S_RS(operand := "DB900_Estado_Mesas".EstadoVI[#Mesa].Err_TOut_Subida, s1 := wire#w1)
      S_Coil( "DB900_Estado_Mesas".EstadoVI[#Mesa].Error_Mx )
   END_RUNG
   RUNG wire#powerrail
      Contact( #Error_TOut_TR )
      Contact( #TEMP_MA_TR_PosE2 )
   END_RUNG wire#w1
   // the same network as SCL:
   IF "DB902_Estado_ZonaMesa".EstadoMesas[#Mesa].Rearme_CBx THEN
       "DB900_Estado_Mesas".EstadoVI[#Mesa].Err_TOut_Subida := FALSE;   // RS flip-flop
   END_IF;
   IF #Error_TOut_TR AND #TEMP_MA_TR_PosE2 THEN
       "DB900_Estado_Mesas".EstadoVI[#Mesa].Err_TOut_Subida := TRUE;
   END_IF;
   IF "DB900_Estado_Mesas".EstadoVI[#Mesa].Err_TOut_Subida THEN
       "DB900_Estado_Mesas".EstadoVI[#Mesa].Error_Mx := TRUE;
   END_IF;
END_REGION

REGION Network 31: Marca General Error
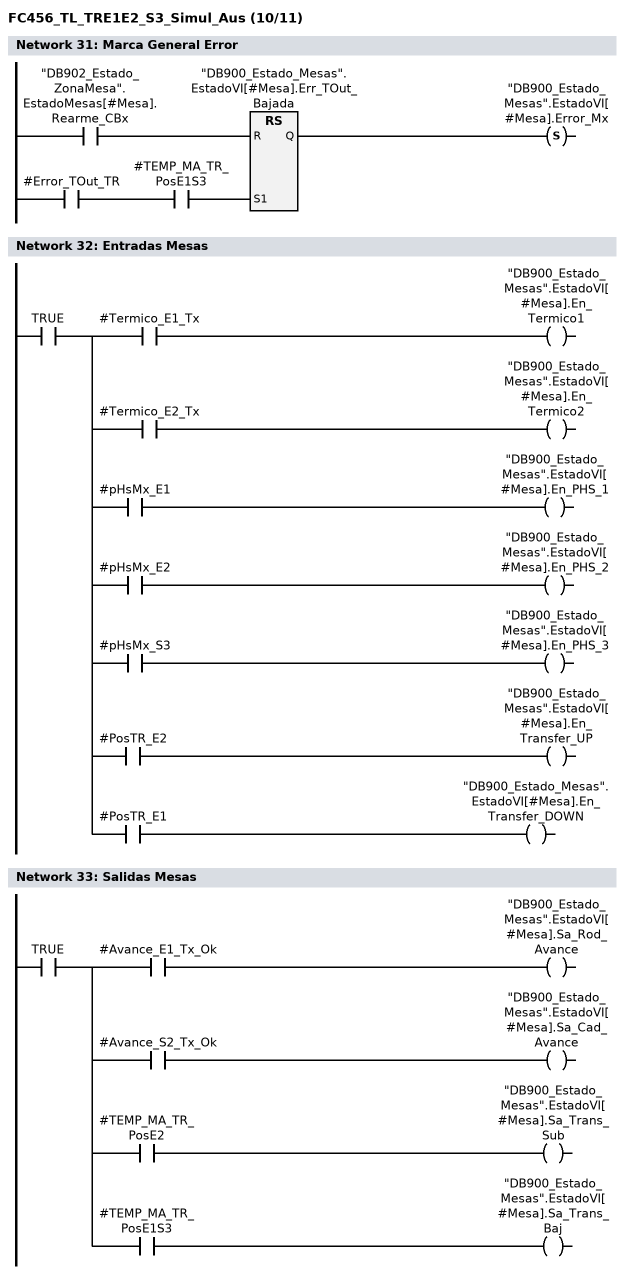
   RUNG wire#powerrail
      Contact( "DB902_Estado_ZonaMesa".EstadoMesas[#Mesa].Rearme_CBx )
      S_RS(operand := "DB900_Estado_Mesas".EstadoVI[#Mesa].Err_TOut_Bajada, s1 := wire#w1)
      S_Coil( "DB900_Estado_Mesas".EstadoVI[#Mesa].Error_Mx )
   END_RUNG
   RUNG wire#powerrail
      Contact( #Error_TOut_TR )
      Contact( #TEMP_MA_TR_PosE1S3 )
   END_RUNG wire#w1
   // the same network as SCL:
   IF "DB902_Estado_ZonaMesa".EstadoMesas[#Mesa].Rearme_CBx THEN
       "DB900_Estado_Mesas".EstadoVI[#Mesa].Err_TOut_Bajada := FALSE;   // RS flip-flop
   END_IF;
   IF #Error_TOut_TR AND #TEMP_MA_TR_PosE1S3 THEN
       "DB900_Estado_Mesas".EstadoVI[#Mesa].Err_TOut_Bajada := TRUE;
   END_IF;
   IF "DB900_Estado_Mesas".EstadoVI[#Mesa].Err_TOut_Bajada THEN
       "DB900_Estado_Mesas".EstadoVI[#Mesa].Error_Mx := TRUE;
   END_IF;
END_REGION

REGION Network 32: Entradas Mesas
   RUNG wire#powerrail
      Contact( TRUE )
      wire#w1
      Contact( #Termico_E1_Tx )
      Coil( "DB900_Estado_Mesas".EstadoVI[#Mesa].En_Termico1 )
   END_RUNG
   RUNG wire#w1
      Contact( #Termico_E2_Tx )
      Coil( "DB900_Estado_Mesas".EstadoVI[#Mesa].En_Termico2 )
   END_RUNG
   RUNG wire#w1
      Contact( #pHsMx_E1 )
      Coil( "DB900_Estado_Mesas".EstadoVI[#Mesa].En_PHS_1 )
   END_RUNG
   RUNG wire#w1
      Contact( #pHsMx_E2 )
      Coil( "DB900_Estado_Mesas".EstadoVI[#Mesa].En_PHS_2 )
   END_RUNG
   RUNG wire#w1
      Contact( #pHsMx_S3 )
      Coil( "DB900_Estado_Mesas".EstadoVI[#Mesa].En_PHS_3 )
   END_RUNG
   RUNG wire#w1
      Contact( #PosTR_E2 )
      Coil( "DB900_Estado_Mesas".EstadoVI[#Mesa].En_Transfer_UP )
   END_RUNG
   RUNG wire#w1
      Contact( #PosTR_E1 )
      Coil( "DB900_Estado_Mesas".EstadoVI[#Mesa].En_Transfer_DOWN )
   END_RUNG
   // the same network as SCL:
   "DB900_Estado_Mesas".EstadoVI[#Mesa].En_Termico1 := TRUE AND #Termico_E1_Tx;
   "DB900_Estado_Mesas".EstadoVI[#Mesa].En_Termico2 := TRUE AND #Termico_E2_Tx;
   "DB900_Estado_Mesas".EstadoVI[#Mesa].En_PHS_1 := TRUE AND #pHsMx_E1;
   "DB900_Estado_Mesas".EstadoVI[#Mesa].En_PHS_2 := TRUE AND #pHsMx_E2;
   "DB900_Estado_Mesas".EstadoVI[#Mesa].En_PHS_3 := TRUE AND #pHsMx_S3;
   "DB900_Estado_Mesas".EstadoVI[#Mesa].En_Transfer_UP := TRUE AND #PosTR_E2;
   "DB900_Estado_Mesas".EstadoVI[#Mesa].En_Transfer_DOWN := TRUE AND #PosTR_E1;
END_REGION

REGION Network 33: Salidas Mesas
   RUNG wire#powerrail
      Contact( TRUE )
      wire#w1
      Contact( #Avance_E1_Tx_Ok )
      Coil( "DB900_Estado_Mesas".EstadoVI[#Mesa].Sa_Rod_Avance )
   END_RUNG
   RUNG wire#w1
      Contact( #Avance_S2_Tx_Ok )
      Coil( "DB900_Estado_Mesas".EstadoVI[#Mesa].Sa_Cad_Avance )
   END_RUNG
   RUNG wire#w1
      Contact( #TEMP_MA_TR_PosE2 )
      Coil( "DB900_Estado_Mesas".EstadoVI[#Mesa].Sa_Trans_Sub )
   END_RUNG
   RUNG wire#w1
      Contact( #TEMP_MA_TR_PosE1S3 )
      Coil( "DB900_Estado_Mesas".EstadoVI[#Mesa].Sa_Trans_Baj )
   END_RUNG
   // the same network as SCL:
   "DB900_Estado_Mesas".EstadoVI[#Mesa].Sa_Rod_Avance := TRUE AND #Avance_E1_Tx_Ok;
   "DB900_Estado_Mesas".EstadoVI[#Mesa].Sa_Cad_Avance := TRUE AND #Avance_S2_Tx_Ok;
   "DB900_Estado_Mesas".EstadoVI[#Mesa].Sa_Trans_Sub := TRUE AND #TEMP_MA_TR_PosE2;
   "DB900_Estado_Mesas".EstadoVI[#Mesa].Sa_Trans_Baj := TRUE AND #TEMP_MA_TR_PosE1S3;
END_REGION

REGION Network 34: Fin de Vehiculo
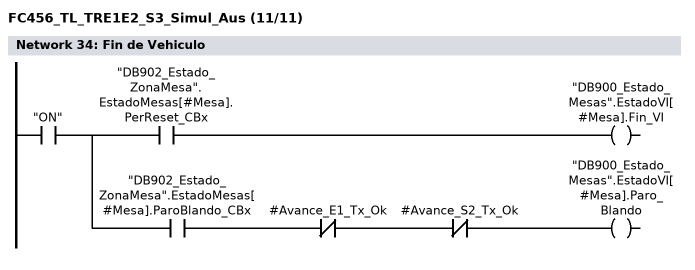
   RUNG wire#powerrail
      Contact( "ON" )
      wire#w1
      Contact( "DB902_Estado_ZonaMesa".EstadoMesas[#Mesa].PerReset_CBx )
      Coil( "DB900_Estado_Mesas".EstadoVI[#Mesa].Fin_VI )
   END_RUNG
   RUNG wire#w1
      Contact( "DB902_Estado_ZonaMesa".EstadoMesas[#Mesa].ParoBlando_CBx )
      I_Contact( #Avance_E1_Tx_Ok )
      I_Contact( #Avance_S2_Tx_Ok )
      Coil( "DB900_Estado_Mesas".EstadoVI[#Mesa].Paro_Blando )
   END_RUNG
   // the same network as SCL:
   "DB900_Estado_Mesas".EstadoVI[#Mesa].Fin_VI := "ON" AND "DB902_Estado_ZonaMesa".EstadoMesas[#Mesa].PerReset_CBx;
   "DB900_Estado_Mesas".EstadoVI[#Mesa].Paro_Blando := "ON" AND "DB902_Estado_ZonaMesa".EstadoMesas[#Mesa].ParoBlando_CBx AND NOT #Avance_E1_Tx_Ok AND NOT #Avance_S2_Tx_Ok;
END_REGION
END_FUNCTION

FUNCTION "FC457_TL_TR_E1E3_S2_Aus" : Void   // FC457, LAD
{ S7_Optimized_Access := 'FALSE' }
AUTHOR : TLigero
NAME : 20180125
VERSION : 3.2
// FECHA:    27/07/2014  AUTOR: G.Martin
// INSTALACION: Magyar Posta
// //////////////////////////////////
// // Registro Incidencias   ////////
// //////////////////////////////////
// FECHA:21/10/14   AUTOR MODIFICACION: N.Rodriguez
// DESCRIPCION: 
// Adaptación de la función al estandar actual
// ULTIMA MODIFICACION: iñaki Arrondo por problemas detectados en la instalacion (ALKAR)
// stored: AutoNumber false, SetENOAutomatically false
   VAR_INPUT
      Mesa : UInt;
      En_Tension : Bool;
      pHsMx_E1 : Bool;
      pHsMx_E3 : Bool;
      pHsMx_S2 : Bool;
      TP_E1_UP : Bool;
      TP_E1_Dw : Bool;
      TP_E3_UP : Bool;
      TP_E3_Dw : Bool;
      Termico_E1_Tx : Bool;
      Termico_S2_Tx : Bool;
      Avance_E1_Tx_Ok : Bool;
      Avance_E3_Tx_Ok : Bool;   // será el retroceso de E1
      Avance_S2_Tx_Ok : Bool;
      PosTR_E1 : Bool;
      PosTR_S2 : Bool;
      AVTF_Ent_M1 : Bool;
      AVTF_Ent_M3 : Bool;
      NXT_Avance : Bool;
      PTF_Mx_MSig : Bool;
      V_CNT_ApHsMx_S2 : UDInt;   // Valor del Contador de ausencia en S2
      V_CNT_ApHsMx_E1 : UDInt;   // Valor del Contador de ausencia en E1
      V_CNT_ApHsMx_E3 : UDInt;   // Valor del Contador de ausencia en S3
      V_Paro : UDInt;
      V_TOut_Tx_Mx : UDInt;
      V_TOut_TR : UDInt;
      V_RepartoColector : UDInt;
   END_VAR
   VAR_OUTPUT
      PTF_Ent_M1 : Bool;
      PTF_Ent_M3 : Bool;
      AVTF_Mx_MSig : Bool;
   END_VAR
   VAR_IN_OUT
      Mem_tmp_Paro : Bool;
      MemAuxFN_E1 : Bool;
      MemFN_pHsE1 : Bool;
      MemFP_pHsE1 : Bool;
      MemAuxFN_E3 : Bool;
      MemFN_pHsE3 : Bool;
      MemAuxFN_S2 : Bool;
      MemFN_pHsS2 : Bool;
   END_VAR
   VAR_TEMP
      OK_Ausencia_Entrada : Bool;
      OK_Ausencia_salida : Bool;
      ok_vaciado : Bool;
      Error_Atasco : Bool;
      Error_TOut_TR : Bool;
      TEMP_MA_TR_PosE1E3 : Bool;
      TEMP_MA_TR_PosS2 : Bool;
      ok_tension : Bool;
      v_ausencia_entrada : UDInt;
   END_VAR
   VAR_TEMP   // added for the SCL form of the ladder/FBD networks
      _w1 : Bool;
      _w2 : Bool;
      _w3 : Bool;
      _w4 : Bool;
      _w5 : Bool;
      _w6 : Bool;
   END_VAR
BEGIN

REGION Network 1: Marca General Error
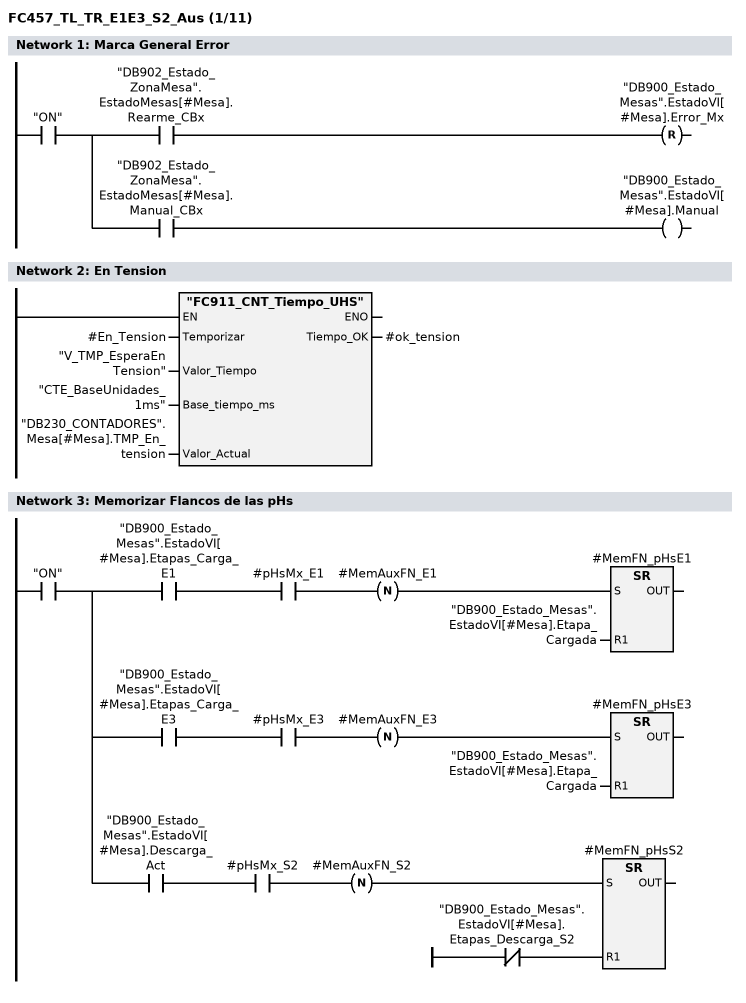
   RUNG wire#powerrail
      Contact( "ON" )
      wire#w1
      Contact( "DB902_Estado_ZonaMesa".EstadoMesas[#Mesa].Rearme_CBx )
      R_Coil( "DB900_Estado_Mesas".EstadoVI[#Mesa].Error_Mx )
   END_RUNG
   RUNG wire#w1
      Contact( "DB902_Estado_ZonaMesa".EstadoMesas[#Mesa].Manual_CBx )
      Coil( "DB900_Estado_Mesas".EstadoVI[#Mesa].Manual )
   END_RUNG
   // the same network as SCL:
   IF "ON" AND "DB902_Estado_ZonaMesa".EstadoMesas[#Mesa].Rearme_CBx THEN
       "DB900_Estado_Mesas".EstadoVI[#Mesa].Error_Mx := FALSE;
   END_IF;
   "DB900_Estado_Mesas".EstadoVI[#Mesa].Manual := "ON" AND "DB902_Estado_ZonaMesa".EstadoMesas[#Mesa].Manual_CBx;
END_REGION

REGION Network 2: En Tension
   RUNG wire#powerrail
      "FC911_CNT_Tiempo_UHS"(Temporizar := #En_Tension, Valor_Tiempo := "V_TMP_EsperaEnTension", Base_tiempo_ms := "CTE_BaseUnidades_1ms", Valor_Actual := "DB230_CONTADORES".Mesa[#Mesa].TMP_En_tension, Tiempo_OK => #ok_tension)
   END_RUNG
   // the same network as SCL:
   "FC911_CNT_Tiempo_UHS"(Temporizar := #En_Tension,
                          Valor_Tiempo := "V_TMP_EsperaEnTension",
                          Base_tiempo_ms := "CTE_BaseUnidades_1ms",
                          Valor_Actual := "DB230_CONTADORES".Mesa[#Mesa].TMP_En_tension,
                          Tiempo_OK => #ok_tension);
END_REGION

REGION Network 3: Memorizar Flancos de las pHs
   RUNG wire#powerrail
      Contact( "ON" )
      wire#w1
      Contact( "DB900_Estado_Mesas".EstadoVI[#Mesa].Etapas_Carga_E1 )
      Contact( #pHsMx_E1 )
      N_Trig( #MemAuxFN_E1 )
      S_SR(operand := #MemFN_pHsE1, r1 := "DB900_Estado_Mesas".EstadoVI[#Mesa].Etapa_Cargada)
   END_RUNG
   RUNG wire#w1
      Contact( "DB900_Estado_Mesas".EstadoVI[#Mesa].Etapas_Carga_E3 )
      Contact( #pHsMx_E3 )
      N_Trig( #MemAuxFN_E3 )
      S_SR(operand := #MemFN_pHsE3, r1 := "DB900_Estado_Mesas".EstadoVI[#Mesa].Etapa_Cargada)
   END_RUNG
   RUNG wire#w1
      Contact( "DB900_Estado_Mesas".EstadoVI[#Mesa].Descarga_Act )
      Contact( #pHsMx_S2 )
      N_Trig( #MemAuxFN_S2 )
      S_SR(operand := #MemFN_pHsS2, r1 := wire#w2)
   END_RUNG
   RUNG wire#powerrail
      I_Contact( "DB900_Estado_Mesas".EstadoVI[#Mesa].Etapas_Descarga_S2 )
   END_RUNG wire#w2
   // the same network as SCL:
   #_w1 := "ON" AND "DB900_Estado_Mesas".EstadoVI[#Mesa].Etapas_Carga_E1 AND #pHsMx_E1;
   #_w2 := NOT #_w1 AND #MemAuxFN_E1;   // falling edge
   #MemAuxFN_E1 := #_w1;
   IF #_w2 THEN
       #MemFN_pHsE1 := TRUE;   // SR flip-flop
   END_IF;
   IF "DB900_Estado_Mesas".EstadoVI[#Mesa].Etapa_Cargada THEN #MemFN_pHsE1 := FALSE; END_IF;
   #_w3 := "ON" AND "DB900_Estado_Mesas".EstadoVI[#Mesa].Etapas_Carga_E3 AND #pHsMx_E3;
   #_w4 := NOT #_w3 AND #MemAuxFN_E3;   // falling edge
   #MemAuxFN_E3 := #_w3;
   IF #_w4 THEN
       #MemFN_pHsE3 := TRUE;   // SR flip-flop
   END_IF;
   IF "DB900_Estado_Mesas".EstadoVI[#Mesa].Etapa_Cargada THEN #MemFN_pHsE3 := FALSE; END_IF;
   #_w5 := "ON" AND "DB900_Estado_Mesas".EstadoVI[#Mesa].Descarga_Act AND #pHsMx_S2;
   #_w6 := NOT #_w5 AND #MemAuxFN_S2;   // falling edge
   #MemAuxFN_S2 := #_w5;
   IF #_w6 THEN
       #MemFN_pHsS2 := TRUE;   // SR flip-flop
   END_IF;
   IF NOT "DB900_Estado_Mesas".EstadoVI[#Mesa].Etapas_Descarga_S2 THEN #MemFN_pHsS2 := FALSE; END_IF;
END_REGION

REGION Network 4: contador vaciado
   // Contador ausencia
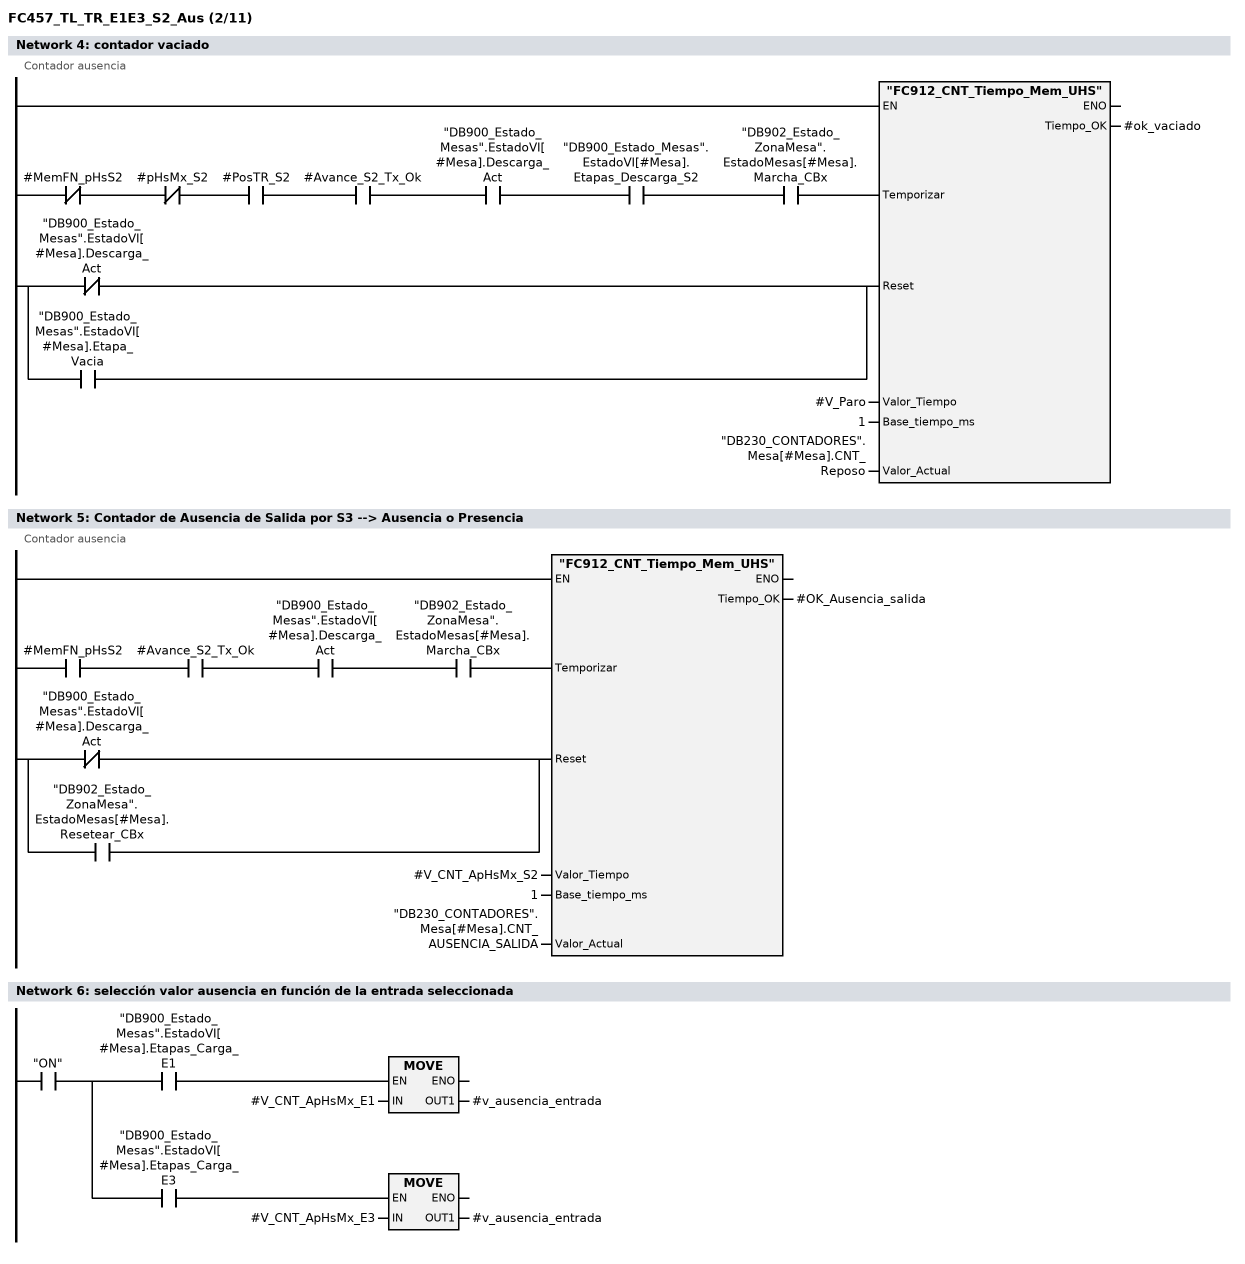
   RUNG wire#powerrail
      "FC912_CNT_Tiempo_Mem_UHS"(Temporizar := wire#w1, Reset := wire#w2, Valor_Tiempo := #V_Paro, Base_tiempo_ms := 1, Valor_Actual := "DB230_CONTADORES".Mesa[#Mesa].CNT_Reposo, Tiempo_OK => #ok_vaciado)
   END_RUNG
   RUNG wire#powerrail
      I_Contact( #MemFN_pHsS2 )
      I_Contact( #pHsMx_S2 )
      Contact( #PosTR_S2 )
      Contact( #Avance_S2_Tx_Ok )
      Contact( "DB900_Estado_Mesas".EstadoVI[#Mesa].Descarga_Act )
      Contact( "DB900_Estado_Mesas".EstadoVI[#Mesa].Etapas_Descarga_S2 )
      Contact( "DB902_Estado_ZonaMesa".EstadoMesas[#Mesa].Marcha_CBx )
   END_RUNG wire#w1
   RUNG wire#powerrail
      I_Contact( "DB900_Estado_Mesas".EstadoVI[#Mesa].Descarga_Act )
   END_RUNG wire#w2
   RUNG wire#powerrail
      Contact( "DB900_Estado_Mesas".EstadoVI[#Mesa].Etapa_Vacia )
   END_RUNG wire#w2
   // the same network as SCL:
   "FC912_CNT_Tiempo_Mem_UHS"(Temporizar := NOT #MemFN_pHsS2 AND NOT #pHsMx_S2 AND #PosTR_S2 AND #Avance_S2_Tx_Ok AND "DB900_Estado_Mesas".EstadoVI[#Mesa].Descarga_Act AND "DB900_Estado_Mesas".EstadoVI[#Mesa].Etapas_Descarga_S2 AND "DB902_Estado_ZonaMesa".EstadoMesas[#Mesa].Marcha_CBx,
                           Reset := NOT "DB900_Estado_Mesas".EstadoVI[#Mesa].Descarga_Act OR "DB900_Estado_Mesas".EstadoVI[#Mesa].Etapa_Vacia,
                           Valor_Tiempo := #V_Paro,
                           Base_tiempo_ms := 1,
                           Valor_Actual := "DB230_CONTADORES".Mesa[#Mesa].CNT_Reposo,
                           Tiempo_OK => #ok_vaciado);
END_REGION

REGION Network 5: Contador de Ausencia de Salida por S3 --> Ausencia o Presencia
   // Contador ausencia
   RUNG wire#powerrail
      "FC912_CNT_Tiempo_Mem_UHS"(Temporizar := wire#w1, Reset := wire#w2, Valor_Tiempo := #V_CNT_ApHsMx_S2, Base_tiempo_ms := 1, Valor_Actual := "DB230_CONTADORES".Mesa[#Mesa].CNT_AUSENCIA_SALIDA, Tiempo_OK => #OK_Ausencia_salida)
   END_RUNG
   RUNG wire#powerrail
      Contact( #MemFN_pHsS2 )
      Contact( #Avance_S2_Tx_Ok )
      Contact( "DB900_Estado_Mesas".EstadoVI[#Mesa].Descarga_Act )
      Contact( "DB902_Estado_ZonaMesa".EstadoMesas[#Mesa].Marcha_CBx )
   END_RUNG wire#w1
   RUNG wire#powerrail
      I_Contact( "DB900_Estado_Mesas".EstadoVI[#Mesa].Descarga_Act )
   END_RUNG wire#w2
   RUNG wire#powerrail
      Contact( "DB902_Estado_ZonaMesa".EstadoMesas[#Mesa].Resetear_CBx )
   END_RUNG wire#w2
   // the same network as SCL:
   "FC912_CNT_Tiempo_Mem_UHS"(Temporizar := #MemFN_pHsS2 AND #Avance_S2_Tx_Ok AND "DB900_Estado_Mesas".EstadoVI[#Mesa].Descarga_Act AND "DB902_Estado_ZonaMesa".EstadoMesas[#Mesa].Marcha_CBx,
                           Reset := NOT "DB900_Estado_Mesas".EstadoVI[#Mesa].Descarga_Act OR "DB902_Estado_ZonaMesa".EstadoMesas[#Mesa].Resetear_CBx,
                           Valor_Tiempo := #V_CNT_ApHsMx_S2,
                           Base_tiempo_ms := 1,
                           Valor_Actual := "DB230_CONTADORES".Mesa[#Mesa].CNT_AUSENCIA_SALIDA,
                           Tiempo_OK => #OK_Ausencia_salida);
END_REGION

REGION Network 6: selección valor ausencia en función de la entrada seleccionada
   RUNG wire#powerrail
      Contact( "ON" )
      wire#w1
      Contact( "DB900_Estado_Mesas".EstadoVI[#Mesa].Etapas_Carga_E1 )
      Move(in := #V_CNT_ApHsMx_E1, out1 => #v_ausencia_entrada)
   END_RUNG
   RUNG wire#w1
      Contact( "DB900_Estado_Mesas".EstadoVI[#Mesa].Etapas_Carga_E3 )
      Move(in := #V_CNT_ApHsMx_E3, out1 => #v_ausencia_entrada)
   END_RUNG
   // the same network as SCL:
   IF "ON" AND "DB900_Estado_Mesas".EstadoVI[#Mesa].Etapas_Carga_E1 THEN
       #v_ausencia_entrada := #V_CNT_ApHsMx_E1;
   END_IF;
   IF "ON" AND "DB900_Estado_Mesas".EstadoVI[#Mesa].Etapas_Carga_E3 THEN
       #v_ausencia_entrada := #V_CNT_ApHsMx_E3;
   END_IF;
END_REGION

REGION Network 7: Contador de Ausencia de Entrada
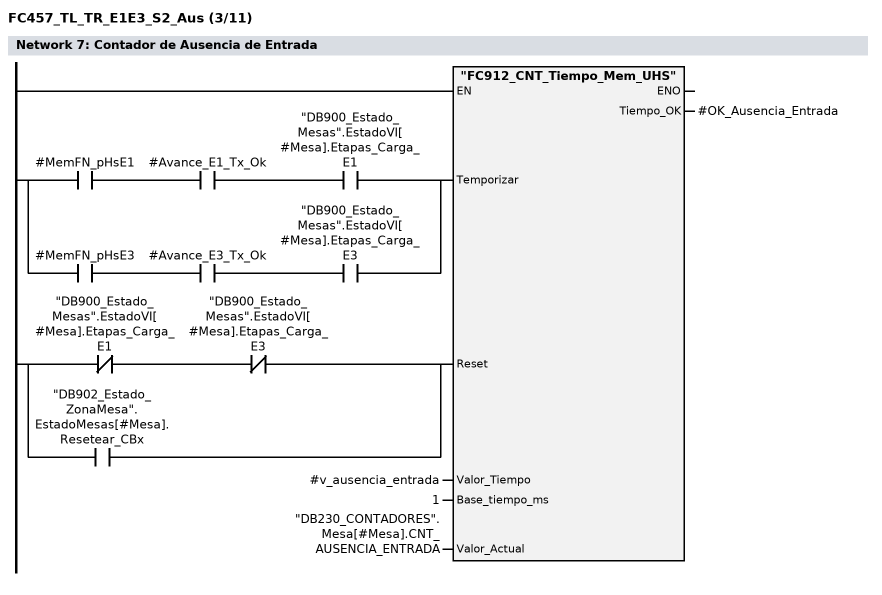
   RUNG wire#powerrail
      "FC912_CNT_Tiempo_Mem_UHS"(Temporizar := wire#w1, Reset := wire#w2, Valor_Tiempo := #v_ausencia_entrada, Base_tiempo_ms := 1, Valor_Actual := "DB230_CONTADORES".Mesa[#Mesa].CNT_AUSENCIA_ENTRADA, Tiempo_OK => #OK_Ausencia_Entrada)
   END_RUNG
   RUNG wire#powerrail
      Contact( #MemFN_pHsE1 )
      Contact( #Avance_E1_Tx_Ok )
      Contact( "DB900_Estado_Mesas".EstadoVI[#Mesa].Etapas_Carga_E1 )
   END_RUNG wire#w1
   RUNG wire#powerrail
      Contact( #MemFN_pHsE3 )
      Contact( #Avance_E3_Tx_Ok )
      Contact( "DB900_Estado_Mesas".EstadoVI[#Mesa].Etapas_Carga_E3 )
   END_RUNG wire#w1
   RUNG wire#powerrail
      I_Contact( "DB900_Estado_Mesas".EstadoVI[#Mesa].Etapas_Carga_E1 )
      I_Contact( "DB900_Estado_Mesas".EstadoVI[#Mesa].Etapas_Carga_E3 )
   END_RUNG wire#w2
   RUNG wire#powerrail
      Contact( "DB902_Estado_ZonaMesa".EstadoMesas[#Mesa].Resetear_CBx )
   END_RUNG wire#w2
   // the same network as SCL:
   "FC912_CNT_Tiempo_Mem_UHS"(Temporizar := (#MemFN_pHsE1 AND #Avance_E1_Tx_Ok AND "DB900_Estado_Mesas".EstadoVI[#Mesa].Etapas_Carga_E1) OR (#MemFN_pHsE3 AND #Avance_E3_Tx_Ok AND "DB900_Estado_Mesas".EstadoVI[#Mesa].Etapas_Carga_E3),
                           Reset := (NOT "DB900_Estado_Mesas".EstadoVI[#Mesa].Etapas_Carga_E1 AND NOT "DB900_Estado_Mesas".EstadoVI[#Mesa].Etapas_Carga_E3) OR "DB902_Estado_ZonaMesa".EstadoMesas[#Mesa].Resetear_CBx,
                           Valor_Tiempo := #v_ausencia_entrada,
                           Base_tiempo_ms := 1,
                           Valor_Actual := "DB230_CONTADORES".Mesa[#Mesa].CNT_AUSENCIA_ENTRADA,
                           Tiempo_OK => #OK_Ausencia_Entrada);
END_REGION

REGION Network 8: Temporizador de PARO
   // Modif Dani: El contador se activa además de con MA_avance_Tx, con el 
   // MA_Avance_TR, pq sino, no se resetean las variables de Mem_Act_E1, E2 tras un 
   // reset
